REGION Network 8: IMMEDIATE STOP ALARMS
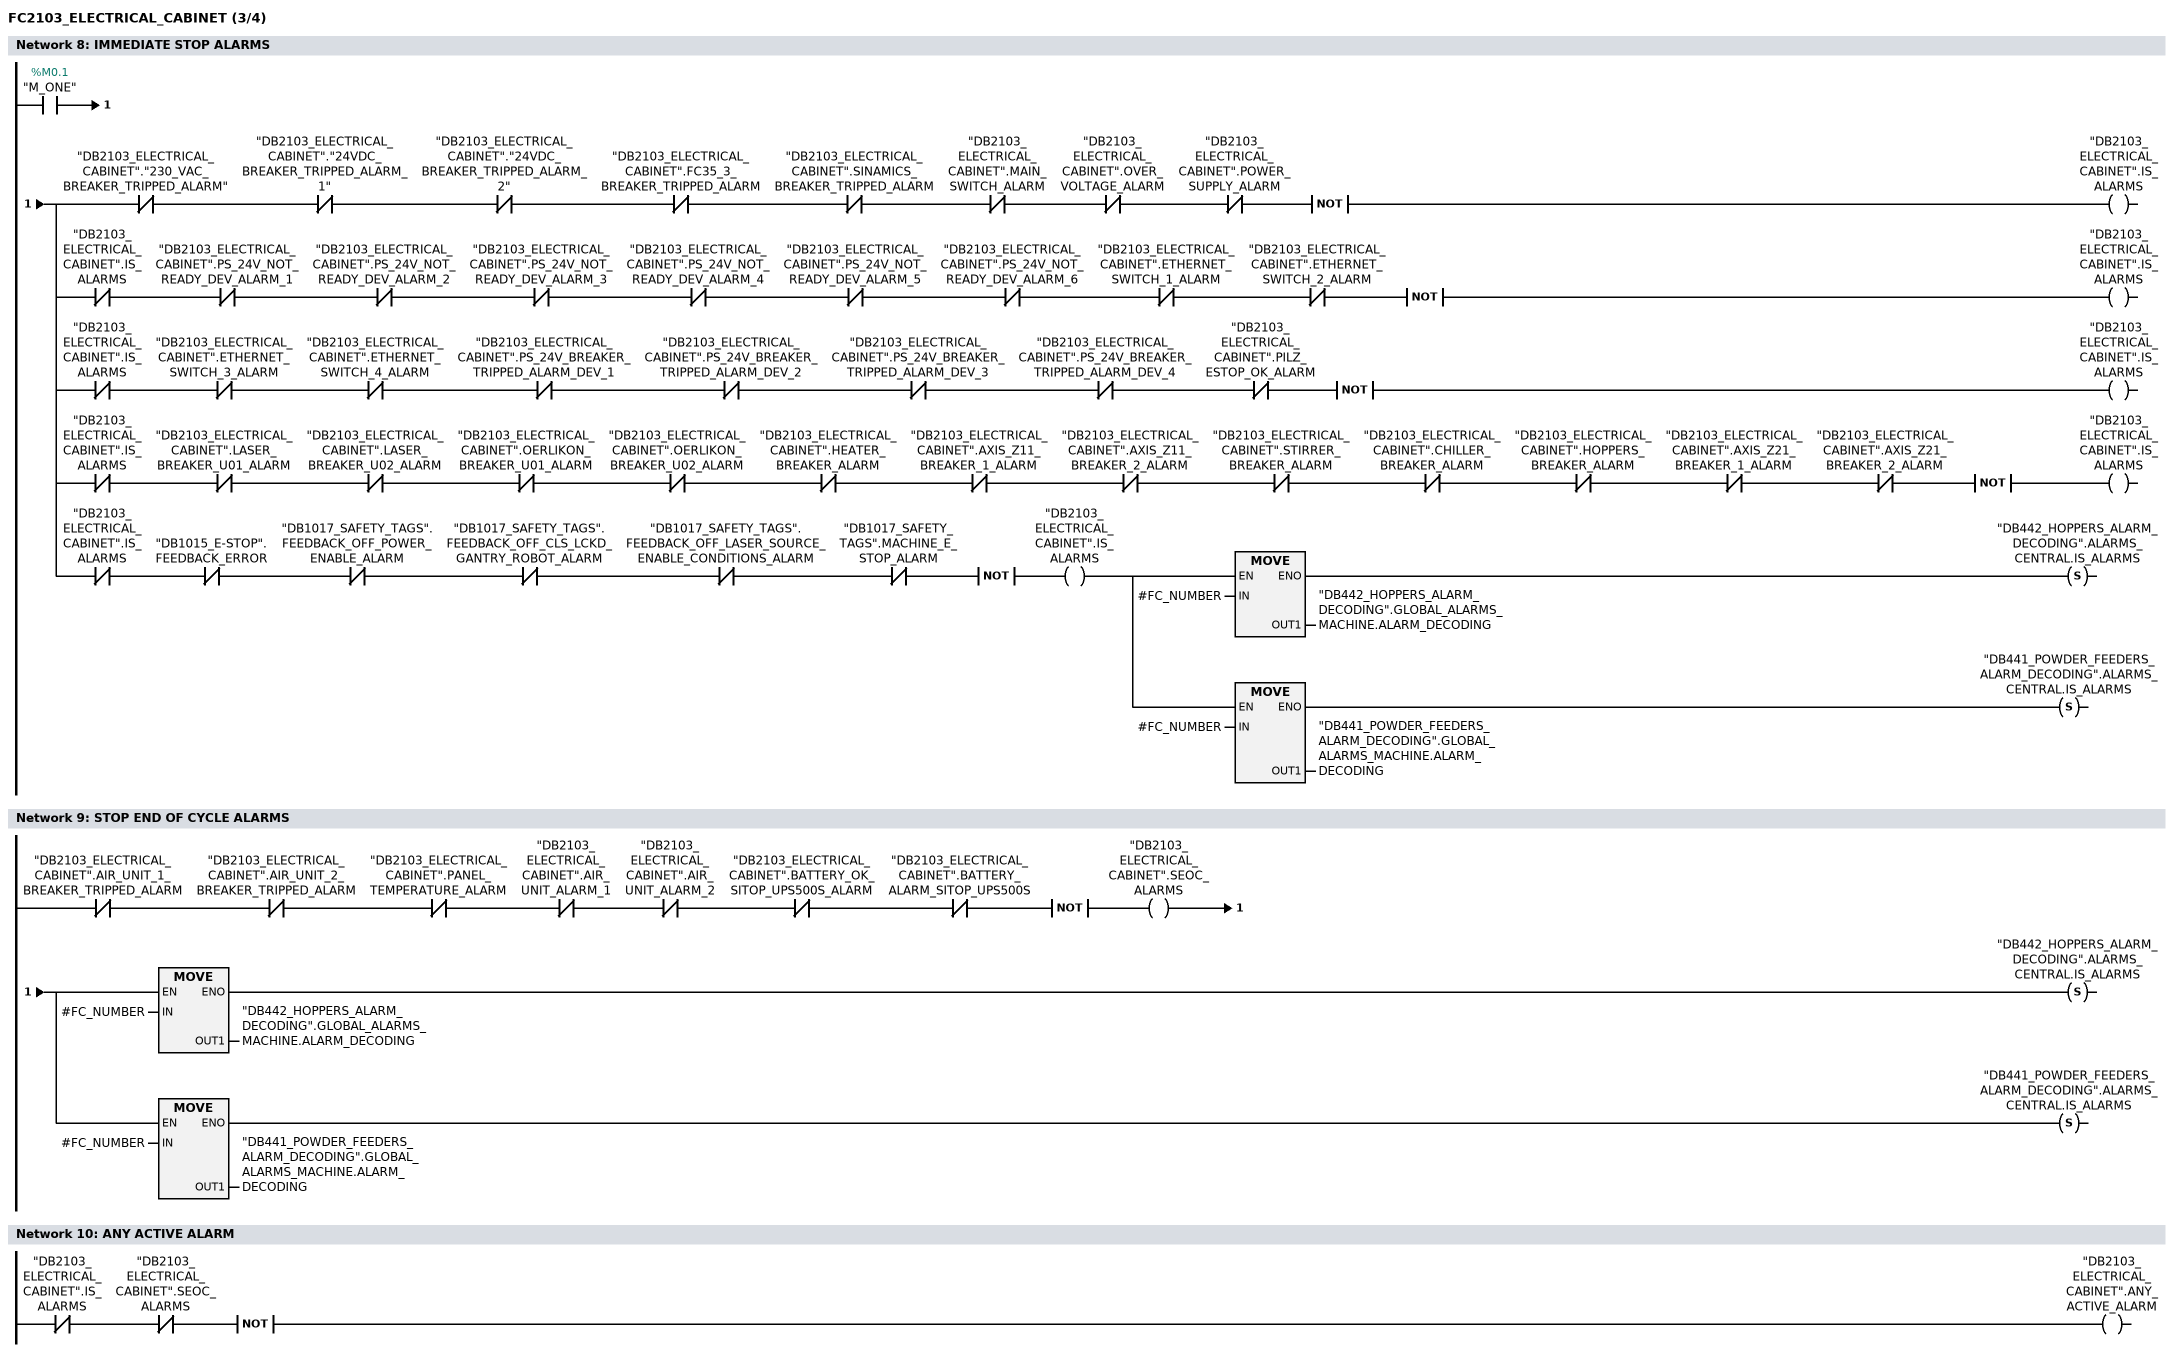
   RUNG wire#powerrail
      Contact( "M_ONE" )
      wire#w1
      I_Contact( "DB2103_ELECTRICAL_CABINET"."230_VAC_BREAKER_TRIPPED_ALARM" )
      I_Contact( "DB2103_ELECTRICAL_CABINET"."24VDC_BREAKER_TRIPPED_ALARM_1" )
      I_Contact( "DB2103_ELECTRICAL_CABINET"."24VDC_BREAKER_TRIPPED_ALARM_2" )
      I_Contact( "DB2103_ELECTRICAL_CABINET".FC35_3_BREAKER_TRIPPED_ALARM )
      I_Contact( "DB2103_ELECTRICAL_CABINET".SINAMICS_BREAKER_TRIPPED_ALARM )
      I_Contact( "DB2103_ELECTRICAL_CABINET".MAIN_SWITCH_ALARM )
      I_Contact( "DB2103_ELECTRICAL_CABINET".OVER_VOLTAGE_ALARM )
      I_Contact( "DB2103_ELECTRICAL_CABINET".POWER_SUPPLY_ALARM )
      Not()
      Coil( "DB2103_ELECTRICAL_CABINET".IS_ALARMS )
   END_RUNG
   RUNG wire#w1
      I_Contact( "DB2103_ELECTRICAL_CABINET".IS_ALARMS )
      I_Contact( "DB2103_ELECTRICAL_CABINET".PS_24V_NOT_READY_DEV_ALARM_1 )
      I_Contact( "DB2103_ELECTRICAL_CABINET".PS_24V_NOT_READY_DEV_ALARM_2 )
      I_Contact( "DB2103_ELECTRICAL_CABINET".PS_24V_NOT_READY_DEV_ALARM_3 )
      I_Contact( "DB2103_ELECTRICAL_CABINET".PS_24V_NOT_READY_DEV_ALARM_4 )
      I_Contact( "DB2103_ELECTRICAL_CABINET".PS_24V_NOT_READY_DEV_ALARM_5 )
      I_Contact( "DB2103_ELECTRICAL_CABINET".PS_24V_NOT_READY_DEV_ALARM_6 )
      I_Contact( "DB2103_ELECTRICAL_CABINET".ETHERNET_SWITCH_1_ALARM )
      I_Contact( "DB2103_ELECTRICAL_CABINET".ETHERNET_SWITCH_2_ALARM )
      Not()
      Coil( "DB2103_ELECTRICAL_CABINET".IS_ALARMS )
   END_RUNG
   RUNG wire#w1
      I_Contact( "DB2103_ELECTRICAL_CABINET".IS_ALARMS )
      I_Contact( "DB2103_ELECTRICAL_CABINET".ETHERNET_SWITCH_3_ALARM )
      I_Contact( "DB2103_ELECTRICAL_CABINET".ETHERNET_SWITCH_4_ALARM )
      I_Contact( "DB2103_ELECTRICAL_CABINET".PS_24V_BREAKER_TRIPPED_ALARM_DEV_1 )
      I_Contact( "DB2103_ELECTRICAL_CABINET".PS_24V_BREAKER_TRIPPED_ALARM_DEV_2 )
      I_Contact( "DB2103_ELECTRICAL_CABINET".PS_24V_BREAKER_TRIPPED_ALARM_DEV_3 )
      I_Contact( "DB2103_ELECTRICAL_CABINET".PS_24V_BREAKER_TRIPPED_ALARM_DEV_4 )
      I_Contact( "DB2103_ELECTRICAL_CABINET".PILZ_ESTOP_OK_ALARM )
      Not()
      Coil( "DB2103_ELECTRICAL_CABINET".IS_ALARMS )
   END_RUNG
   RUNG wire#w1
      I_Contact( "DB2103_ELECTRICAL_CABINET".IS_ALARMS )
      I_Contact( "DB2103_ELECTRICAL_CABINET".LASER_BREAKER_U01_ALARM )
      I_Contact( "DB2103_ELECTRICAL_CABINET".LASER_BREAKER_U02_ALARM )
      I_Contact( "DB2103_ELECTRICAL_CABINET".OERLIKON_BREAKER_U01_ALARM )
      I_Contact( "DB2103_ELECTRICAL_CABINET".OERLIKON_BREAKER_U02_ALARM )
      I_Contact( "DB2103_ELECTRICAL_CABINET".HEATER_BREAKER_ALARM )
      I_Contact( "DB2103_ELECTRICAL_CABINET".AXIS_Z11_BREAKER_1_ALARM )
      I_Contact( "DB2103_ELECTRICAL_CABINET".AXIS_Z11_BREAKER_2_ALARM )
      I_Contact( "DB2103_ELECTRICAL_CABINET".STIRRER_BREAKER_ALARM )
      I_Contact( "DB2103_ELECTRICAL_CABINET".CHILLER_BREAKER_ALARM )
      I_Contact( "DB2103_ELECTRICAL_CABINET".HOPPERS_BREAKER_ALARM )
      I_Contact( "DB2103_ELECTRICAL_CABINET".AXIS_Z21_BREAKER_1_ALARM )
      I_Contact( "DB2103_ELECTRICAL_CABINET".AXIS_Z21_BREAKER_2_ALARM )
      Not()
      Coil( "DB2103_ELECTRICAL_CABINET".IS_ALARMS )
   END_RUNG
   RUNG wire#w1
      I_Contact( "DB2103_ELECTRICAL_CABINET".IS_ALARMS )
      I_Contact( "DB1015_E-STOP".FEEDBACK_ERROR )
      I_Contact( "DB1017_SAFETY_TAGS".FEEDBACK_OFF_POWER_ENABLE_ALARM )
      I_Contact( "DB1017_SAFETY_TAGS".FEEDBACK_OFF_CLS_LCKD_GANTRY_ROBOT_ALARM )
      I_Contact( "DB1017_SAFETY_TAGS".FEEDBACK_OFF_LASER_SOURCE_ENABLE_CONDITIONS_ALARM )
      I_Contact( "DB1017_SAFETY_TAGS".MACHINE_E_STOP_ALARM )
      Not()
      Coil( "DB2103_ELECTRICAL_CABINET".IS_ALARMS )
      wire#w2
      { S7_GenerateENO := "TRUE" } Move(in := #FC_NUMBER, out1 => "DB442_HOPPERS_ALARM_DECODING".GLOBAL_ALARMS_MACHINE.ALARM_DECODING)
      S_Coil( "DB442_HOPPERS_ALARM_DECODING".ALARMS_CENTRAL.IS_ALARMS )
   END_RUNG
   RUNG wire#w2
      { S7_GenerateENO := "TRUE" } Move(in := #FC_NUMBER, out1 => "DB441_POWDER_FEEDERS_ALARM_DECODING".GLOBAL_ALARMS_MACHINE.ALARM_DECODING)
      S_Coil( "DB441_POWDER_FEEDERS_ALARM_DECODING".ALARMS_CENTRAL.IS_ALARMS )
   END_RUNG
   // the same network as SCL:
   // ENO of a box is taken as its EN; it also drops when the box reports an error
   "DB2103_ELECTRICAL_CABINET".IS_ALARMS := NOT ("M_ONE" AND NOT "DB2103_ELECTRICAL_CABINET"."230_VAC_BREAKER_TRIPPED_ALARM" AND NOT "DB2103_ELECTRICAL_CABINET"."24VDC_BREAKER_TRIPPED_ALARM_1" AND NOT "DB2103_ELECTRICAL_CABINET"."24VDC_BREAKER_TRIPPED_ALARM_2" AND NOT "DB2103_ELECTRICAL_CABINET".FC35_3_BREAKER_TRIPPED_ALARM AND NOT "DB2103_ELECTRICAL_CABINET".SINAMICS_BREAKER_TRIPPED_ALARM AND NOT "DB2103_ELECTRICAL_CABINET".MAIN_SWITCH_ALARM AND NOT "DB2103_ELECTRICAL_CABINET".OVER_VOLTAGE_ALARM AND NOT "DB2103_ELECTRICAL_CABINET".POWER_SUPPLY_ALARM);
   "DB2103_ELECTRICAL_CABINET".IS_ALARMS := NOT ("M_ONE" AND NOT "DB2103_ELECTRICAL_CABINET".IS_ALARMS AND NOT "DB2103_ELECTRICAL_CABINET".PS_24V_NOT_READY_DEV_ALARM_1 AND NOT "DB2103_ELECTRICAL_CABINET".PS_24V_NOT_READY_DEV_ALARM_2 AND NOT "DB2103_ELECTRICAL_CABINET".PS_24V_NOT_READY_DEV_ALARM_3 AND NOT "DB2103_ELECTRICAL_CABINET".PS_24V_NOT_READY_DEV_ALARM_4 AND NOT "DB2103_ELECTRICAL_CABINET".PS_24V_NOT_READY_DEV_ALARM_5 AND NOT "DB2103_ELECTRICAL_CABINET".PS_24V_NOT_READY_DEV_ALARM_6 AND NOT "DB2103_ELECTRICAL_CABINET".ETHERNET_SWITCH_1_ALARM AND NOT "DB2103_ELECTRICAL_CABINET".ETHERNET_SWITCH_2_ALARM);
   "DB2103_ELECTRICAL_CABINET".IS_ALARMS := NOT ("M_ONE" AND NOT "DB2103_ELECTRICAL_CABINET".IS_ALARMS AND NOT "DB2103_ELECTRICAL_CABINET".ETHERNET_SWITCH_3_ALARM AND NOT "DB2103_ELECTRICAL_CABINET".ETHERNET_SWITCH_4_ALARM AND NOT "DB2103_ELECTRICAL_CABINET".PS_24V_BREAKER_TRIPPED_ALARM_DEV_1 AND NOT "DB2103_ELECTRICAL_CABINET".PS_24V_BREAKER_TRIPPED_ALARM_DEV_2 AND NOT "DB2103_ELECTRICAL_CABINET".PS_24V_BREAKER_TRIPPED_ALARM_DEV_3 AND NOT "DB2103_ELECTRICAL_CABINET".PS_24V_BREAKER_TRIPPED_ALARM_DEV_4 AND NOT "DB2103_ELECTRICAL_CABINET".PILZ_ESTOP_OK_ALARM);
   "DB2103_ELECTRICAL_CABINET".IS_ALARMS := NOT ("M_ONE" AND NOT "DB2103_ELECTRICAL_CABINET".IS_ALARMS AND NOT "DB2103_ELECTRICAL_CABINET".LASER_BREAKER_U01_ALARM AND NOT "DB2103_ELECTRICAL_CABINET".LASER_BREAKER_U02_ALARM AND NOT "DB2103_ELECTRICAL_CABINET".OERLIKON_BREAKER_U01_ALARM AND NOT "DB2103_ELECTRICAL_CABINET".OERLIKON_BREAKER_U02_ALARM AND NOT "DB2103_ELECTRICAL_CABINET".HEATER_BREAKER_ALARM AND NOT "DB2103_ELECTRICAL_CABINET".AXIS_Z11_BREAKER_1_ALARM AND NOT "DB2103_ELECTRICAL_CABINET".AXIS_Z11_BREAKER_2_ALARM AND NOT "DB2103_ELECTRICAL_CABINET".STIRRER_BREAKER_ALARM AND NOT "DB2103_ELECTRICAL_CABINET".CHILLER_BREAKER_ALARM AND NOT "DB2103_ELECTRICAL_CABINET".HOPPERS_BREAKER_ALARM AND NOT "DB2103_ELECTRICAL_CABINET".AXIS_Z21_BREAKER_1_ALARM AND NOT "DB2103_ELECTRICAL_CABINET".AXIS_Z21_BREAKER_2_ALARM);
   "DB2103_ELECTRICAL_CABINET".IS_ALARMS := NOT ("M_ONE" AND NOT "DB2103_ELECTRICAL_CABINET".IS_ALARMS AND NOT "DB1015_E-STOP".FEEDBACK_ERROR AND NOT "DB1017_SAFETY_TAGS".FEEDBACK_OFF_POWER_ENABLE_ALARM AND NOT "DB1017_SAFETY_TAGS".FEEDBACK_OFF_CLS_LCKD_GANTRY_ROBOT_ALARM AND NOT "DB1017_SAFETY_TAGS".FEEDBACK_OFF_LASER_SOURCE_ENABLE_CONDITIONS_ALARM AND NOT "DB1017_SAFETY_TAGS".MACHINE_E_STOP_ALARM);
   IF "DB2103_ELECTRICAL_CABINET".IS_ALARMS THEN
       "DB442_HOPPERS_ALARM_DECODING".GLOBAL_ALARMS_MACHINE.ALARM_DECODING := #FC_NUMBER;
       "DB442_HOPPERS_ALARM_DECODING".ALARMS_CENTRAL.IS_ALARMS := TRUE;
       "DB441_POWDER_FEEDERS_ALARM_DECODING".GLOBAL_ALARMS_MACHINE.ALARM_DECODING := #FC_NUMBER;
       "DB441_POWDER_FEEDERS_ALARM_DECODING".ALARMS_CENTRAL.IS_ALARMS := TRUE;
   END_IF;
END_REGION

REGION Network 9: STOP END OF CYCLE ALARMS
   RUNG wire#powerrail
      I_Contact( "DB2103_ELECTRICAL_CABINET".AIR_UNIT_1_BREAKER_TRIPPED_ALARM )
      I_Contact( "DB2103_ELECTRICAL_CABINET".AIR_UNIT_2_BREAKER_TRIPPED_ALARM )
      I_Contact( "DB2103_ELECTRICAL_CABINET".PANEL_TEMPERATURE_ALARM )
      I_Contact( "DB2103_ELECTRICAL_CABINET".AIR_UNIT_ALARM_1 )
      I_Contact( "DB2103_ELECTRICAL_CABINET".AIR_UNIT_ALARM_2 )
      I_Contact( "DB2103_ELECTRICAL_CABINET".BATTERY_OK_SITOP_UPS500S_ALARM )
      I_Contact( "DB2103_ELECTRICAL_CABINET".BATTERY_ALARM_SITOP_UPS500S )
      Not()
      Coil( "DB2103_ELECTRICAL_CABINET".SEOC_ALARMS )
      wire#w1
      { S7_GenerateENO := "TRUE" } Move(in := #FC_NUMBER, out1 => "DB442_HOPPERS_ALARM_DECODING".GLOBAL_ALARMS_MACHINE.ALARM_DECODING)
      S_Coil( "DB442_HOPPERS_ALARM_DECODING".ALARMS_CENTRAL.IS_ALARMS )
   END_RUNG
   RUNG wire#w1
      { S7_GenerateENO := "TRUE" } Move(in := #FC_NUMBER, out1 => "DB441_POWDER_FEEDERS_ALARM_DECODING".GLOBAL_ALARMS_MACHINE.ALARM_DECODING)
      S_Coil( "DB441_POWDER_FEEDERS_ALARM_DECODING".ALARMS_CENTRAL.IS_ALARMS )
   END_RUNG
   // the same network as SCL:
   // ENO of a box is taken as its EN; it also drops when the box reports an error
   "DB2103_ELECTRICAL_CABINET".SEOC_ALARMS := NOT (NOT "DB2103_ELECTRICAL_CABINET".AIR_UNIT_1_BREAKER_TRIPPED_ALARM AND NOT "DB2103_ELECTRICAL_CABINET".AIR_UNIT_2_BREAKER_TRIPPED_ALARM AND NOT "DB2103_ELECTRICAL_CABINET".PANEL_TEMPERATURE_ALARM AND NOT "DB2103_ELECTRICAL_CABINET".AIR_UNIT_ALARM_1 AND NOT "DB2103_ELECTRICAL_CABINET".AIR_UNIT_ALARM_2 AND NOT "DB2103_ELECTRICAL_CABINET".BATTERY_OK_SITOP_UPS500S_ALARM AND NOT "DB2103_ELECTRICAL_CABINET".BATTERY_ALARM_SITOP_UPS500S);
   IF "DB2103_ELECTRICAL_CABINET".SEOC_ALARMS THEN
       "DB442_HOPPERS_ALARM_DECODING".GLOBAL_ALARMS_MACHINE.ALARM_DECODING := #FC_NUMBER;
       "DB442_HOPPERS_ALARM_DECODING".ALARMS_CENTRAL.IS_ALARMS := TRUE;
       "DB441_POWDER_FEEDERS_ALARM_DECODING".GLOBAL_ALARMS_MACHINE.ALARM_DECODING := #FC_NUMBER;
       "DB441_POWDER_FEEDERS_ALARM_DECODING".ALARMS_CENTRAL.IS_ALARMS := TRUE;
   END_IF;
END_REGION

REGION Network 10: ANY ACTIVE ALARM
   RUNG wire#powerrail
      I_Contact( "DB2103_ELECTRICAL_CABINET".IS_ALARMS )
      I_Contact( "DB2103_ELECTRICAL_CABINET".SEOC_ALARMS )
      Not()
      Coil( "DB2103_ELECTRICAL_CABINET".ANY_ACTIVE_ALARM )
   END_RUNG
   // the same network as SCL:
   "DB2103_ELECTRICAL_CABINET".ANY_ACTIVE_ALARM := NOT (NOT "DB2103_ELECTRICAL_CABINET".IS_ALARMS AND NOT "DB2103_ELECTRICAL_CABINET".SEOC_ALARMS);
END_REGION

REGION Network 11: WARNINGS
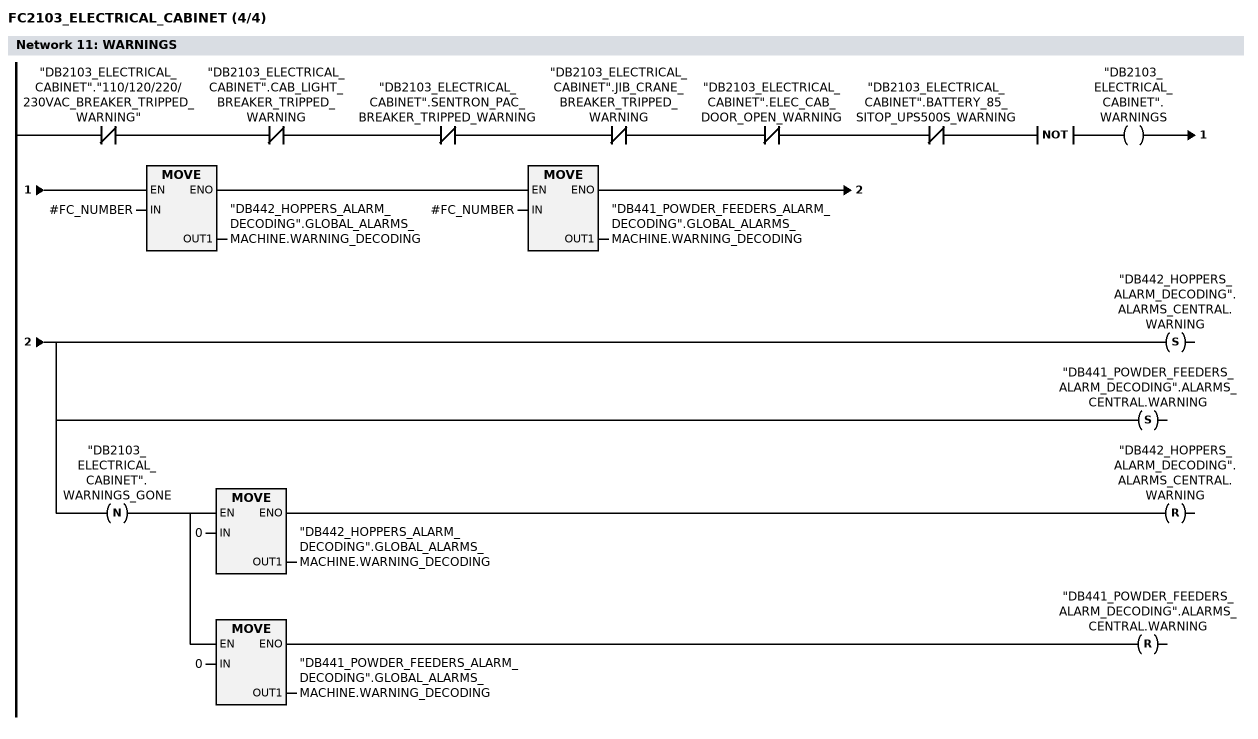
   RUNG wire#powerrail
      I_Contact( "DB2103_ELECTRICAL_CABINET"."110/120/220/230VAC_BREAKER_TRIPPED_WARNING" )
      I_Contact( "DB2103_ELECTRICAL_CABINET".CAB_LIGHT_BREAKER_TRIPPED_WARNING )
      I_Contact( "DB2103_ELECTRICAL_CABINET".SENTRON_PAC_BREAKER_TRIPPED_WARNING )
      I_Contact( "DB2103_ELECTRICAL_CABINET".JIB_CRANE_BREAKER_TRIPPED_WARNING )
      I_Contact( "DB2103_ELECTRICAL_CABINET".ELEC_CAB_DOOR_OPEN_WARNING )
      I_Contact( "DB2103_ELECTRICAL_CABINET".BATTERY_85_SITOP_UPS500S_WARNING )
      Not()
      Coil( "DB2103_ELECTRICAL_CABINET".WARNINGS )
      { S7_GenerateENO := "TRUE" } Move(in := #FC_NUMBER, out1 => "DB442_HOPPERS_ALARM_DECODING".GLOBAL_ALARMS_MACHINE.WARNING_DECODING)
      { S7_GenerateENO := "TRUE" } Move(in := #FC_NUMBER, out1 => "DB441_POWDER_FEEDERS_ALARM_DECODING".GLOBAL_ALARMS_MACHINE.WARNING_DECODING)
      wire#w1
      S_Coil( "DB442_HOPPERS_ALARM_DECODING".ALARMS_CENTRAL.WARNING )
   END_RUNG
   RUNG wire#w1
      S_Coil( "DB441_POWDER_FEEDERS_ALARM_DECODING".ALARMS_CENTRAL.WARNING )
   END_RUNG
   RUNG wire#w1
      N_Trig( "DB2103_ELECTRICAL_CABINET".WARNINGS_GONE )
      wire#w2
      { S7_GenerateENO := "TRUE" } Move(in := 0, out1 => "DB442_HOPPERS_ALARM_DECODING".GLOBAL_ALARMS_MACHINE.WARNING_DECODING)
      R_Coil( "DB442_HOPPERS_ALARM_DECODING".ALARMS_CENTRAL.WARNING )
   END_RUNG
   RUNG wire#w2
      { S7_GenerateENO := "TRUE" } Move(in := 0, out1 => "DB441_POWDER_FEEDERS_ALARM_DECODING".GLOBAL_ALARMS_MACHINE.WARNING_DECODING)
      R_Coil( "DB441_POWDER_FEEDERS_ALARM_DECODING".ALARMS_CENTRAL.WARNING )
   END_RUNG
   // the same network as SCL:
   // ENO of a box is taken as its EN; it also drops when the box reports an error
   "DB2103_ELECTRICAL_CABINET".WARNINGS := NOT (NOT "DB2103_ELECTRICAL_CABINET"."110/120/220/230VAC_BREAKER_TRIPPED_WARNING" AND NOT "DB2103_ELECTRICAL_CABINET".CAB_LIGHT_BREAKER_TRIPPED_WARNING AND NOT "DB2103_ELECTRICAL_CABINET".SENTRON_PAC_BREAKER_TRIPPED_WARNING AND NOT "DB2103_ELECTRICAL_CABINET".JIB_CRANE_BREAKER_TRIPPED_WARNING AND NOT "DB2103_ELECTRICAL_CABINET".ELEC_CAB_DOOR_OPEN_WARNING AND NOT "DB2103_ELECTRICAL_CABINET".BATTERY_85_SITOP_UPS500S_WARNING);
   IF "DB2103_ELECTRICAL_CABINET".WARNINGS THEN
       "DB442_HOPPERS_ALARM_DECODING".GLOBAL_ALARMS_MACHINE.WARNING_DECODING := #FC_NUMBER;
       "DB441_POWDER_FEEDERS_ALARM_DECODING".GLOBAL_ALARMS_MACHINE.WARNING_DECODING := #FC_NUMBER;
       "DB442_HOPPERS_ALARM_DECODING".ALARMS_CENTRAL.WARNING := TRUE;
       "DB441_POWDER_FEEDERS_ALARM_DECODING".ALARMS_CENTRAL.WARNING := TRUE;
   END_IF;
   #_w1 := NOT "DB2103_ELECTRICAL_CABINET".WARNINGS AND "DB2103_ELECTRICAL_CABINET".WARNINGS_GONE;   // falling edge
   "DB2103_ELECTRICAL_CABINET".WARNINGS_GONE := "DB2103_ELECTRICAL_CABINET".WARNINGS;
   IF #_w1 THEN
       "DB442_HOPPERS_ALARM_DECODING".GLOBAL_ALARMS_MACHINE.WARNING_DECODING := 0;
       "DB442_HOPPERS_ALARM_DECODING".ALARMS_CENTRAL.WARNING := FALSE;
       "DB441_POWDER_FEEDERS_ALARM_DECODING".GLOBAL_ALARMS_MACHINE.WARNING_DECODING := 0;
       "DB441_POWDER_FEEDERS_ALARM_DECODING".ALARMS_CENTRAL.WARNING := FALSE;
   END_IF;
END_REGION
END_FUNCTION

FUNCTION "FC2120_MPP_ITC_IPC" : Void   // FC2120, LAD
{ S7_Optimized_Access := 'FALSE' }
AUTHOR : ETXETAR
VERSION : 1.0
// stored: AutoNumber false, IsIECCheckEnabled false, SetENOAutomatically false, UDAEnableTagReadback false
   VAR_TEMP
      O_BYTE_0 : Struct   // OPTIONS BYTE 0
         IPC : Bool;   // IPC OPTION
      END_STRUCT;
      TCU_INDEX_SEL : Int;
   END_VAR
   VAR CONSTANT
      FC_NUMBER : DInt := 2120;   // FC NUMBER
   END_VAR
   VAR_TEMP   // added for the SCL form of the ladder/FBD networks
      _w1 : Bool;
      _w2 : Bool;
   END_VAR
BEGIN

REGION Network 1: OPTIONS
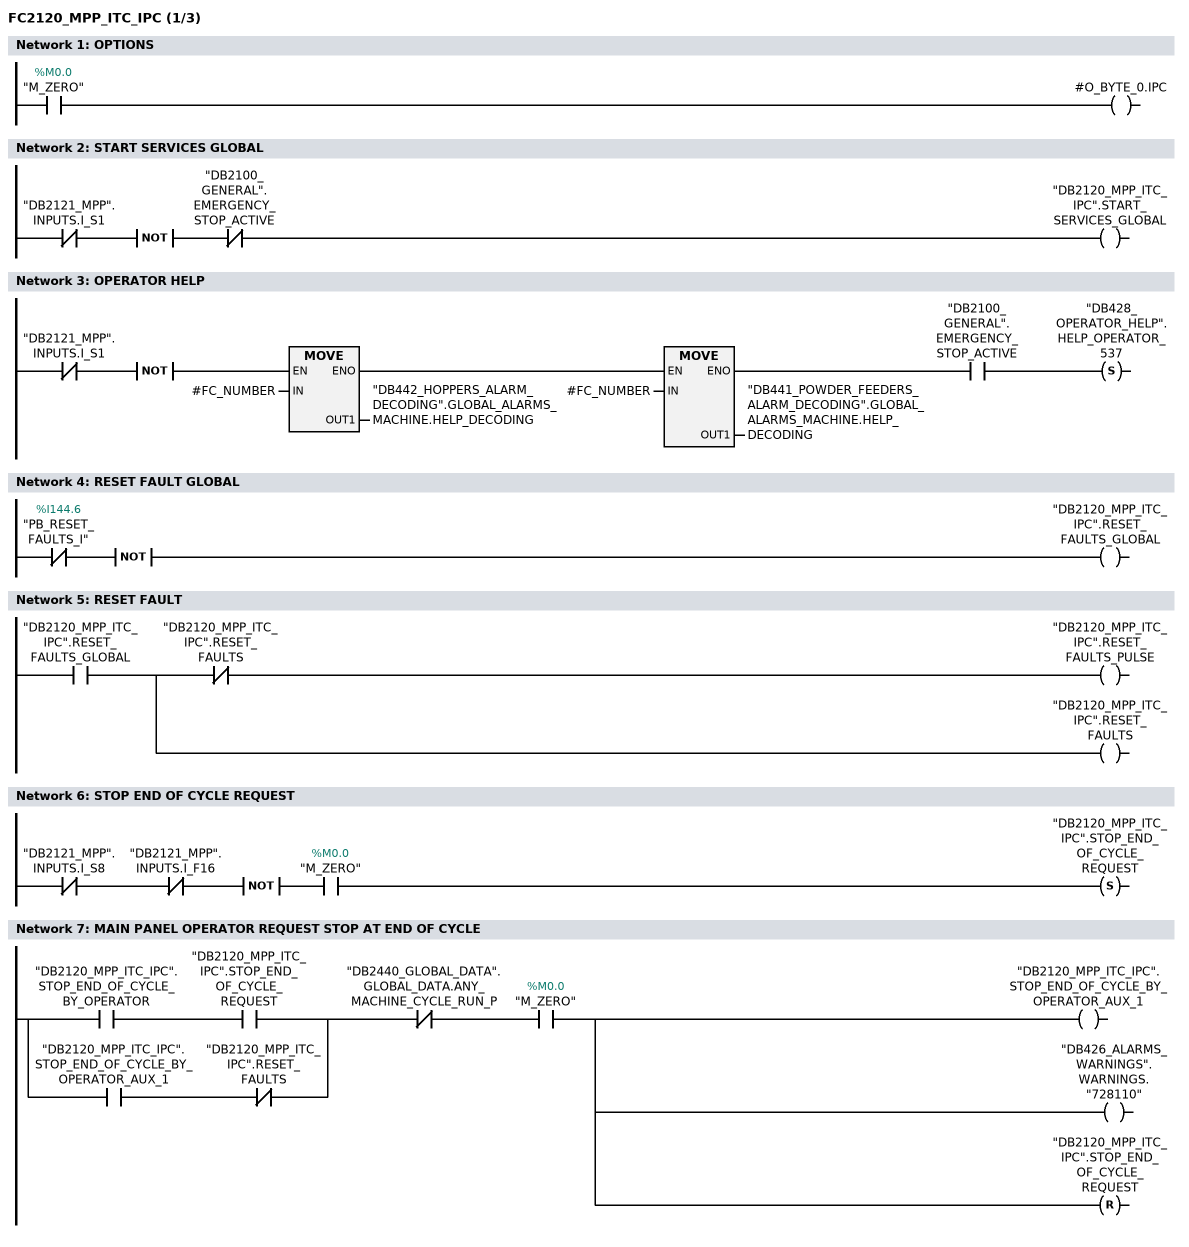
   RUNG wire#powerrail
      Contact( "M_ZERO" )
      Coil( #O_BYTE_0.IPC )
   END_RUNG
   // the same network as SCL:
   #O_BYTE_0.IPC := "M_ZERO";
END_REGION

REGION Network 2: START SERVICES GLOBAL
   RUNG wire#powerrail
      I_Contact( "DB2121_MPP".INPUTS.I_S1 )
      Not()
      I_Contact( "DB2100_GENERAL".EMERGENCY_STOP_ACTIVE )
      Coil( "DB2120_MPP_ITC_IPC".START_SERVICES_GLOBAL )
   END_RUNG
   // the same network as SCL:
   "DB2120_MPP_ITC_IPC".START_SERVICES_GLOBAL := NOT (NOT "DB2121_MPP".INPUTS.I_S1) AND NOT "DB2100_GENERAL".EMERGENCY_STOP_ACTIVE;
END_REGION

REGION Network 3: OPERATOR HELP
   RUNG wire#powerrail
      I_Contact( "DB2121_MPP".INPUTS.I_S1 )
      Not()
      { S7_GenerateENO := "TRUE" } Move(in := #FC_NUMBER, out1 => "DB442_HOPPERS_ALARM_DECODING".GLOBAL_ALARMS_MACHINE.HELP_DECODING)
      { S7_GenerateENO := "TRUE" } Move(in := #FC_NUMBER, out1 => "DB441_POWDER_FEEDERS_ALARM_DECODING".GLOBAL_ALARMS_MACHINE.HELP_DECODING)
      Contact( "DB2100_GENERAL".EMERGENCY_STOP_ACTIVE )
      S_Coil( "DB428_OPERATOR_HELP".HELP_OPERATOR_537 )
   END_RUNG
   // the same network as SCL:
   // ENO of a box is taken as its EN; it also drops when the box reports an error
   #_w1 := NOT (NOT "DB2121_MPP".INPUTS.I_S1);
   IF #_w1 THEN
       "DB442_HOPPERS_ALARM_DECODING".GLOBAL_ALARMS_MACHINE.HELP_DECODING := #FC_NUMBER;
       "DB441_POWDER_FEEDERS_ALARM_DECODING".GLOBAL_ALARMS_MACHINE.HELP_DECODING := #FC_NUMBER;
   END_IF;
   IF #_w1 AND "DB2100_GENERAL".EMERGENCY_STOP_ACTIVE THEN
       "DB428_OPERATOR_HELP".HELP_OPERATOR_537 := TRUE;
   END_IF;
END_REGION

REGION Network 4: RESET FAULT GLOBAL
   RUNG wire#powerrail
      I_Contact( "PB_RESET_FAULTS_I" )
      Not()
      Coil( "DB2120_MPP_ITC_IPC".RESET_FAULTS_GLOBAL )
   END_RUNG
   // the same network as SCL:
   "DB2120_MPP_ITC_IPC".RESET_FAULTS_GLOBAL := NOT (NOT "PB_RESET_FAULTS_I");
END_REGION

REGION Network 5: RESET FAULT
   RUNG wire#powerrail
      Contact( "DB2120_MPP_ITC_IPC".RESET_FAULTS_GLOBAL )
      wire#w1
      I_Contact( "DB2120_MPP_ITC_IPC".RESET_FAULTS )
      Coil( "DB2120_MPP_ITC_IPC".RESET_FAULTS_PULSE )
   END_RUNG
   RUNG wire#w1
      Coil( "DB2120_MPP_ITC_IPC".RESET_FAULTS )
   END_RUNG
   // the same network as SCL:
   "DB2120_MPP_ITC_IPC".RESET_FAULTS_PULSE := "DB2120_MPP_ITC_IPC".RESET_FAULTS_GLOBAL AND NOT "DB2120_MPP_ITC_IPC".RESET_FAULTS;
   "DB2120_MPP_ITC_IPC".RESET_FAULTS := "DB2120_MPP_ITC_IPC".RESET_FAULTS_GLOBAL;
END_REGION

REGION Network 6: STOP END OF CYCLE REQUEST
   RUNG wire#powerrail
      I_Contact( "DB2121_MPP".INPUTS.I_S8 )
      I_Contact( "DB2121_MPP".INPUTS.I_F16 )
      Not()
      Contact( "M_ZERO" )
      S_Coil( "DB2120_MPP_ITC_IPC".STOP_END_OF_CYCLE_REQUEST )
   END_RUNG
   // the same network as SCL:
   IF NOT (NOT "DB2121_MPP".INPUTS.I_S8 AND NOT "DB2121_MPP".INPUTS.I_F16) AND "M_ZERO" THEN
       "DB2120_MPP_ITC_IPC".STOP_END_OF_CYCLE_REQUEST := TRUE;
   END_IF;
END_REGION

REGION Network 7: MAIN PANEL OPERATOR REQUEST STOP AT END OF CYCLE
   RUNG wire#powerrail
      Contact( "DB2120_MPP_ITC_IPC".STOP_END_OF_CYCLE_BY_OPERATOR )
      Contact( "DB2120_MPP_ITC_IPC".STOP_END_OF_CYCLE_REQUEST )
      wire#w1
      I_Contact( "DB2440_GLOBAL_DATA".GLOBAL_DATA.ANY_MACHINE_CYCLE_RUN_P )
      Contact( "M_ZERO" )
      wire#w2
      Coil( "DB2120_MPP_ITC_IPC".STOP_END_OF_CYCLE_BY_OPERATOR_AUX_1 )
   END_RUNG
   RUNG wire#powerrail
      Contact( "DB2120_MPP_ITC_IPC".STOP_END_OF_CYCLE_BY_OPERATOR_AUX_1 )
      I_Contact( "DB2120_MPP_ITC_IPC".RESET_FAULTS )
   END_RUNG wire#w1
   RUNG wire#w2
      Coil( "DB426_ALARMS_WARNINGS".WARNINGS."728110" )
   END_RUNG
   RUNG wire#w2
      R_Coil( "DB2120_MPP_ITC_IPC".STOP_END_OF_CYCLE_REQUEST )
   END_RUNG
   // the same network as SCL:
   "DB2120_MPP_ITC_IPC".STOP_END_OF_CYCLE_BY_OPERATOR_AUX_1 := (("DB2120_MPP_ITC_IPC".STOP_END_OF_CYCLE_BY_OPERATOR AND "DB2120_MPP_ITC_IPC".STOP_END_OF_CYCLE_REQUEST) OR ("DB2120_MPP_ITC_IPC".STOP_END_OF_CYCLE_BY_OPERATOR_AUX_1 AND NOT "DB2120_MPP_ITC_IPC".RESET_FAULTS)) AND NOT "DB2440_GLOBAL_DATA".GLOBAL_DATA.ANY_MACHINE_CYCLE_RUN_P AND "M_ZERO";
   "DB426_ALARMS_WARNINGS".WARNINGS."728110" := "DB2120_MPP_ITC_IPC".STOP_END_OF_CYCLE_BY_OPERATOR_AUX_1;
   IF "DB2120_MPP_ITC_IPC".STOP_END_OF_CYCLE_BY_OPERATOR_AUX_1 THEN
       "DB2120_MPP_ITC_IPC".STOP_END_OF_CYCLE_REQUEST := FALSE;
   END_IF;
END_REGION

REGION Network 8: AUXILIARY PANEL OPERATOR REQUEST STOP AT END OF CYCLE
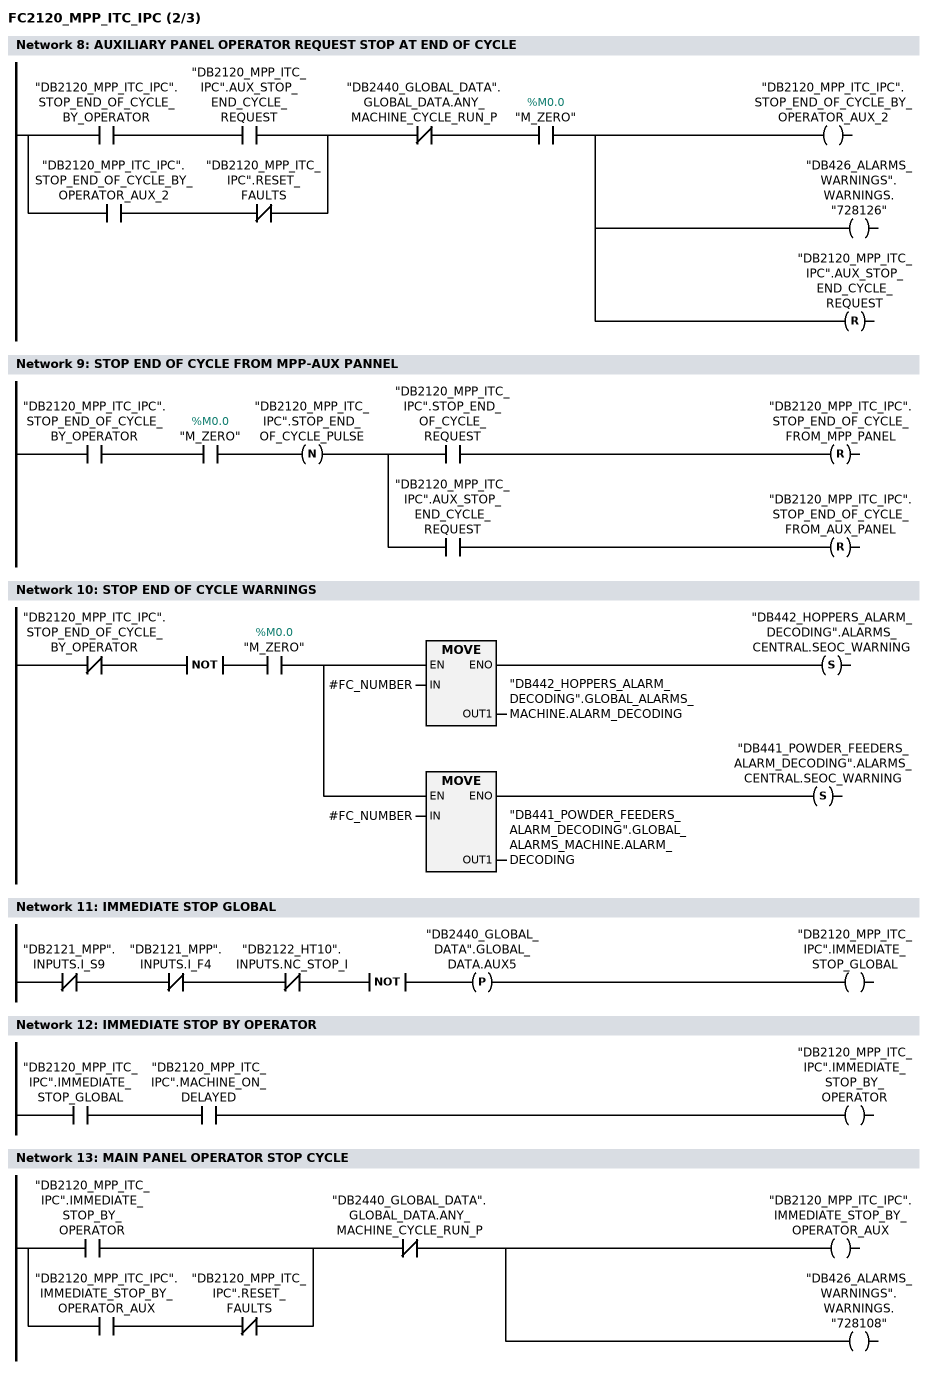
   RUNG wire#powerrail
      Contact( "DB2120_MPP_ITC_IPC".STOP_END_OF_CYCLE_BY_OPERATOR )
      Contact( "DB2120_MPP_ITC_IPC".AUX_STOP_END_CYCLE_REQUEST )
      wire#w1
      I_Contact( "DB2440_GLOBAL_DATA".GLOBAL_DATA.ANY_MACHINE_CYCLE_RUN_P )
      Contact( "M_ZERO" )
      wire#w2
      Coil( "DB2120_MPP_ITC_IPC".STOP_END_OF_CYCLE_BY_OPERATOR_AUX_2 )
   END_RUNG
   RUNG wire#powerrail
      Contact( "DB2120_MPP_ITC_IPC".STOP_END_OF_CYCLE_BY_OPERATOR_AUX_2 )
      I_Contact( "DB2120_MPP_ITC_IPC".RESET_FAULTS )
   END_RUNG wire#w1
   RUNG wire#w2
      Coil( "DB426_ALARMS_WARNINGS".WARNINGS."728126" )
   END_RUNG
   RUNG wire#w2
      R_Coil( "DB2120_MPP_ITC_IPC".AUX_STOP_END_CYCLE_REQUEST )
   END_RUNG
   // the same network as SCL:
   "DB2120_MPP_ITC_IPC".STOP_END_OF_CYCLE_BY_OPERATOR_AUX_2 := (("DB2120_MPP_ITC_IPC".STOP_END_OF_CYCLE_BY_OPERATOR AND "DB2120_MPP_ITC_IPC".AUX_STOP_END_CYCLE_REQUEST) OR ("DB2120_MPP_ITC_IPC".STOP_END_OF_CYCLE_BY_OPERATOR_AUX_2 AND NOT "DB2120_MPP_ITC_IPC".RESET_FAULTS)) AND NOT "DB2440_GLOBAL_DATA".GLOBAL_DATA.ANY_MACHINE_CYCLE_RUN_P AND "M_ZERO";
   "DB426_ALARMS_WARNINGS".WARNINGS."728126" := "DB2120_MPP_ITC_IPC".STOP_END_OF_CYCLE_BY_OPERATOR_AUX_2;
   IF "DB2120_MPP_ITC_IPC".STOP_END_OF_CYCLE_BY_OPERATOR_AUX_2 THEN
       "DB2120_MPP_ITC_IPC".AUX_STOP_END_CYCLE_REQUEST := FALSE;
   END_IF;
END_REGION

REGION Network 9: STOP END OF CYCLE FROM MPP-AUX PANNEL
   RUNG wire#powerrail
      Contact( "DB2120_MPP_ITC_IPC".STOP_END_OF_CYCLE_BY_OPERATOR )
      Contact( "M_ZERO" )
      N_Trig( "DB2120_MPP_ITC_IPC".STOP_END_OF_CYCLE_PULSE )
      wire#w1
      Contact( "DB2120_MPP_ITC_IPC".STOP_END_OF_CYCLE_REQUEST )
      R_Coil( "DB2120_MPP_ITC_IPC".STOP_END_OF_CYCLE_FROM_MPP_PANEL )
   END_RUNG
   RUNG wire#w1
      Contact( "DB2120_MPP_ITC_IPC".AUX_STOP_END_CYCLE_REQUEST )
      R_Coil( "DB2120_MPP_ITC_IPC".STOP_END_OF_CYCLE_FROM_AUX_PANEL )
   END_RUNG
   // the same network as SCL:
   #_w1 := "DB2120_MPP_ITC_IPC".STOP_END_OF_CYCLE_BY_OPERATOR AND "M_ZERO";
   #_w2 := NOT #_w1 AND "DB2120_MPP_ITC_IPC".STOP_END_OF_CYCLE_PULSE;   // falling edge
   "DB2120_MPP_ITC_IPC".STOP_END_OF_CYCLE_PULSE := #_w1;
   IF #_w2 AND "DB2120_MPP_ITC_IPC".STOP_END_OF_CYCLE_REQUEST THEN
       "DB2120_MPP_ITC_IPC".STOP_END_OF_CYCLE_FROM_MPP_PANEL := FALSE;
   END_IF;
   IF #_w2 AND "DB2120_MPP_ITC_IPC".AUX_STOP_END_CYCLE_REQUEST THEN
       "DB2120_MPP_ITC_IPC".STOP_END_OF_CYCLE_FROM_AUX_PANEL := FALSE;
   END_IF;
END_REGION

REGION Network 10: STOP END OF CYCLE WARNINGS
   RUNG wire#powerrail
      I_Contact( "DB2120_MPP_ITC_IPC".STOP_END_OF_CYCLE_BY_OPERATOR )
      Not()
      Contact( "M_ZERO" )
      wire#w1
      { S7_GenerateENO := "TRUE" } Move(in := #FC_NUMBER, out1 => "DB442_HOPPERS_ALARM_DECODING".GLOBAL_ALARMS_MACHINE.ALARM_DECODING)
      S_Coil( "DB442_HOPPERS_ALARM_DECODING".ALARMS_CENTRAL.SEOC_WARNING )
   END_RUNG
   RUNG wire#w1
      { S7_GenerateENO := "TRUE" } Move(in := #FC_NUMBER, out1 => "DB441_POWDER_FEEDERS_ALARM_DECODING".GLOBAL_ALARMS_MACHINE.ALARM_DECODING)
      S_Coil( "DB441_POWDER_FEEDERS_ALARM_DECODING".ALARMS_CENTRAL.SEOC_WARNING )
   END_RUNG
   // the same network as SCL:
   // ENO of a box is taken as its EN; it also drops when the box reports an error
   IF NOT (NOT "DB2120_MPP_ITC_IPC".STOP_END_OF_CYCLE_BY_OPERATOR) AND "M_ZERO" THEN
       "DB442_HOPPERS_ALARM_DECODING".GLOBAL_ALARMS_MACHINE.ALARM_DECODING := #FC_NUMBER;
       "DB442_HOPPERS_ALARM_DECODING".ALARMS_CENTRAL.SEOC_WARNING := TRUE;
       "DB441_POWDER_FEEDERS_ALARM_DECODING".GLOBAL_ALARMS_MACHINE.ALARM_DECODING := #FC_NUMBER;
       "DB441_POWDER_FEEDERS_ALARM_DECODING".ALARMS_CENTRAL.SEOC_WARNING := TRUE;
   END_IF;
END_REGION

REGION Network 11: IMMEDIATE STOP GLOBAL
   RUNG wire#powerrail
      I_Contact( "DB2121_MPP".INPUTS.I_S9 )
      I_Contact( "DB2121_MPP".INPUTS.I_F4 )
      I_Contact( "DB2122_HT10".INPUTS.NC_STOP_I )
      Not()
      P_Trig( "DB2440_GLOBAL_DATA".GLOBAL_DATA.AUX5 )
      Coil( "DB2120_MPP_ITC_IPC".IMMEDIATE_STOP_GLOBAL )
   END_RUNG
   // the same network as SCL:
   #_w1 := NOT (NOT "DB2121_MPP".INPUTS.I_S9 AND NOT "DB2121_MPP".INPUTS.I_F4 AND NOT "DB2122_HT10".INPUTS.NC_STOP_I);
   #_w2 := #_w1 AND NOT "DB2440_GLOBAL_DATA".GLOBAL_DATA.AUX5;   // rising edge
   "DB2440_GLOBAL_DATA".GLOBAL_DATA.AUX5 := #_w1;
   "DB2120_MPP_ITC_IPC".IMMEDIATE_STOP_GLOBAL := #_w2;
END_REGION

REGION Network 12: IMMEDIATE STOP BY OPERATOR
   RUNG wire#powerrail
      Contact( "DB2120_MPP_ITC_IPC".IMMEDIATE_STOP_GLOBAL )
      Contact( "DB2120_MPP_ITC_IPC".MACHINE_ON_DELAYED )
      Coil( "DB2120_MPP_ITC_IPC".IMMEDIATE_STOP_BY_OPERATOR )
   END_RUNG
   // the same network as SCL:
   "DB2120_MPP_ITC_IPC".IMMEDIATE_STOP_BY_OPERATOR := "DB2120_MPP_ITC_IPC".IMMEDIATE_STOP_GLOBAL AND "DB2120_MPP_ITC_IPC".MACHINE_ON_DELAYED;
END_REGION

REGION Network 13: MAIN PANEL OPERATOR STOP CYCLE
   RUNG wire#powerrail
      Contact( "DB2120_MPP_ITC_IPC".IMMEDIATE_STOP_BY_OPERATOR )
      wire#w1
      I_Contact( "DB2440_GLOBAL_DATA".GLOBAL_DATA.ANY_MACHINE_CYCLE_RUN_P )
      wire#w2
      Coil( "DB2120_MPP_ITC_IPC".IMMEDIATE_STOP_BY_OPERATOR_AUX )
   END_RUNG
   RUNG wire#powerrail
      Contact( "DB2120_MPP_ITC_IPC".IMMEDIATE_STOP_BY_OPERATOR_AUX )
      I_Contact( "DB2120_MPP_ITC_IPC".RESET_FAULTS )
   END_RUNG wire#w1
   RUNG wire#w2
      Coil( "DB426_ALARMS_WARNINGS".WARNINGS."728108" )
   END_RUNG
   // the same network as SCL:
   "DB2120_MPP_ITC_IPC".IMMEDIATE_STOP_BY_OPERATOR_AUX := ("DB2120_MPP_ITC_IPC".IMMEDIATE_STOP_BY_OPERATOR OR ("DB2120_MPP_ITC_IPC".IMMEDIATE_STOP_BY_OPERATOR_AUX AND NOT "DB2120_MPP_ITC_IPC".RESET_FAULTS)) AND NOT "DB2440_GLOBAL_DATA".GLOBAL_DATA.ANY_MACHINE_CYCLE_RUN_P;
   "DB426_ALARMS_WARNINGS".WARNINGS."728108" := "DB2120_MPP_ITC_IPC".IMMEDIATE_STOP_BY_OPERATOR_AUX;
END_REGION

REGION Network 14: IMMEDIATE STOP WARNING
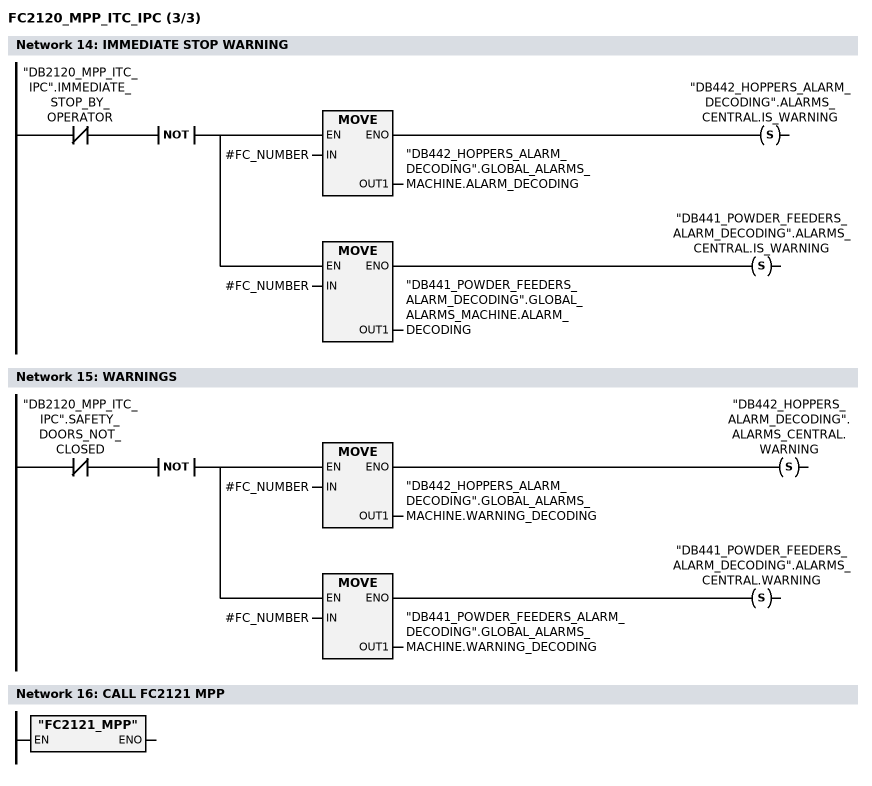
   RUNG wire#powerrail
      I_Contact( "DB2120_MPP_ITC_IPC".IMMEDIATE_STOP_BY_OPERATOR )
      Not()
      wire#w1
      { S7_GenerateENO := "TRUE" } Move(in := #FC_NUMBER, out1 => "DB442_HOPPERS_ALARM_DECODING".GLOBAL_ALARMS_MACHINE.ALARM_DECODING)
      S_Coil( "DB442_HOPPERS_ALARM_DECODING".ALARMS_CENTRAL.IS_WARNING )
   END_RUNG
   RUNG wire#w1
      { S7_GenerateENO := "TRUE" } Move(in := #FC_NUMBER, out1 => "DB441_POWDER_FEEDERS_ALARM_DECODING".GLOBAL_ALARMS_MACHINE.ALARM_DECODING)
      S_Coil( "DB441_POWDER_FEEDERS_ALARM_DECODING".ALARMS_CENTRAL.IS_WARNING )
   END_RUNG
   // the same network as SCL:
   // ENO of a box is taken as its EN; it also drops when the box reports an error
   IF NOT (NOT "DB2120_MPP_ITC_IPC".IMMEDIATE_STOP_BY_OPERATOR) THEN
       "DB442_HOPPERS_ALARM_DECODING".GLOBAL_ALARMS_MACHINE.ALARM_DECODING := #FC_NUMBER;
       "DB442_HOPPERS_ALARM_DECODING".ALARMS_CENTRAL.IS_WARNING := TRUE;
       "DB441_POWDER_FEEDERS_ALARM_DECODING".GLOBAL_ALARMS_MACHINE.ALARM_DECODING := #FC_NUMBER;
       "DB441_POWDER_FEEDERS_ALARM_DECODING".ALARMS_CENTRAL.IS_WARNING := TRUE;
   END_IF;
END_REGION

REGION Network 15: WARNINGS
   RUNG wire#powerrail
      I_Contact( "DB2120_MPP_ITC_IPC".SAFETY_DOORS_NOT_CLOSED )
      Not()
      wire#w1
      { S7_GenerateENO := "TRUE" } Move(in := #FC_NUMBER, out1 => "DB442_HOPPERS_ALARM_DECODING".GLOBAL_ALARMS_MACHINE.WARNING_DECODING)
      S_Coil( "DB442_HOPPERS_ALARM_DECODING".ALARMS_CENTRAL.WARNING )
   END_RUNG
   RUNG wire#w1
      { S7_GenerateENO := "TRUE" } Move(in := #FC_NUMBER, out1 => "DB441_POWDER_FEEDERS_ALARM_DECODING".GLOBAL_ALARMS_MACHINE.WARNING_DECODING)
      S_Coil( "DB441_POWDER_FEEDERS_ALARM_DECODING".ALARMS_CENTRAL.WARNING )
   END_RUNG
   // the same network as SCL:
   // ENO of a box is taken as its EN; it also drops when the box reports an error
   IF NOT (NOT "DB2120_MPP_ITC_IPC".SAFETY_DOORS_NOT_CLOSED) THEN
       "DB442_HOPPERS_ALARM_DECODING".GLOBAL_ALARMS_MACHINE.WARNING_DECODING := #FC_NUMBER;
       "DB442_HOPPERS_ALARM_DECODING".ALARMS_CENTRAL.WARNING := TRUE;
       "DB441_POWDER_FEEDERS_ALARM_DECODING".GLOBAL_ALARMS_MACHINE.WARNING_DECODING := #FC_NUMBER;
       "DB441_POWDER_FEEDERS_ALARM_DECODING".ALARMS_CENTRAL.WARNING := TRUE;
   END_IF;
END_REGION

REGION Network 16: CALL FC2121 MPP
   RUNG wire#powerrail
      "FC2121_MPP"()
   END_RUNG
   // the same network as SCL:
   "FC2121_MPP"();
END_REGION
END_FUNCTION

FUNCTION "FC2121_MPP" : Void   // FC2121, LAD
{ S7_Optimized_Access := 'FALSE' }
AUTHOR : ETXETAR
VERSION : 1.0
// stored: AutoNumber false, IsIECCheckEnabled false, SetENOAutomatically false, UDAEnableTagReadback false
   VAR_TEMP
      ONE : Int;
      RETVAL1 : Int;
      SIMU_PANEL_HMI_SEL : Bool;   // SIMULATED PANEL IN HMI SELECTED
   END_VAR
   VAR CONSTANT
      FC_NUMBER : DInt := 2121;   // FC NUMBER
   END_VAR
BEGIN

REGION Network 1: INPUTS
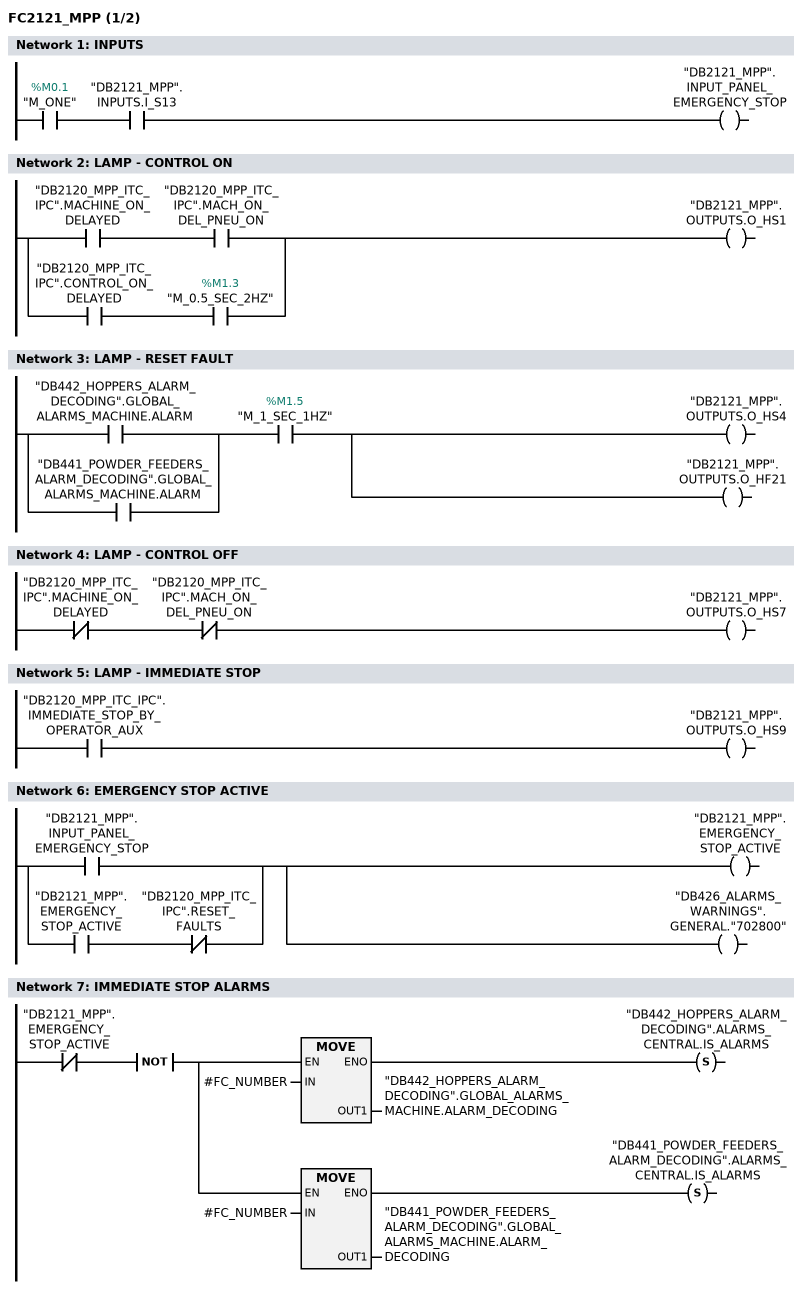
   RUNG wire#powerrail
      Contact( "M_ONE" )
      Contact( "DB2121_MPP".INPUTS.I_S13 )
      Coil( "DB2121_MPP".INPUT_PANEL_EMERGENCY_STOP )
   END_RUNG
   // the same network as SCL:
   "DB2121_MPP".INPUT_PANEL_EMERGENCY_STOP := "M_ONE" AND "DB2121_MPP".INPUTS.I_S13;
END_REGION

REGION Network 2: LAMP - CONTROL ON
   RUNG wire#powerrail
      Contact( "DB2120_MPP_ITC_IPC".MACHINE_ON_DELAYED )
      Contact( "DB2120_MPP_ITC_IPC".MACH_ON_DEL_PNEU_ON )
      wire#w1
      Coil( "DB2121_MPP".OUTPUTS.O_HS1 )
   END_RUNG
   RUNG wire#powerrail
      Contact( "DB2120_MPP_ITC_IPC".CONTROL_ON_DELAYED )
      Contact( "M_0.5_SEC_2HZ" )
   END_RUNG wire#w1
   // the same network as SCL:
   "DB2121_MPP".OUTPUTS.O_HS1 := ("DB2120_MPP_ITC_IPC".MACHINE_ON_DELAYED AND "DB2120_MPP_ITC_IPC".MACH_ON_DEL_PNEU_ON) OR ("DB2120_MPP_ITC_IPC".CONTROL_ON_DELAYED AND "M_0.5_SEC_2HZ");
END_REGION

REGION Network 3: LAMP - RESET FAULT
   RUNG wire#powerrail
      Contact( "DB442_HOPPERS_ALARM_DECODING".GLOBAL_ALARMS_MACHINE.ALARM )
      wire#w1
      Contact( "M_1_SEC_1HZ" )
      wire#w2
      Coil( "DB2121_MPP".OUTPUTS.O_HS4 )
   END_RUNG
   RUNG wire#powerrail
      Contact( "DB441_POWDER_FEEDERS_ALARM_DECODING".GLOBAL_ALARMS_MACHINE.ALARM )
   END_RUNG wire#w1
   RUNG wire#w2
      Coil( "DB2121_MPP".OUTPUTS.O_HF21 )
   END_RUNG
   // the same network as SCL:
   "DB2121_MPP".OUTPUTS.O_HS4 := ("DB442_HOPPERS_ALARM_DECODING".GLOBAL_ALARMS_MACHINE.ALARM OR "DB441_POWDER_FEEDERS_ALARM_DECODING".GLOBAL_ALARMS_MACHINE.ALARM) AND "M_1_SEC_1HZ";
   "DB2121_MPP".OUTPUTS.O_HF21 := "DB2121_MPP".OUTPUTS.O_HS4;
END_REGION

REGION Network 4: LAMP - CONTROL OFF
   RUNG wire#powerrail
      I_Contact( "DB2120_MPP_ITC_IPC".MACHINE_ON_DELAYED )
      I_Contact( "DB2120_MPP_ITC_IPC".MACH_ON_DEL_PNEU_ON )
      Coil( "DB2121_MPP".OUTPUTS.O_HS7 )
   END_RUNG
   // the same network as SCL:
   "DB2121_MPP".OUTPUTS.O_HS7 := NOT "DB2120_MPP_ITC_IPC".MACHINE_ON_DELAYED AND NOT "DB2120_MPP_ITC_IPC".MACH_ON_DEL_PNEU_ON;
END_REGION

REGION Network 5: LAMP - IMMEDIATE STOP
   RUNG wire#powerrail
      Contact( "DB2120_MPP_ITC_IPC".IMMEDIATE_STOP_BY_OPERATOR_AUX )
      Coil( "DB2121_MPP".OUTPUTS.O_HS9 )
   END_RUNG
   // the same network as SCL:
   "DB2121_MPP".OUTPUTS.O_HS9 := "DB2120_MPP_ITC_IPC".IMMEDIATE_STOP_BY_OPERATOR_AUX;
END_REGION

REGION Network 6: EMERGENCY STOP ACTIVE
   RUNG wire#powerrail
      Contact( "DB2121_MPP".INPUT_PANEL_EMERGENCY_STOP )
      wire#w1
      Coil( "DB2121_MPP".EMERGENCY_STOP_ACTIVE )
   END_RUNG
   RUNG wire#powerrail
      Contact( "DB2121_MPP".EMERGENCY_STOP_ACTIVE )
      I_Contact( "DB2120_MPP_ITC_IPC".RESET_FAULTS )
   END_RUNG wire#w1
   RUNG wire#w1
      Coil( "DB426_ALARMS_WARNINGS".GENERAL."702800" )
   END_RUNG
   // the same network as SCL:
   "DB2121_MPP".EMERGENCY_STOP_ACTIVE := "DB2121_MPP".INPUT_PANEL_EMERGENCY_STOP OR ("DB2121_MPP".EMERGENCY_STOP_ACTIVE AND NOT "DB2120_MPP_ITC_IPC".RESET_FAULTS);
   "DB426_ALARMS_WARNINGS".GENERAL."702800" := "DB2121_MPP".EMERGENCY_STOP_ACTIVE;
END_REGION

REGION Network 7: IMMEDIATE STOP ALARMS
   RUNG wire#powerrail
      I_Contact( "DB2121_MPP".EMERGENCY_STOP_ACTIVE )
      Not()
      wire#w1
      { S7_GenerateENO := "TRUE" } Move(in := #FC_NUMBER, out1 => "DB442_HOPPERS_ALARM_DECODING".GLOBAL_ALARMS_MACHINE.ALARM_DECODING)
      S_Coil( "DB442_HOPPERS_ALARM_DECODING".ALARMS_CENTRAL.IS_ALARMS )
   END_RUNG
   RUNG wire#w1
      { S7_GenerateENO := "TRUE" } Move(in := #FC_NUMBER, out1 => "DB441_POWDER_FEEDERS_ALARM_DECODING".GLOBAL_ALARMS_MACHINE.ALARM_DECODING)
      S_Coil( "DB441_POWDER_FEEDERS_ALARM_DECODING".ALARMS_CENTRAL.IS_ALARMS )
   END_RUNG
   // the same network as SCL:
   // ENO of a box is taken as its EN; it also drops when the box reports an error
   IF NOT (NOT "DB2121_MPP".EMERGENCY_STOP_ACTIVE) THEN
       "DB442_HOPPERS_ALARM_DECODING".GLOBAL_ALARMS_MACHINE.ALARM_DECODING := #FC_NUMBER;
       "DB442_HOPPERS_ALARM_DECODING".ALARMS_CENTRAL.IS_ALARMS := TRUE;
       "DB441_POWDER_FEEDERS_ALARM_DECODING".GLOBAL_ALARMS_MACHINE.ALARM_DECODING := #FC_NUMBER;
       "DB441_POWDER_FEEDERS_ALARM_DECODING".ALARMS_CENTRAL.IS_ALARMS := TRUE;
   END_IF;
END_REGION

REGION Network 8: WARNING
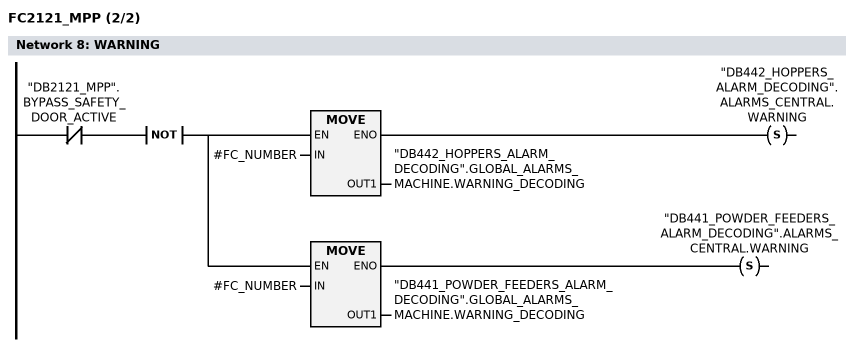
   RUNG wire#powerrail
      I_Contact( "DB2121_MPP".BYPASS_SAFETY_DOOR_ACTIVE )
      Not()
      wire#w1
      { S7_GenerateENO := "TRUE" } Move(in := #FC_NUMBER, out1 => "DB442_HOPPERS_ALARM_DECODING".GLOBAL_ALARMS_MACHINE.WARNING_DECODING)
      S_Coil( "DB442_HOPPERS_ALARM_DECODING".ALARMS_CENTRAL.WARNING )
   END_RUNG
   RUNG wire#w1
      { S7_GenerateENO := "TRUE" } Move(in := #FC_NUMBER, out1 => "DB441_POWDER_FEEDERS_ALARM_DECODING".GLOBAL_ALARMS_MACHINE.WARNING_DECODING)
      S_Coil( "DB441_POWDER_FEEDERS_ALARM_DECODING".ALARMS_CENTRAL.WARNING )
   END_RUNG
   // the same network as SCL:
   // ENO of a box is taken as its EN; it also drops when the box reports an error
   IF NOT (NOT "DB2121_MPP".BYPASS_SAFETY_DOOR_ACTIVE) THEN
       "DB442_HOPPERS_ALARM_DECODING".GLOBAL_ALARMS_MACHINE.WARNING_DECODING := #FC_NUMBER;
       "DB442_HOPPERS_ALARM_DECODING".ALARMS_CENTRAL.WARNING := TRUE;
       "DB441_POWDER_FEEDERS_ALARM_DECODING".GLOBAL_ALARMS_MACHINE.WARNING_DECODING := #FC_NUMBER;
       "DB441_POWDER_FEEDERS_ALARM_DECODING".ALARMS_CENTRAL.WARNING := TRUE;
   END_IF;
END_REGION
END_FUNCTION

FUNCTION "FC2109_HOPPERS_CONTROL_ON" : Void   // FC2109, LAD
{ S7_Optimized_Access := 'FALSE' }
AUTHOR : ETXETAR
VERSION : 1.0
// stored: AutoNumber false, IsIECCheckEnabled false, SetENOAutomatically false, UDAEnableTagReadback false
   VAR_TEMP
      O_BYTE_0 : Struct   // OPTIONS BYTE 0
         GM_COOLANT_PUMP_OFF_DELAY : Bool;   // GM COOLANT PUMP POWER OFF DELAY OPTION
      END_STRUCT;
   END_VAR
   VAR CONSTANT
      FC_NUMBER : DInt := 2109;   // FC NUMBER
   END_VAR
   VAR_TEMP   // added for the SCL form of the ladder/FBD networks
      _w1 : Bool;
   END_VAR
BEGIN

REGION Network 1: INPUTS
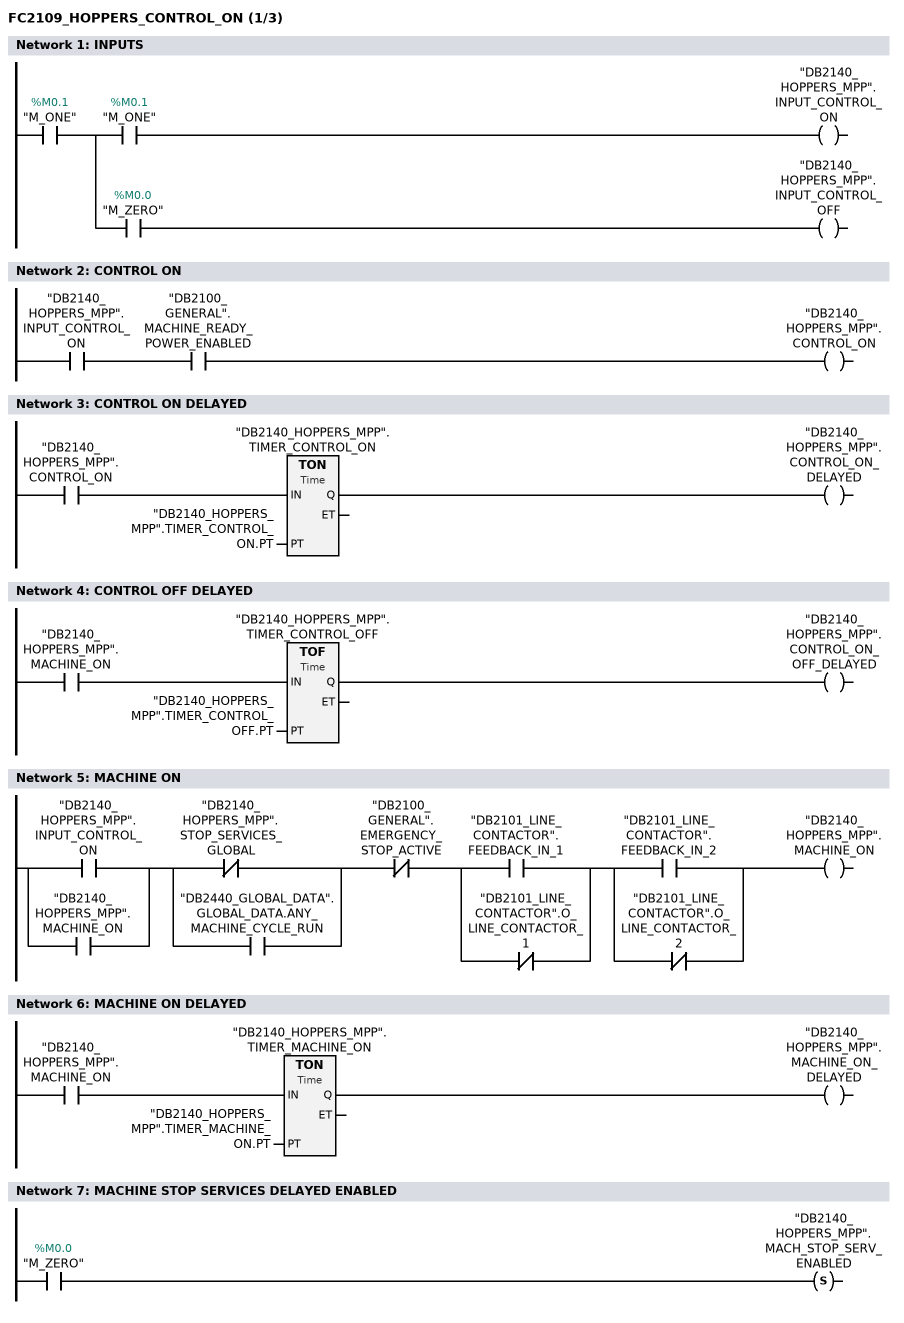
   RUNG wire#powerrail
      Contact( "M_ONE" )
      wire#w1
      Contact( "M_ONE" )
      Coil( "DB2140_HOPPERS_MPP".INPUT_CONTROL_ON )
   END_RUNG
   RUNG wire#w1
      Contact( "M_ZERO" )
      Coil( "DB2140_HOPPERS_MPP".INPUT_CONTROL_OFF )
   END_RUNG
   // the same network as SCL:
   "DB2140_HOPPERS_MPP".INPUT_CONTROL_ON := "M_ONE" AND "M_ONE";
   "DB2140_HOPPERS_MPP".INPUT_CONTROL_OFF := "M_ONE" AND "M_ZERO";
END_REGION

REGION Network 2: CONTROL ON
   RUNG wire#powerrail
      Contact( "DB2140_HOPPERS_MPP".INPUT_CONTROL_ON )
      Contact( "DB2100_GENERAL".MACHINE_READY_POWER_ENABLED )
      Coil( "DB2140_HOPPERS_MPP".CONTROL_ON )
   END_RUNG
   // the same network as SCL:
   "DB2140_HOPPERS_MPP".CONTROL_ON := "DB2140_HOPPERS_MPP".INPUT_CONTROL_ON AND "DB2100_GENERAL".MACHINE_READY_POWER_ENABLED;
END_REGION

REGION Network 3: CONTROL ON DELAYED
   RUNG wire#powerrail
      Contact( "DB2140_HOPPERS_MPP".CONTROL_ON )
      { S7_Templates := "time_type := Time" } "DB2140_HOPPERS_MPP".TIMER_CONTROL_ON.TON(pt := "DB2140_HOPPERS_MPP".TIMER_CONTROL_ON.PT, et =>)
      Coil( "DB2140_HOPPERS_MPP".CONTROL_ON_DELAYED )
   END_RUNG
   // the same network as SCL:
   "DB2140_HOPPERS_MPP".TIMER_CONTROL_ON.TON(IN := "DB2140_HOPPERS_MPP".CONTROL_ON,
                           PT := "DB2140_HOPPERS_MPP".TIMER_CONTROL_ON.PT);
   "DB2140_HOPPERS_MPP".CONTROL_ON_DELAYED := "DB2140_HOPPERS_MPP".TIMER_CONTROL_ON.Q;
END_REGION

REGION Network 4: CONTROL OFF DELAYED
   RUNG wire#powerrail
      Contact( "DB2140_HOPPERS_MPP".MACHINE_ON )
      { S7_Templates := "time_type := Time" } "DB2140_HOPPERS_MPP".TIMER_CONTROL_OFF.TOF(pt := "DB2140_HOPPERS_MPP".TIMER_CONTROL_OFF.PT, et =>)
      Coil( "DB2140_HOPPERS_MPP".CONTROL_ON_OFF_DELAYED )
   END_RUNG
   // the same network as SCL:
   "DB2140_HOPPERS_MPP".TIMER_CONTROL_OFF.TOF(IN := "DB2140_HOPPERS_MPP".MACHINE_ON,
                           PT := "DB2140_HOPPERS_MPP".TIMER_CONTROL_OFF.PT);
   "DB2140_HOPPERS_MPP".CONTROL_ON_OFF_DELAYED := "DB2140_HOPPERS_MPP".TIMER_CONTROL_OFF.Q;
END_REGION

REGION Network 5: MACHINE ON
   RUNG wire#powerrail
      Contact( "DB2140_HOPPERS_MPP".INPUT_CONTROL_ON )
      wire#w1
      I_Contact( "DB2140_HOPPERS_MPP".STOP_SERVICES_GLOBAL )
      wire#w2
      I_Contact( "DB2100_GENERAL".EMERGENCY_STOP_ACTIVE )
      wire#w3
      Contact( "DB2101_LINE_CONTACTOR".FEEDBACK_IN_1 )
      wire#w4
      Contact( "DB2101_LINE_CONTACTOR".FEEDBACK_IN_2 )
      wire#w5
      Coil( "DB2140_HOPPERS_MPP".MACHINE_ON )
   END_RUNG
   RUNG wire#powerrail
      Contact( "DB2140_HOPPERS_MPP".MACHINE_ON )
   END_RUNG wire#w1
   RUNG wire#w1
      Contact( "DB2440_GLOBAL_DATA".GLOBAL_DATA.ANY_MACHINE_CYCLE_RUN )
   END_RUNG wire#w2
   RUNG wire#w3
      I_Contact( "DB2101_LINE_CONTACTOR".O_LINE_CONTACTOR_1 )
   END_RUNG wire#w4
   RUNG wire#w4
      I_Contact( "DB2101_LINE_CONTACTOR".O_LINE_CONTACTOR_2 )
   END_RUNG wire#w5
   // the same network as SCL:
   "DB2140_HOPPERS_MPP".MACHINE_ON := ("DB2140_HOPPERS_MPP".INPUT_CONTROL_ON OR "DB2140_HOPPERS_MPP".MACHINE_ON) AND (NOT "DB2140_HOPPERS_MPP".STOP_SERVICES_GLOBAL OR "DB2440_GLOBAL_DATA".GLOBAL_DATA.ANY_MACHINE_CYCLE_RUN) AND NOT "DB2100_GENERAL".EMERGENCY_STOP_ACTIVE AND ("DB2101_LINE_CONTACTOR".FEEDBACK_IN_1 OR NOT "DB2101_LINE_CONTACTOR".O_LINE_CONTACTOR_1) AND ("DB2101_LINE_CONTACTOR".FEEDBACK_IN_2 OR NOT "DB2101_LINE_CONTACTOR".O_LINE_CONTACTOR_2);
END_REGION

REGION Network 6: MACHINE ON DELAYED
   RUNG wire#powerrail
      Contact( "DB2140_HOPPERS_MPP".MACHINE_ON )
      { S7_Templates := "time_type := Time" } "DB2140_HOPPERS_MPP".TIMER_MACHINE_ON.TON(pt := "DB2140_HOPPERS_MPP".TIMER_MACHINE_ON.PT, et =>)
      Coil( "DB2140_HOPPERS_MPP".MACHINE_ON_DELAYED )
   END_RUNG
   // the same network as SCL:
   "DB2140_HOPPERS_MPP".TIMER_MACHINE_ON.TON(IN := "DB2140_HOPPERS_MPP".MACHINE_ON,
                           PT := "DB2140_HOPPERS_MPP".TIMER_MACHINE_ON.PT);
   "DB2140_HOPPERS_MPP".MACHINE_ON_DELAYED := "DB2140_HOPPERS_MPP".TIMER_MACHINE_ON.Q;
END_REGION

REGION Network 7: MACHINE STOP SERVICES DELAYED ENABLED
   RUNG wire#powerrail
      Contact( "M_ZERO" )
      S_Coil( "DB2140_HOPPERS_MPP".MACH_STOP_SERV_ENABLED )
   END_RUNG
   // the same network as SCL:
   IF "M_ZERO" THEN "DB2140_HOPPERS_MPP".MACH_STOP_SERV_ENABLED := TRUE; END_IF;
END_REGION

REGION Network 8: MACHINE STOP SERVICES DELAYED ENABLED
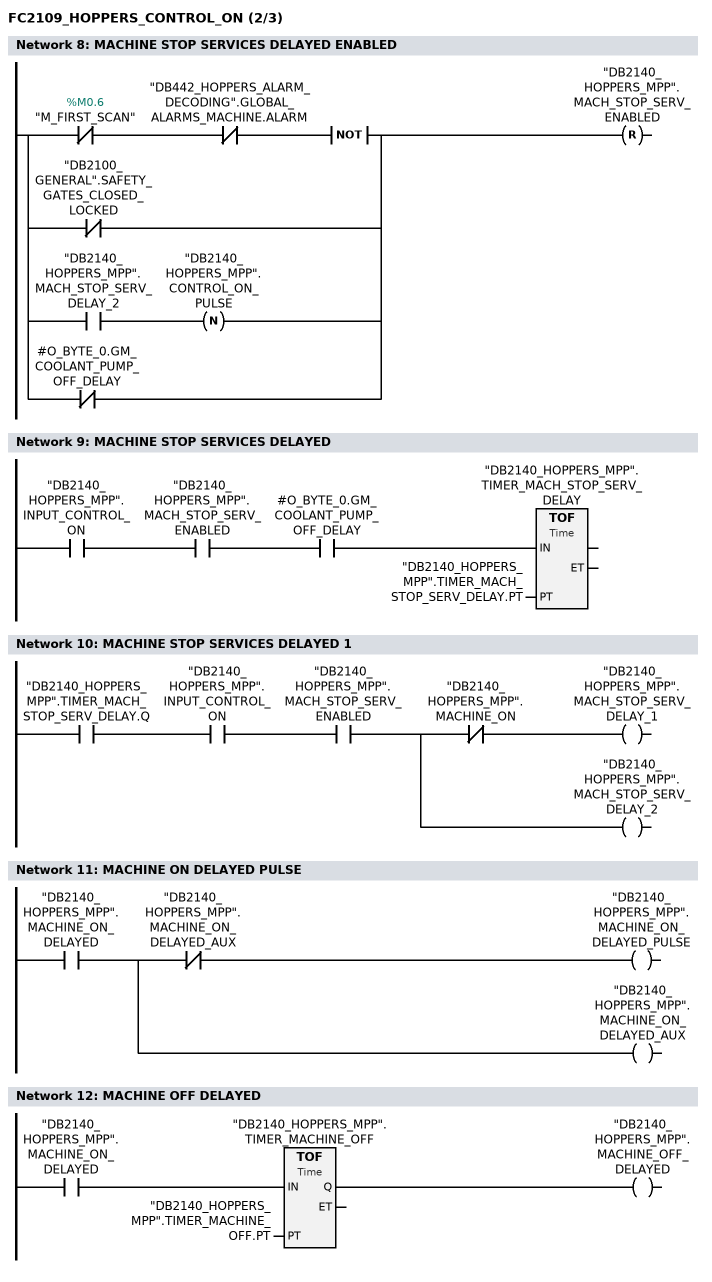
   RUNG wire#powerrail
      I_Contact( "M_FIRST_SCAN" )
      I_Contact( "DB442_HOPPERS_ALARM_DECODING".GLOBAL_ALARMS_MACHINE.ALARM )
      Not()
      wire#w1
      R_Coil( "DB2140_HOPPERS_MPP".MACH_STOP_SERV_ENABLED )
   END_RUNG
   RUNG wire#powerrail
      I_Contact( "DB2100_GENERAL".SAFETY_GATES_CLOSED_LOCKED )
   END_RUNG wire#w1
   RUNG wire#powerrail
      Contact( "DB2140_HOPPERS_MPP".MACH_STOP_SERV_DELAY_2 )
      N_Trig( "DB2140_HOPPERS_MPP".CONTROL_ON_PULSE )
   END_RUNG wire#w1
   RUNG wire#powerrail
      I_Contact( #O_BYTE_0.GM_COOLANT_PUMP_OFF_DELAY )
   END_RUNG wire#w1
   // the same network as SCL:
   #_w1 := NOT "DB2140_HOPPERS_MPP".MACH_STOP_SERV_DELAY_2 AND "DB2140_HOPPERS_MPP".CONTROL_ON_PULSE;   // falling edge
   "DB2140_HOPPERS_MPP".CONTROL_ON_PULSE := "DB2140_HOPPERS_MPP".MACH_STOP_SERV_DELAY_2;
   IF NOT (NOT "M_FIRST_SCAN" AND NOT "DB442_HOPPERS_ALARM_DECODING".GLOBAL_ALARMS_MACHINE.ALARM) OR NOT "DB2100_GENERAL".SAFETY_GATES_CLOSED_LOCKED OR #_w1 OR NOT #O_BYTE_0.GM_COOLANT_PUMP_OFF_DELAY THEN
       "DB2140_HOPPERS_MPP".MACH_STOP_SERV_ENABLED := FALSE;
   END_IF;
END_REGION

REGION Network 9: MACHINE STOP SERVICES DELAYED
   RUNG wire#powerrail
      Contact( "DB2140_HOPPERS_MPP".INPUT_CONTROL_ON )
      Contact( "DB2140_HOPPERS_MPP".MACH_STOP_SERV_ENABLED )
      Contact( #O_BYTE_0.GM_COOLANT_PUMP_OFF_DELAY )
      { S7_Templates := "time_type := Time" } "DB2140_HOPPERS_MPP".TIMER_MACH_STOP_SERV_DELAY.TOF(pt := "DB2140_HOPPERS_MPP".TIMER_MACH_STOP_SERV_DELAY.PT, et =>)
   END_RUNG
   // the same network as SCL:
   "DB2140_HOPPERS_MPP".TIMER_MACH_STOP_SERV_DELAY.TOF(IN := "DB2140_HOPPERS_MPP".INPUT_CONTROL_ON AND "DB2140_HOPPERS_MPP".MACH_STOP_SERV_ENABLED AND #O_BYTE_0.GM_COOLANT_PUMP_OFF_DELAY,
                           PT := "DB2140_HOPPERS_MPP".TIMER_MACH_STOP_SERV_DELAY.PT);
END_REGION

REGION Network 10: MACHINE STOP SERVICES DELAYED 1
   RUNG wire#powerrail
      Contact( "DB2140_HOPPERS_MPP".TIMER_MACH_STOP_SERV_DELAY.Q )
      Contact( "DB2140_HOPPERS_MPP".INPUT_CONTROL_ON )
      Contact( "DB2140_HOPPERS_MPP".MACH_STOP_SERV_ENABLED )
      wire#w1
      I_Contact( "DB2140_HOPPERS_MPP".MACHINE_ON )
      Coil( "DB2140_HOPPERS_MPP".MACH_STOP_SERV_DELAY_1 )
   END_RUNG
   RUNG wire#w1
      Coil( "DB2140_HOPPERS_MPP".MACH_STOP_SERV_DELAY_2 )
   END_RUNG
   // the same network as SCL:
   #_w1 := "DB2140_HOPPERS_MPP".TIMER_MACH_STOP_SERV_DELAY.Q AND "DB2140_HOPPERS_MPP".INPUT_CONTROL_ON AND "DB2140_HOPPERS_MPP".MACH_STOP_SERV_ENABLED;
   "DB2140_HOPPERS_MPP".MACH_STOP_SERV_DELAY_1 := #_w1 AND NOT "DB2140_HOPPERS_MPP".MACHINE_ON;
   "DB2140_HOPPERS_MPP".MACH_STOP_SERV_DELAY_2 := #_w1;
END_REGION

REGION Network 11: MACHINE ON DELAYED PULSE
   RUNG wire#powerrail
      Contact( "DB2140_HOPPERS_MPP".MACHINE_ON_DELAYED )
      wire#w1
      I_Contact( "DB2140_HOPPERS_MPP".MACHINE_ON_DELAYED_AUX )
      Coil( "DB2140_HOPPERS_MPP".MACHINE_ON_DELAYED_PULSE )
   END_RUNG
   RUNG wire#w1
      Coil( "DB2140_HOPPERS_MPP".MACHINE_ON_DELAYED_AUX )
   END_RUNG
   // the same network as SCL:
   "DB2140_HOPPERS_MPP".MACHINE_ON_DELAYED_PULSE := "DB2140_HOPPERS_MPP".MACHINE_ON_DELAYED AND NOT "DB2140_HOPPERS_MPP".MACHINE_ON_DELAYED_AUX;
   "DB2140_HOPPERS_MPP".MACHINE_ON_DELAYED_AUX := "DB2140_HOPPERS_MPP".MACHINE_ON_DELAYED;
END_REGION

REGION Network 12: MACHINE OFF DELAYED
   RUNG wire#powerrail
      Contact( "DB2140_HOPPERS_MPP".MACHINE_ON_DELAYED )
      { S7_Templates := "time_type := Time" } "DB2140_HOPPERS_MPP".TIMER_MACHINE_OFF.TOF(pt := "DB2140_HOPPERS_MPP".TIMER_MACHINE_OFF.PT, et =>)
      Coil( "DB2140_HOPPERS_MPP".MACHINE_OFF_DELAYED )
   END_RUNG
   // the same network as SCL:
   "DB2140_HOPPERS_MPP".TIMER_MACHINE_OFF.TOF(IN := "DB2140_HOPPERS_MPP".MACHINE_ON_DELAYED,
                           PT := "DB2140_HOPPERS_MPP".TIMER_MACHINE_OFF.PT);
   "DB2140_HOPPERS_MPP".MACHINE_OFF_DELAYED := "DB2140_HOPPERS_MPP".TIMER_MACHINE_OFF.Q;
END_REGION

REGION Network 13: MACHINE ON DELAYED AND HYDRAULIC AND PNEUMATIC IN SERVICE
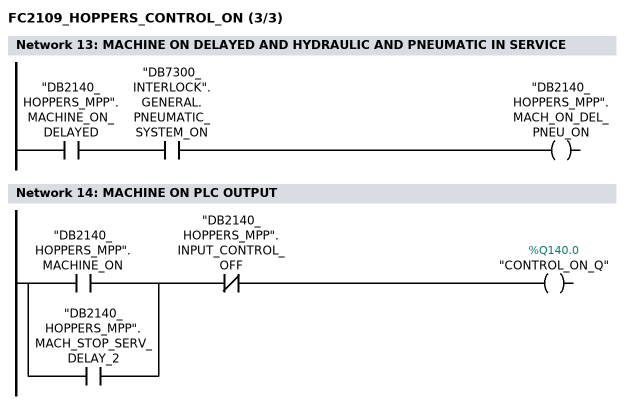
   RUNG wire#powerrail
      Contact( "DB2140_HOPPERS_MPP".MACHINE_ON_DELAYED )
      Contact( "DB7300_INTERLOCK".GENERAL.PNEUMATIC_SYSTEM_ON )
      Coil( "DB2140_HOPPERS_MPP".MACH_ON_DEL_PNEU_ON )
   END_RUNG
   // the same network as SCL:
   "DB2140_HOPPERS_MPP".MACH_ON_DEL_PNEU_ON := "DB2140_HOPPERS_MPP".MACHINE_ON_DELAYED AND "DB7300_INTERLOCK".GENERAL.PNEUMATIC_SYSTEM_ON;
END_REGION

REGION Network 14: MACHINE ON PLC OUTPUT
   RUNG wire#powerrail
      Contact( "DB2140_HOPPERS_MPP".MACHINE_ON )
      wire#w1
      I_Contact( "DB2140_HOPPERS_MPP".INPUT_CONTROL_OFF )
      Coil( "CONTROL_ON_Q" )
   END_RUNG
   RUNG wire#powerrail
      Contact( "DB2140_HOPPERS_MPP".MACH_STOP_SERV_DELAY_2 )
   END_RUNG wire#w1
   // the same network as SCL:
   "CONTROL_ON_Q" := ("DB2140_HOPPERS_MPP".MACHINE_ON OR "DB2140_HOPPERS_MPP".MACH_STOP_SERV_DELAY_2) AND NOT "DB2140_HOPPERS_MPP".INPUT_CONTROL_OFF;
END_REGION
END_FUNCTION

FUNCTION "FC2140_HOPPERS_BUTTONS" : Void   // FC2140, LAD
{ S7_Optimized_Access := 'FALSE' }
AUTHOR : ETXETAR
VERSION : 1.0
// stored: AutoNumber false, IsIECCheckEnabled false, SetENOAutomatically false, UDAEnableTagReadback false
   VAR_TEMP
      O_BYTE_0 : Struct   // OPTIONS BYTE 0
         IPC : Bool;   // IPC OPTION
      END_STRUCT;
      TCU_INDEX_SEL : Int;
   END_VAR
   VAR CONSTANT
      FC_NUMBER : DInt := 2140;   // FC NUMBER
   END_VAR
   VAR_TEMP   // added for the SCL form of the ladder/FBD networks
      _w1 : Bool;
   END_VAR
BEGIN

REGION Network 1: OPTIONS
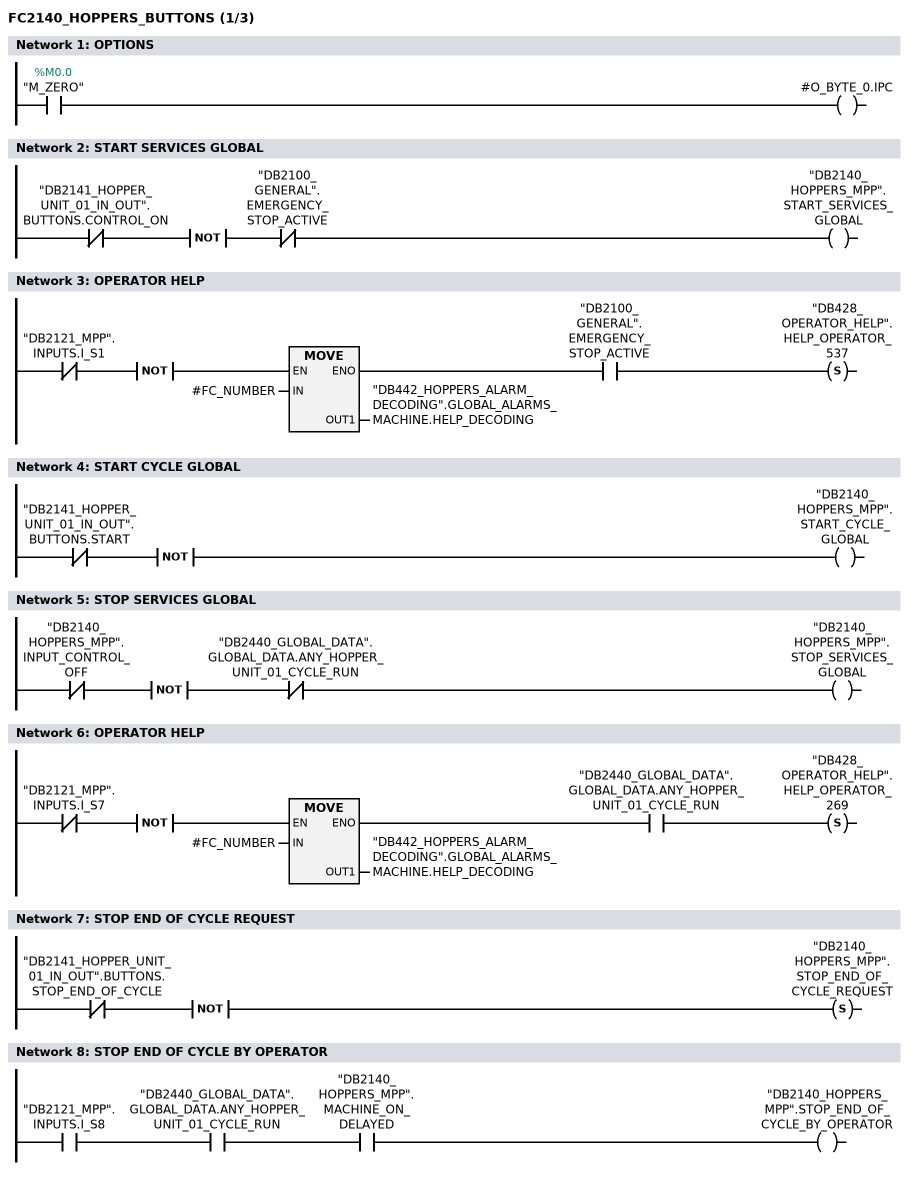
   RUNG wire#powerrail
      Contact( "M_ZERO" )
      Coil( #O_BYTE_0.IPC )
   END_RUNG
   // the same network as SCL:
   #O_BYTE_0.IPC := "M_ZERO";
END_REGION

REGION Network 2: START SERVICES GLOBAL
   RUNG wire#powerrail
      I_Contact( "DB2141_HOPPER_UNIT_01_IN_OUT".BUTTONS.CONTROL_ON )
      Not()
      I_Contact( "DB2100_GENERAL".EMERGENCY_STOP_ACTIVE )
      Coil( "DB2140_HOPPERS_MPP".START_SERVICES_GLOBAL )
   END_RUNG
   // the same network as SCL:
   "DB2140_HOPPERS_MPP".START_SERVICES_GLOBAL := NOT (NOT "DB2141_HOPPER_UNIT_01_IN_OUT".BUTTONS.CONTROL_ON) AND NOT "DB2100_GENERAL".EMERGENCY_STOP_ACTIVE;
END_REGION

REGION Network 3: OPERATOR HELP
   RUNG wire#powerrail
      I_Contact( "DB2121_MPP".INPUTS.I_S1 )
      Not()
      { S7_GenerateENO := "TRUE" } Move(in := #FC_NUMBER, out1 => "DB442_HOPPERS_ALARM_DECODING".GLOBAL_ALARMS_MACHINE.HELP_DECODING)
      Contact( "DB2100_GENERAL".EMERGENCY_STOP_ACTIVE )
      S_Coil( "DB428_OPERATOR_HELP".HELP_OPERATOR_537 )
   END_RUNG
   // the same network as SCL:
   // ENO of a box is taken as its EN; it also drops when the box reports an error
   #_w1 := NOT (NOT "DB2121_MPP".INPUTS.I_S1);
   IF #_w1 THEN "DB442_HOPPERS_ALARM_DECODING".GLOBAL_ALARMS_MACHINE.HELP_DECODING := #FC_NUMBER; END_IF;
   IF #_w1 AND "DB2100_GENERAL".EMERGENCY_STOP_ACTIVE THEN
       "DB428_OPERATOR_HELP".HELP_OPERATOR_537 := TRUE;
   END_IF;
END_REGION

REGION Network 4: START CYCLE GLOBAL
   RUNG wire#powerrail
      I_Contact( "DB2141_HOPPER_UNIT_01_IN_OUT".BUTTONS.START )
      Not()
      Coil( "DB2140_HOPPERS_MPP".START_CYCLE_GLOBAL )
   END_RUNG
   // the same network as SCL:
   "DB2140_HOPPERS_MPP".START_CYCLE_GLOBAL := NOT (NOT "DB2141_HOPPER_UNIT_01_IN_OUT".BUTTONS.START);
END_REGION

REGION Network 5: STOP SERVICES GLOBAL
   RUNG wire#powerrail
      I_Contact( "DB2140_HOPPERS_MPP".INPUT_CONTROL_OFF )
      Not()
      I_Contact( "DB2440_GLOBAL_DATA".GLOBAL_DATA.ANY_HOPPER_UNIT_01_CYCLE_RUN )
      Coil( "DB2140_HOPPERS_MPP".STOP_SERVICES_GLOBAL )
   END_RUNG
   // the same network as SCL:
   "DB2140_HOPPERS_MPP".STOP_SERVICES_GLOBAL := NOT (NOT "DB2140_HOPPERS_MPP".INPUT_CONTROL_OFF) AND NOT "DB2440_GLOBAL_DATA".GLOBAL_DATA.ANY_HOPPER_UNIT_01_CYCLE_RUN;
END_REGION

REGION Network 6: OPERATOR HELP
   RUNG wire#powerrail
      I_Contact( "DB2121_MPP".INPUTS.I_S7 )
      Not()
      { S7_GenerateENO := "TRUE" } Move(in := #FC_NUMBER, out1 => "DB442_HOPPERS_ALARM_DECODING".GLOBAL_ALARMS_MACHINE.HELP_DECODING)
      Contact( "DB2440_GLOBAL_DATA".GLOBAL_DATA.ANY_HOPPER_UNIT_01_CYCLE_RUN )
      S_Coil( "DB428_OPERATOR_HELP".HELP_OPERATOR_269 )
   END_RUNG
   // the same network as SCL:
   // ENO of a box is taken as its EN; it also drops when the box reports an error
   #_w1 := NOT (NOT "DB2121_MPP".INPUTS.I_S7);
   IF #_w1 THEN "DB442_HOPPERS_ALARM_DECODING".GLOBAL_ALARMS_MACHINE.HELP_DECODING := #FC_NUMBER; END_IF;
   IF #_w1 AND "DB2440_GLOBAL_DATA".GLOBAL_DATA.ANY_HOPPER_UNIT_01_CYCLE_RUN THEN
       "DB428_OPERATOR_HELP".HELP_OPERATOR_269 := TRUE;
   END_IF;
END_REGION

REGION Network 7: STOP END OF CYCLE REQUEST
   RUNG wire#powerrail
      I_Contact( "DB2141_HOPPER_UNIT_01_IN_OUT".BUTTONS.STOP_END_OF_CYCLE )
      Not()
      S_Coil( "DB2140_HOPPERS_MPP".STOP_END_OF_CYCLE_REQUEST )
   END_RUNG
   // the same network as SCL:
   IF NOT (NOT "DB2141_HOPPER_UNIT_01_IN_OUT".BUTTONS.STOP_END_OF_CYCLE) THEN
       "DB2140_HOPPERS_MPP".STOP_END_OF_CYCLE_REQUEST := TRUE;
   END_IF;
END_REGION

REGION Network 8: STOP END OF CYCLE BY OPERATOR
   RUNG wire#powerrail
      Contact( "DB2121_MPP".INPUTS.I_S8 )
      Contact( "DB2440_GLOBAL_DATA".GLOBAL_DATA.ANY_HOPPER_UNIT_01_CYCLE_RUN )
      Contact( "DB2140_HOPPERS_MPP".MACHINE_ON_DELAYED )
      Coil( "DB2140_HOPPERS_MPP".STOP_END_OF_CYCLE_BY_OPERATOR )
   END_RUNG
   // the same network as SCL:
   "DB2140_HOPPERS_MPP".STOP_END_OF_CYCLE_BY_OPERATOR := "DB2121_MPP".INPUTS.I_S8 AND "DB2440_GLOBAL_DATA".GLOBAL_DATA.ANY_HOPPER_UNIT_01_CYCLE_RUN AND "DB2140_HOPPERS_MPP".MACHINE_ON_DELAYED;
END_REGION

REGION Network 9: MAIN PANEL OPERATOR REQUEST STOP AT END OF CYCLE
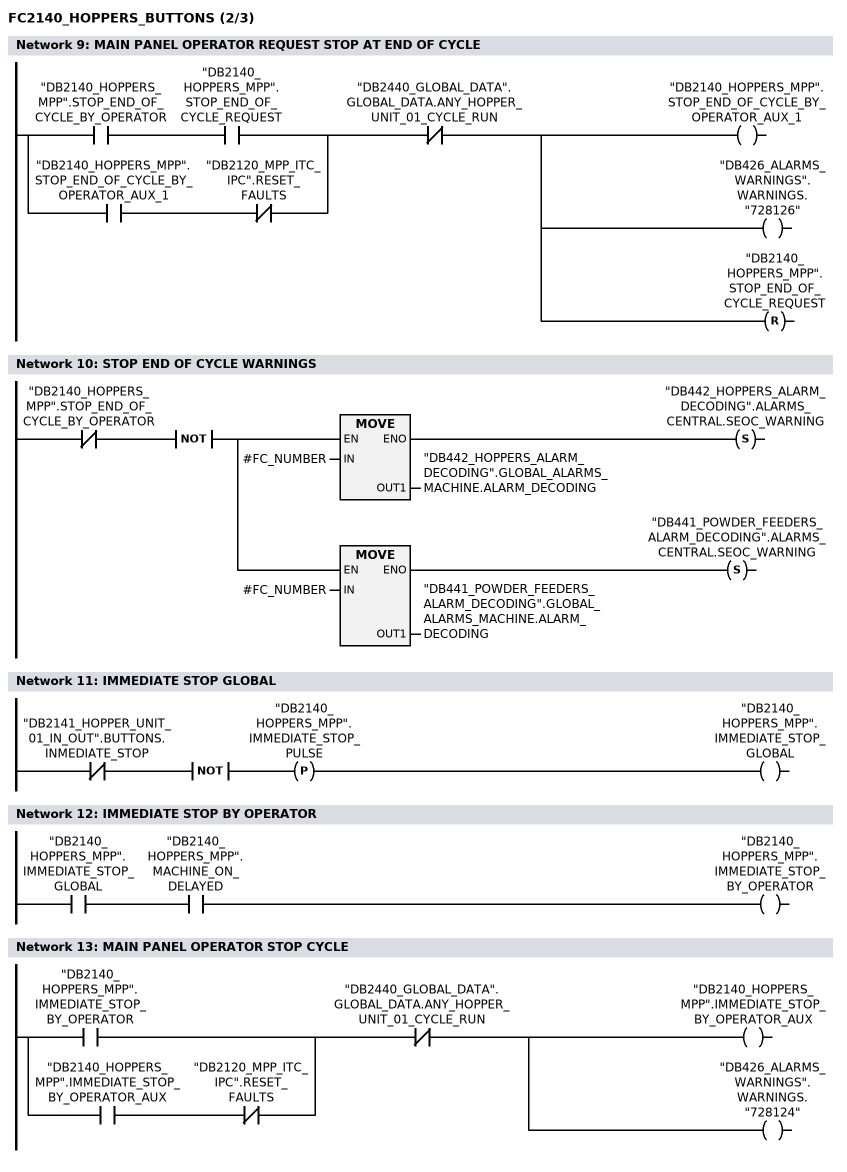
   RUNG wire#powerrail
      Contact( "DB2140_HOPPERS_MPP".STOP_END_OF_CYCLE_BY_OPERATOR )
      Contact( "DB2140_HOPPERS_MPP".STOP_END_OF_CYCLE_REQUEST )
      wire#w1
      I_Contact( "DB2440_GLOBAL_DATA".GLOBAL_DATA.ANY_HOPPER_UNIT_01_CYCLE_RUN )
      wire#w2
      Coil( "DB2140_HOPPERS_MPP".STOP_END_OF_CYCLE_BY_OPERATOR_AUX_1 )
   END_RUNG
   RUNG wire#powerrail
      Contact( "DB2140_HOPPERS_MPP".STOP_END_OF_CYCLE_BY_OPERATOR_AUX_1 )
      I_Contact( "DB2120_MPP_ITC_IPC".RESET_FAULTS )
   END_RUNG wire#w1
   RUNG wire#w2
      Coil( "DB426_ALARMS_WARNINGS".WARNINGS."728126" )
   END_RUNG
   RUNG wire#w2
      R_Coil( "DB2140_HOPPERS_MPP".STOP_END_OF_CYCLE_REQUEST )
   END_RUNG
   // the same network as SCL:
   "DB2140_HOPPERS_MPP".STOP_END_OF_CYCLE_BY_OPERATOR_AUX_1 := (("DB2140_HOPPERS_MPP".STOP_END_OF_CYCLE_BY_OPERATOR AND "DB2140_HOPPERS_MPP".STOP_END_OF_CYCLE_REQUEST) OR ("DB2140_HOPPERS_MPP".STOP_END_OF_CYCLE_BY_OPERATOR_AUX_1 AND NOT "DB2120_MPP_ITC_IPC".RESET_FAULTS)) AND NOT "DB2440_GLOBAL_DATA".GLOBAL_DATA.ANY_HOPPER_UNIT_01_CYCLE_RUN;
   "DB426_ALARMS_WARNINGS".WARNINGS."728126" := "DB2140_HOPPERS_MPP".STOP_END_OF_CYCLE_BY_OPERATOR_AUX_1;
   IF "DB2140_HOPPERS_MPP".STOP_END_OF_CYCLE_BY_OPERATOR_AUX_1 THEN
       "DB2140_HOPPERS_MPP".STOP_END_OF_CYCLE_REQUEST := FALSE;
   END_IF;
END_REGION

REGION Network 10: STOP END OF CYCLE WARNINGS
   RUNG wire#powerrail
      I_Contact( "DB2140_HOPPERS_MPP".STOP_END_OF_CYCLE_BY_OPERATOR )
      Not()
      wire#w1
      { S7_GenerateENO := "TRUE" } Move(in := #FC_NUMBER, out1 => "DB442_HOPPERS_ALARM_DECODING".GLOBAL_ALARMS_MACHINE.ALARM_DECODING)
      S_Coil( "DB442_HOPPERS_ALARM_DECODING".ALARMS_CENTRAL.SEOC_WARNING )
   END_RUNG
   RUNG wire#w1
      { S7_GenerateENO := "TRUE" } Move(in := #FC_NUMBER, out1 => "DB441_POWDER_FEEDERS_ALARM_DECODING".GLOBAL_ALARMS_MACHINE.ALARM_DECODING)
      S_Coil( "DB441_POWDER_FEEDERS_ALARM_DECODING".ALARMS_CENTRAL.SEOC_WARNING )
   END_RUNG
   // the same network as SCL:
   // ENO of a box is taken as its EN; it also drops when the box reports an error
   IF NOT (NOT "DB2140_HOPPERS_MPP".STOP_END_OF_CYCLE_BY_OPERATOR) THEN
       "DB442_HOPPERS_ALARM_DECODING".GLOBAL_ALARMS_MACHINE.ALARM_DECODING := #FC_NUMBER;
       "DB442_HOPPERS_ALARM_DECODING".ALARMS_CENTRAL.SEOC_WARNING := TRUE;
       "DB441_POWDER_FEEDERS_ALARM_DECODING".GLOBAL_ALARMS_MACHINE.ALARM_DECODING := #FC_NUMBER;
       "DB441_POWDER_FEEDERS_ALARM_DECODING".ALARMS_CENTRAL.SEOC_WARNING := TRUE;
   END_IF;
END_REGION

REGION Network 11: IMMEDIATE STOP GLOBAL
   RUNG wire#powerrail
      I_Contact( "DB2141_HOPPER_UNIT_01_IN_OUT".BUTTONS.INMEDIATE_STOP )
      Not()
      P_Trig( "DB2140_HOPPERS_MPP".IMMEDIATE_STOP_PULSE )
      Coil( "DB2140_HOPPERS_MPP".IMMEDIATE_STOP_GLOBAL )
   END_RUNG
   // the same network as SCL:
   #_w1 := NOT (NOT "DB2141_HOPPER_UNIT_01_IN_OUT".BUTTONS.INMEDIATE_STOP) AND NOT "DB2140_HOPPERS_MPP".IMMEDIATE_STOP_PULSE;   // rising edge
   "DB2140_HOPPERS_MPP".IMMEDIATE_STOP_PULSE := NOT (NOT "DB2141_HOPPER_UNIT_01_IN_OUT".BUTTONS.INMEDIATE_STOP);
   "DB2140_HOPPERS_MPP".IMMEDIATE_STOP_GLOBAL := #_w1;
END_REGION

REGION Network 12: IMMEDIATE STOP BY OPERATOR
   RUNG wire#powerrail
      Contact( "DB2140_HOPPERS_MPP".IMMEDIATE_STOP_GLOBAL )
      Contact( "DB2140_HOPPERS_MPP".MACHINE_ON_DELAYED )
      Coil( "DB2140_HOPPERS_MPP".IMMEDIATE_STOP_BY_OPERATOR )
   END_RUNG
   // the same network as SCL:
   "DB2140_HOPPERS_MPP".IMMEDIATE_STOP_BY_OPERATOR := "DB2140_HOPPERS_MPP".IMMEDIATE_STOP_GLOBAL AND "DB2140_HOPPERS_MPP".MACHINE_ON_DELAYED;
END_REGION

REGION Network 13: MAIN PANEL OPERATOR STOP CYCLE
   RUNG wire#powerrail
      Contact( "DB2140_HOPPERS_MPP".IMMEDIATE_STOP_BY_OPERATOR )
      wire#w1
      I_Contact( "DB2440_GLOBAL_DATA".GLOBAL_DATA.ANY_HOPPER_UNIT_01_CYCLE_RUN )
      wire#w2
      Coil( "DB2140_HOPPERS_MPP".IMMEDIATE_STOP_BY_OPERATOR_AUX )
   END_RUNG
   RUNG wire#powerrail
      Contact( "DB2140_HOPPERS_MPP".IMMEDIATE_STOP_BY_OPERATOR_AUX )
      I_Contact( "DB2120_MPP_ITC_IPC".RESET_FAULTS )
   END_RUNG wire#w1
   RUNG wire#w2
      Coil( "DB426_ALARMS_WARNINGS".WARNINGS."728124" )
   END_RUNG
   // the same network as SCL:
   "DB2140_HOPPERS_MPP".IMMEDIATE_STOP_BY_OPERATOR_AUX := ("DB2140_HOPPERS_MPP".IMMEDIATE_STOP_BY_OPERATOR OR ("DB2140_HOPPERS_MPP".IMMEDIATE_STOP_BY_OPERATOR_AUX AND NOT "DB2120_MPP_ITC_IPC".RESET_FAULTS)) AND NOT "DB2440_GLOBAL_DATA".GLOBAL_DATA.ANY_HOPPER_UNIT_01_CYCLE_RUN;
   "DB426_ALARMS_WARNINGS".WARNINGS."728124" := "DB2140_HOPPERS_MPP".IMMEDIATE_STOP_BY_OPERATOR_AUX;
END_REGION

REGION Network 14: IMMEDIATE STOP WARNING
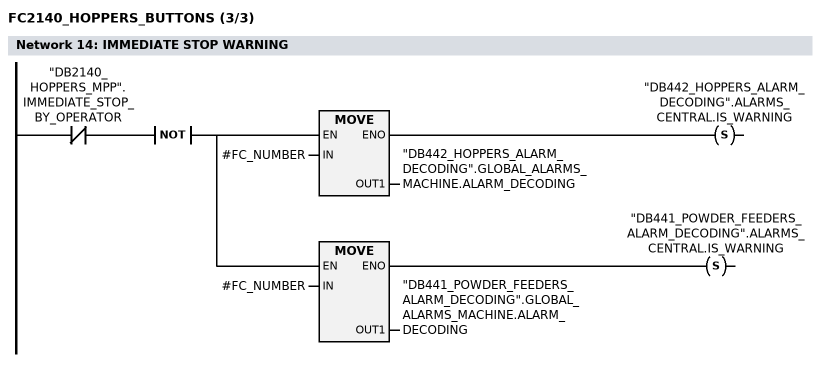
   RUNG wire#powerrail
      I_Contact( "DB2140_HOPPERS_MPP".IMMEDIATE_STOP_BY_OPERATOR )
      Not()
      wire#w1
      { S7_GenerateENO := "TRUE" } Move(in := #FC_NUMBER, out1 => "DB442_HOPPERS_ALARM_DECODING".GLOBAL_ALARMS_MACHINE.ALARM_DECODING)
      S_Coil( "DB442_HOPPERS_ALARM_DECODING".ALARMS_CENTRAL.IS_WARNING )
   END_RUNG
   RUNG wire#w1
      { S7_GenerateENO := "TRUE" } Move(in := #FC_NUMBER, out1 => "DB441_POWDER_FEEDERS_ALARM_DECODING".GLOBAL_ALARMS_MACHINE.ALARM_DECODING)
      S_Coil( "DB441_POWDER_FEEDERS_ALARM_DECODING".ALARMS_CENTRAL.IS_WARNING )
   END_RUNG
   // the same network as SCL:
   // ENO of a box is taken as its EN; it also drops when the box reports an error
   IF NOT (NOT "DB2140_HOPPERS_MPP".IMMEDIATE_STOP_BY_OPERATOR) THEN
       "DB442_HOPPERS_ALARM_DECODING".GLOBAL_ALARMS_MACHINE.ALARM_DECODING := #FC_NUMBER;
       "DB442_HOPPERS_ALARM_DECODING".ALARMS_CENTRAL.IS_WARNING := TRUE;
       "DB441_POWDER_FEEDERS_ALARM_DECODING".GLOBAL_ALARMS_MACHINE.ALARM_DECODING := #FC_NUMBER;
       "DB441_POWDER_FEEDERS_ALARM_DECODING".ALARMS_CENTRAL.IS_WARNING := TRUE;
   END_IF;
END_REGION
END_FUNCTION

FUNCTION "FC2141_HOPPERS_LAMPS" : Void   // FC2141, LAD
{ S7_Optimized_Access := 'FALSE' }
AUTHOR : ETXETAR
VERSION : 1.0
// stored: AutoNumber false, IsIECCheckEnabled false, SetENOAutomatically false, UDAEnableTagReadback false
   VAR_TEMP
      ONE : Int;
      RETVAL1 : Int;
      SIMU_PANEL_HMI_SEL : Bool;   // SIMULATED PANEL IN HMI SELECTED
   END_VAR
   VAR CONSTANT
      FC_NUMBER : DInt := 2141;   // FC NUMBER
   END_VAR
BEGIN

REGION Network 1: LAMP - CONTROL ON
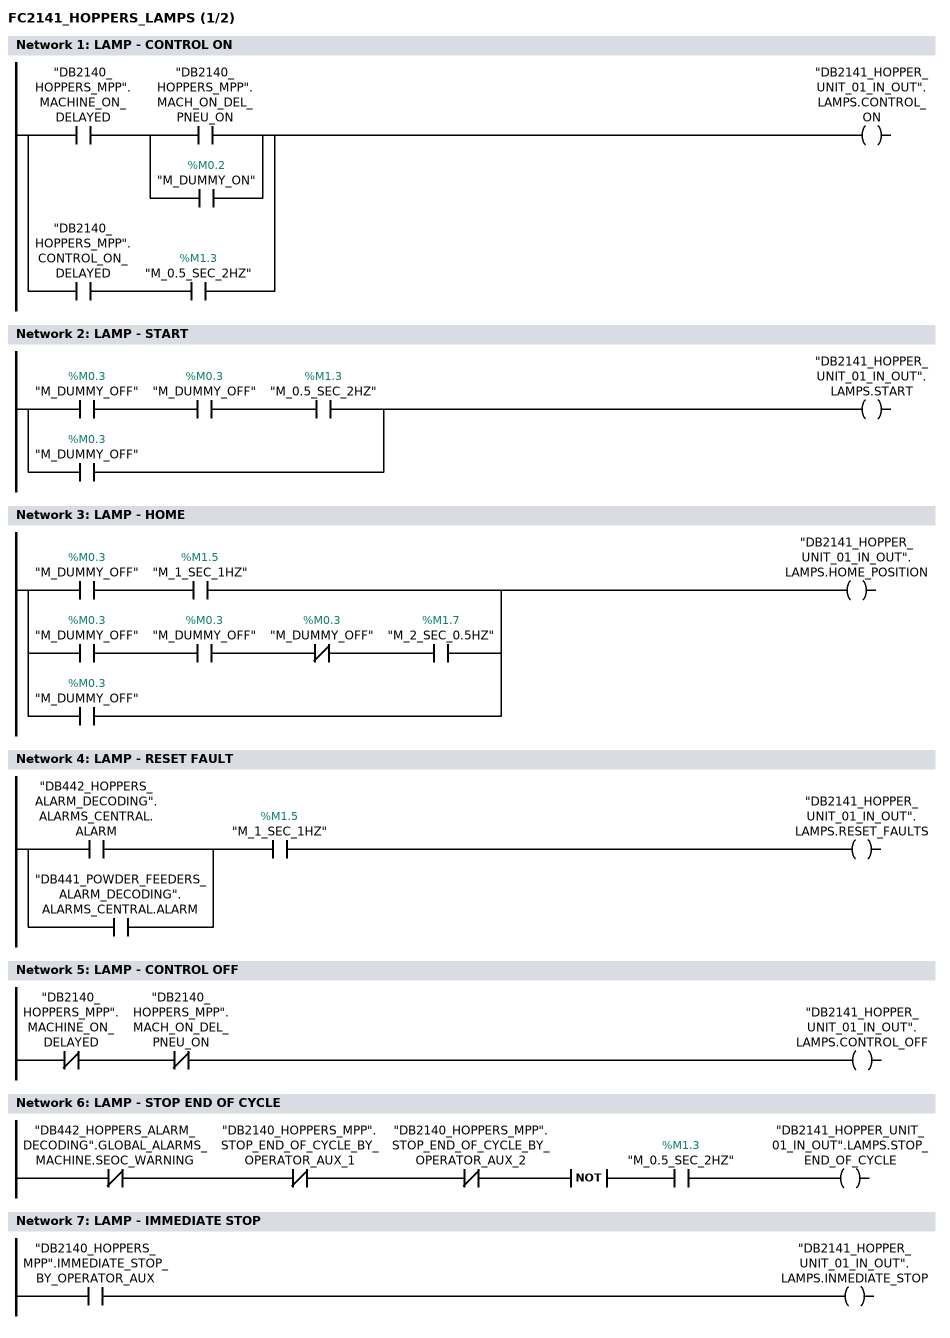
   RUNG wire#powerrail
      Contact( "DB2140_HOPPERS_MPP".MACHINE_ON_DELAYED )
      wire#w1
      Contact( "DB2140_HOPPERS_MPP".MACH_ON_DEL_PNEU_ON )
      wire#w2
      Coil( "DB2141_HOPPER_UNIT_01_IN_OUT".LAMPS.CONTROL_ON )
   END_RUNG
   RUNG wire#w1
      Contact( "M_DUMMY_ON" )
   END_RUNG wire#w2
   RUNG wire#powerrail
      Contact( "DB2140_HOPPERS_MPP".CONTROL_ON_DELAYED )
      Contact( "M_0.5_SEC_2HZ" )
   END_RUNG wire#w2
   // the same network as SCL:
   "DB2141_HOPPER_UNIT_01_IN_OUT".LAMPS.CONTROL_ON := ("DB2140_HOPPERS_MPP".MACHINE_ON_DELAYED AND ("DB2140_HOPPERS_MPP".MACH_ON_DEL_PNEU_ON OR "M_DUMMY_ON")) OR ("DB2140_HOPPERS_MPP".CONTROL_ON_DELAYED AND "M_0.5_SEC_2HZ");
END_REGION

REGION Network 2: LAMP - START
   RUNG wire#powerrail
      Contact( "M_DUMMY_OFF" )
      Contact( "M_DUMMY_OFF" )
      Contact( "M_0.5_SEC_2HZ" )
      wire#w1
      Coil( "DB2141_HOPPER_UNIT_01_IN_OUT".LAMPS.START )
   END_RUNG
   RUNG wire#powerrail
      Contact( "M_DUMMY_OFF" )
   END_RUNG wire#w1
   // the same network as SCL:
   "DB2141_HOPPER_UNIT_01_IN_OUT".LAMPS.START := ("M_DUMMY_OFF" AND "M_DUMMY_OFF" AND "M_0.5_SEC_2HZ") OR "M_DUMMY_OFF";
END_REGION

REGION Network 3: LAMP - HOME
   RUNG wire#powerrail
      Contact( "M_DUMMY_OFF" )
      Contact( "M_1_SEC_1HZ" )
      wire#w1
      Coil( "DB2141_HOPPER_UNIT_01_IN_OUT".LAMPS.HOME_POSITION )
   END_RUNG
   RUNG wire#powerrail
      Contact( "M_DUMMY_OFF" )
      Contact( "M_DUMMY_OFF" )
      I_Contact( "M_DUMMY_OFF" )
      Contact( "M_2_SEC_0.5HZ" )
   END_RUNG wire#w1
   RUNG wire#powerrail
      Contact( "M_DUMMY_OFF" )
   END_RUNG wire#w1
   // the same network as SCL:
   "DB2141_HOPPER_UNIT_01_IN_OUT".LAMPS.HOME_POSITION := ("M_DUMMY_OFF" AND "M_1_SEC_1HZ") OR ("M_DUMMY_OFF" AND "M_DUMMY_OFF" AND NOT "M_DUMMY_OFF" AND "M_2_SEC_0.5HZ") OR "M_DUMMY_OFF";
END_REGION

REGION Network 4: LAMP - RESET FAULT
   RUNG wire#powerrail
      Contact( "DB442_HOPPERS_ALARM_DECODING".ALARMS_CENTRAL.ALARM )
      wire#w1
      Contact( "M_1_SEC_1HZ" )
      Coil( "DB2141_HOPPER_UNIT_01_IN_OUT".LAMPS.RESET_FAULTS )
   END_RUNG
   RUNG wire#powerrail
      Contact( "DB441_POWDER_FEEDERS_ALARM_DECODING".ALARMS_CENTRAL.ALARM )
   END_RUNG wire#w1
   // the same network as SCL:
   "DB2141_HOPPER_UNIT_01_IN_OUT".LAMPS.RESET_FAULTS := ("DB442_HOPPERS_ALARM_DECODING".ALARMS_CENTRAL.ALARM OR "DB441_POWDER_FEEDERS_ALARM_DECODING".ALARMS_CENTRAL.ALARM) AND "M_1_SEC_1HZ";
END_REGION

REGION Network 5: LAMP - CONTROL OFF
   RUNG wire#powerrail
      I_Contact( "DB2140_HOPPERS_MPP".MACHINE_ON_DELAYED )
      I_Contact( "DB2140_HOPPERS_MPP".MACH_ON_DEL_PNEU_ON )
      Coil( "DB2141_HOPPER_UNIT_01_IN_OUT".LAMPS.CONTROL_OFF )
   END_RUNG
   // the same network as SCL:
   "DB2141_HOPPER_UNIT_01_IN_OUT".LAMPS.CONTROL_OFF := NOT "DB2140_HOPPERS_MPP".MACHINE_ON_DELAYED AND NOT "DB2140_HOPPERS_MPP".MACH_ON_DEL_PNEU_ON;
END_REGION

REGION Network 6: LAMP - STOP END OF CYCLE
   RUNG wire#powerrail
      I_Contact( "DB442_HOPPERS_ALARM_DECODING".GLOBAL_ALARMS_MACHINE.SEOC_WARNING )
      I_Contact( "DB2140_HOPPERS_MPP".STOP_END_OF_CYCLE_BY_OPERATOR_AUX_1 )
      I_Contact( "DB2140_HOPPERS_MPP".STOP_END_OF_CYCLE_BY_OPERATOR_AUX_2 )
      Not()
      Contact( "M_0.5_SEC_2HZ" )
      Coil( "DB2141_HOPPER_UNIT_01_IN_OUT".LAMPS.STOP_END_OF_CYCLE )
   END_RUNG
   // the same network as SCL:
   "DB2141_HOPPER_UNIT_01_IN_OUT".LAMPS.STOP_END_OF_CYCLE := NOT (NOT "DB442_HOPPERS_ALARM_DECODING".GLOBAL_ALARMS_MACHINE.SEOC_WARNING AND NOT "DB2140_HOPPERS_MPP".STOP_END_OF_CYCLE_BY_OPERATOR_AUX_1 AND NOT "DB2140_HOPPERS_MPP".STOP_END_OF_CYCLE_BY_OPERATOR_AUX_2) AND "M_0.5_SEC_2HZ";
END_REGION

REGION Network 7: LAMP - IMMEDIATE STOP
   RUNG wire#powerrail
      Contact( "DB2140_HOPPERS_MPP".IMMEDIATE_STOP_BY_OPERATOR_AUX )
      Coil( "DB2141_HOPPER_UNIT_01_IN_OUT".LAMPS.INMEDIATE_STOP )
   END_RUNG
   // the same network as SCL:
   "DB2141_HOPPER_UNIT_01_IN_OUT".LAMPS.INMEDIATE_STOP := "DB2140_HOPPERS_MPP".IMMEDIATE_STOP_BY_OPERATOR_AUX;
END_REGION

REGION Network 8: LAMPS - MODES
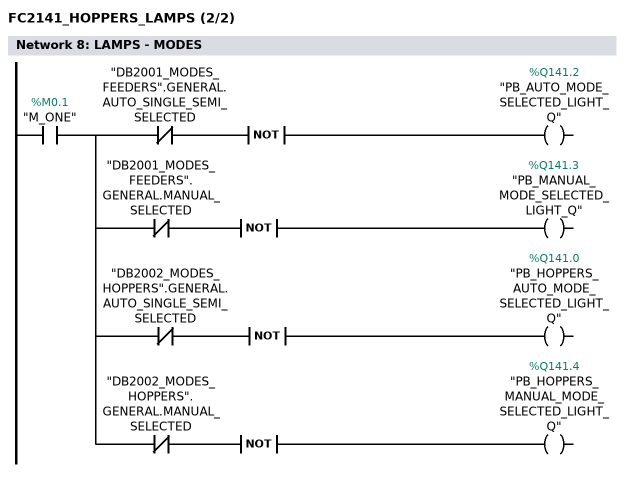
   RUNG wire#powerrail
      Contact( "M_ONE" )
      wire#w1
      I_Contact( "DB2001_MODES_FEEDERS".GENERAL.AUTO_SINGLE_SEMI_SELECTED )
      Not()
      Coil( "PB_AUTO_MODE_SELECTED_LIGHT_Q" )
   END_RUNG
   RUNG wire#w1
      I_Contact( "DB2001_MODES_FEEDERS".GENERAL.MANUAL_SELECTED )
      Not()
      Coil( "PB_MANUAL_MODE_SELECTED_LIGHT_Q" )
   END_RUNG
   RUNG wire#w1
      I_Contact( "DB2002_MODES_HOPPERS".GENERAL.AUTO_SINGLE_SEMI_SELECTED )
      Not()
      Coil( "PB_HOPPERS_AUTO_MODE_SELECTED_LIGHT_Q" )
   END_RUNG
   RUNG wire#w1
      I_Contact( "DB2002_MODES_HOPPERS".GENERAL.MANUAL_SELECTED )
      Not()
      Coil( "PB_HOPPERS_MANUAL_MODE_SELECTED_LIGHT_Q" )
   END_RUNG
   // the same network as SCL:
   "PB_AUTO_MODE_SELECTED_LIGHT_Q" := NOT ("M_ONE" AND NOT "DB2001_MODES_FEEDERS".GENERAL.AUTO_SINGLE_SEMI_SELECTED);
   "PB_MANUAL_MODE_SELECTED_LIGHT_Q" := NOT ("M_ONE" AND NOT "DB2001_MODES_FEEDERS".GENERAL.MANUAL_SELECTED);
   "PB_HOPPERS_AUTO_MODE_SELECTED_LIGHT_Q" := NOT ("M_ONE" AND NOT "DB2002_MODES_HOPPERS".GENERAL.AUTO_SINGLE_SEMI_SELECTED);
   "PB_HOPPERS_MANUAL_MODE_SELECTED_LIGHT_Q" := NOT ("M_ONE" AND NOT "DB2002_MODES_HOPPERS".GENERAL.MANUAL_SELECTED);
END_REGION
END_FUNCTION

FUNCTION "FC6500_CYLINDERS" : Void   // FC6500, LAD
{ S7_Optimized_Access := 'FALSE' }
AUTHOR : ETXETAR
VERSION : 1.0
// stored: AutoNumber false, IsIECCheckEnabled false, SetENOAutomatically false, UDAEnableTagReadback false
BEGIN

REGION Network 1: FC6600_UNIT_01_UP_SEALING_STRUCTURE
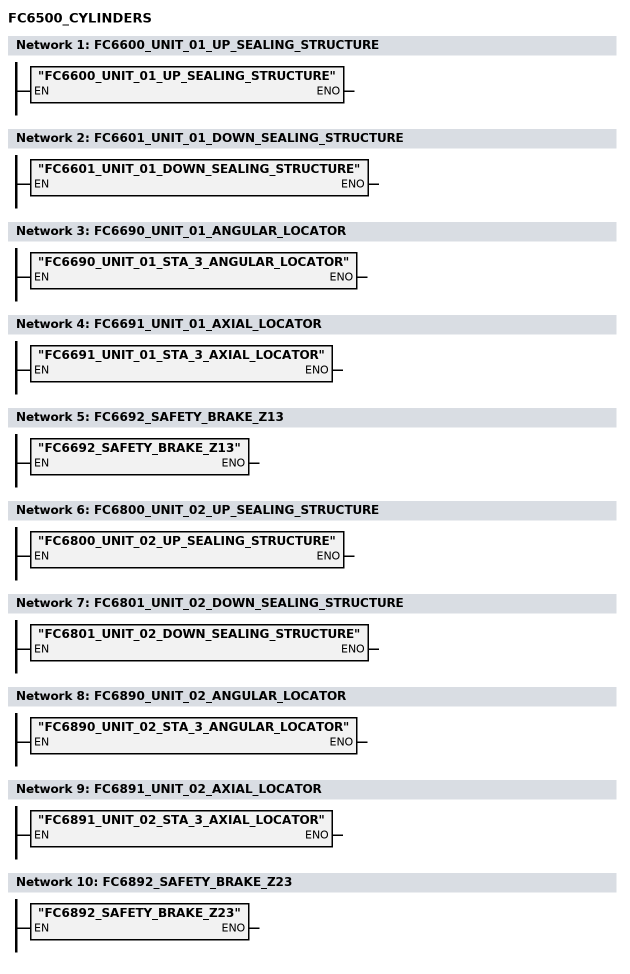
   RUNG wire#powerrail
      "FC6600_UNIT_01_UP_SEALING_STRUCTURE"()
   END_RUNG
   // the same network as SCL:
   "FC6600_UNIT_01_UP_SEALING_STRUCTURE"();
END_REGION

REGION Network 2: FC6601_UNIT_01_DOWN_SEALING_STRUCTURE
   RUNG wire#powerrail
      "FC6601_UNIT_01_DOWN_SEALING_STRUCTURE"()
   END_RUNG
   // the same network as SCL:
   "FC6601_UNIT_01_DOWN_SEALING_STRUCTURE"();
END_REGION

REGION Network 3: FC6690_UNIT_01_ANGULAR_LOCATOR
   RUNG wire#powerrail
      "FC6690_UNIT_01_STA_3_ANGULAR_LOCATOR"()
   END_RUNG
   // the same network as SCL:
   "FC6690_UNIT_01_STA_3_ANGULAR_LOCATOR"();
END_REGION

REGION Network 4: FC6691_UNIT_01_AXIAL_LOCATOR
   RUNG wire#powerrail
      "FC6691_UNIT_01_STA_3_AXIAL_LOCATOR"()
   END_RUNG
   // the same network as SCL:
   "FC6691_UNIT_01_STA_3_AXIAL_LOCATOR"();
END_REGION

REGION Network 5: FC6692_SAFETY_BRAKE_Z13
   RUNG wire#powerrail
      "FC6692_SAFETY_BRAKE_Z13"()
   END_RUNG
   // the same network as SCL:
   "FC6692_SAFETY_BRAKE_Z13"();
END_REGION

REGION Network 6: FC6800_UNIT_02_UP_SEALING_STRUCTURE
   RUNG wire#powerrail
      "FC6800_UNIT_02_UP_SEALING_STRUCTURE"()
   END_RUNG
   // the same network as SCL:
   "FC6800_UNIT_02_UP_SEALING_STRUCTURE"();
END_REGION

REGION Network 7: FC6801_UNIT_02_DOWN_SEALING_STRUCTURE
   RUNG wire#powerrail
      "FC6801_UNIT_02_DOWN_SEALING_STRUCTURE"()
   END_RUNG
   // the same network as SCL:
   "FC6801_UNIT_02_DOWN_SEALING_STRUCTURE"();
END_REGION

REGION Network 8: FC6890_UNIT_02_ANGULAR_LOCATOR
   RUNG wire#powerrail
      "FC6890_UNIT_02_STA_3_ANGULAR_LOCATOR"()
   END_RUNG
   // the same network as SCL:
   "FC6890_UNIT_02_STA_3_ANGULAR_LOCATOR"();
END_REGION

REGION Network 9: FC6891_UNIT_02_AXIAL_LOCATOR
   RUNG wire#powerrail
      "FC6891_UNIT_02_STA_3_AXIAL_LOCATOR"()
   END_RUNG
   // the same network as SCL:
   "FC6891_UNIT_02_STA_3_AXIAL_LOCATOR"();
END_REGION

REGION Network 10: FC6892_SAFETY_BRAKE_Z23
   RUNG wire#powerrail
      "FC6892_SAFETY_BRAKE_Z23"()
   END_RUNG
   // the same network as SCL:
   "FC6892_SAFETY_BRAKE_Z23"();
END_REGION
END_FUNCTION

FUNCTION "FC7000_SAFETY_DOORS" : Void   // FC7000, LAD
{ S7_Optimized_Access := 'FALSE' }
AUTHOR : ETXETAR
VERSION : 1.0
// stored: AutoNumber false, IsIECCheckEnabled false, SetENOAutomatically false, UDAEnableTagReadback false
BEGIN

REGION Network 1: CALL FC7002 UNIT 01 STATION 2 SAFETY DOOR
   // 2#0000_0001 OPTIONS 0 BIT 0 IMMEDIATE STOP REACTION OPTION
   // 2#0000_0010 OPTIONS 0 BIT 1 SEOC WARNING REACTION OPTION
   // 2#0000_0100 OPTIONS 0 BIT 2 CLOSED SENSOR INPUT OPTION
   // 2#0000_1000 OPTIONS 0 BIT 3 CIRCUIT E2 OPTION
   // 2#0001_0000 OPTIONS 0 BIT 4 PNEUMATIC DRIVE OPTION
   // 2#0010_0000 OPTIONS 0 BIT 5 GANTRY ROBOT OK TO OPEN OPTION
   // 2#0100_0000 OPTIONS 0 BIT 6 SPARE OPTION
   // 2#1000_0000 OPTIONS 0 BIT 7 SPARE OPTION
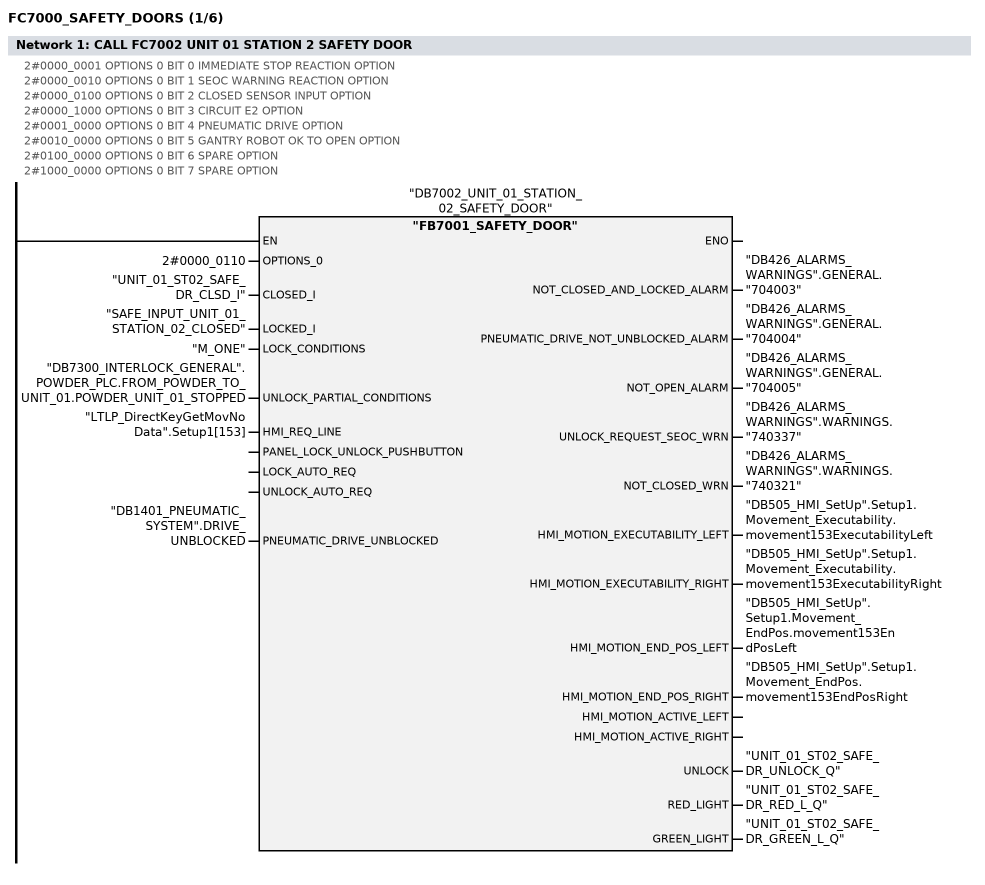
   RUNG wire#powerrail
      "DB7002_UNIT_01_STATION_02_SAFETY_DOOR"(OPTIONS_0 := 2#0000_0110, CLOSED_I := "UNIT_01_ST02_SAFE_DR_CLSD_I", LOCKED_I := "SAFE_INPUT_UNIT_01_STATION_02_CLOSED", LOCK_CONDITIONS := "M_ONE", UNLOCK_PARTIAL_CONDITIONS := "DB7300_INTERLOCK_GENERAL".POWDER_PLC.FROM_POWDER_TO_UNIT_01.POWDER_UNIT_01_STOPPED, HMI_REQ_LINE := "LTLP_DirectKeyGetMovNoData".Setup1[153], PANEL_LOCK_UNLOCK_PUSHBUTTON :=, LOCK_AUTO_REQ :=, UNLOCK_AUTO_REQ :=, PNEUMATIC_DRIVE_UNBLOCKED := "DB1401_PNEUMATIC_SYSTEM".DRIVE_UNBLOCKED, NOT_CLOSED_AND_LOCKED_ALARM => "DB426_ALARMS_WARNINGS".GENERAL."704003", PNEUMATIC_DRIVE_NOT_UNBLOCKED_ALARM => "DB426_ALARMS_WARNINGS".GENERAL."704004", NOT_OPEN_ALARM => "DB426_ALARMS_WARNINGS".GENERAL."704005", UNLOCK_REQUEST_SEOC_WRN => "DB426_ALARMS_WARNINGS".WARNINGS."740337", NOT_CLOSED_WRN => "DB426_ALARMS_WARNINGS".WARNINGS."740321", HMI_MOTION_EXECUTABILITY_LEFT => "DB505_HMI_SetUp".Setup1.Movement_Executability.movement153ExecutabilityLeft, HMI_MOTION_EXECUTABILITY_RIGHT => "DB505_HMI_SetUp".Setup1.Movement_Executability.movement153ExecutabilityRight, HMI_MOTION_END_POS_LEFT => "DB505_HMI_SetUp".Setup1.Movement_EndPos.movement153EndPosLeft, HMI_MOTION_END_POS_RIGHT => "DB505_HMI_SetUp".Setup1.Movement_EndPos.movement153EndPosRight, HMI_MOTION_ACTIVE_LEFT =>, HMI_MOTION_ACTIVE_RIGHT =>, UNLOCK => "UNIT_01_ST02_SAFE_DR_UNLOCK_Q", RED_LIGHT => "UNIT_01_ST02_SAFE_DR_RED_L_Q", GREEN_LIGHT => "UNIT_01_ST02_SAFE_DR_GREEN_L_Q")
   END_RUNG
   // the same network as SCL:
   "DB7002_UNIT_01_STATION_02_SAFETY_DOOR"(OPTIONS_0 := 2#0000_0110,   // "FB7001_SAFETY_DOOR"
                           CLOSED_I := "UNIT_01_ST02_SAFE_DR_CLSD_I",
                           LOCKED_I := "SAFE_INPUT_UNIT_01_STATION_02_CLOSED",
                           LOCK_CONDITIONS := "M_ONE",
                           UNLOCK_PARTIAL_CONDITIONS := "DB7300_INTERLOCK_GENERAL".POWDER_PLC.FROM_POWDER_TO_UNIT_01.POWDER_UNIT_01_STOPPED,
                           HMI_REQ_LINE := "LTLP_DirectKeyGetMovNoData".Setup1[153],
                           PNEUMATIC_DRIVE_UNBLOCKED := "DB1401_PNEUMATIC_SYSTEM".DRIVE_UNBLOCKED,
                           NOT_CLOSED_AND_LOCKED_ALARM => "DB426_ALARMS_WARNINGS".GENERAL."704003",
                           PNEUMATIC_DRIVE_NOT_UNBLOCKED_ALARM => "DB426_ALARMS_WARNINGS".GENERAL."704004",
                           NOT_OPEN_ALARM => "DB426_ALARMS_WARNINGS".GENERAL."704005",
                           UNLOCK_REQUEST_SEOC_WRN => "DB426_ALARMS_WARNINGS".WARNINGS."740337",
                           NOT_CLOSED_WRN => "DB426_ALARMS_WARNINGS".WARNINGS."740321",
                           HMI_MOTION_EXECUTABILITY_LEFT => "DB505_HMI_SetUp".Setup1.Movement_Executability.movement153ExecutabilityLeft,
                           HMI_MOTION_EXECUTABILITY_RIGHT => "DB505_HMI_SetUp".Setup1.Movement_Executability.movement153ExecutabilityRight,
                           HMI_MOTION_END_POS_LEFT => "DB505_HMI_SetUp".Setup1.Movement_EndPos.movement153EndPosLeft,
                           HMI_MOTION_END_POS_RIGHT => "DB505_HMI_SetUp".Setup1.Movement_EndPos.movement153EndPosRight,
                           UNLOCK => "UNIT_01_ST02_SAFE_DR_UNLOCK_Q",
                           RED_LIGHT => "UNIT_01_ST02_SAFE_DR_RED_L_Q",
                           GREEN_LIGHT => "UNIT_01_ST02_SAFE_DR_GREEN_L_Q");
END_REGION

REGION Network 2: CALL FC7002 UNIT 01 STATION 4 SAFETY DOOR
   // 2#0000_0001 OPTIONS 0 BIT 0 IMMEDIATE STOP REACTION OPTION
   // 2#0000_0010 OPTIONS 0 BIT 1 SEOC WARNING REACTION OPTION
   // 2#0000_0100 OPTIONS 0 BIT 2 CLOSED SENSOR INPUT OPTION
   // 2#0000_1000 OPTIONS 0 BIT 3 CIRCUIT E2 OPTION
   // 2#0001_0000 OPTIONS 0 BIT 4 PNEUMATIC DRIVE OPTION
   // 2#0010_0000 OPTIONS 0 BIT 5 GANTRY ROBOT OK TO OPEN OPTION
   // 2#0100_0000 OPTIONS 0 BIT 6 SPARE OPTION
   // 2#1000_0000 OPTIONS 0 BIT 7 SPARE OPTION
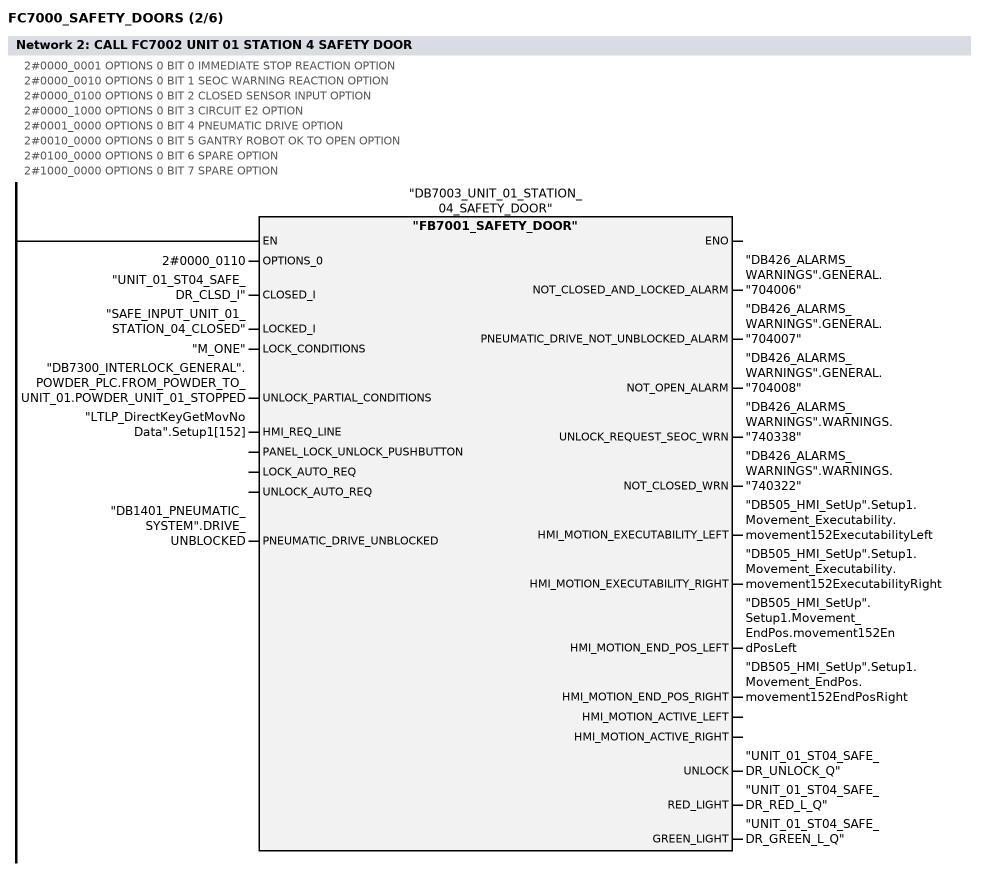
   RUNG wire#powerrail
      "DB7003_UNIT_01_STATION_04_SAFETY_DOOR"(OPTIONS_0 := 2#0000_0110, CLOSED_I := "UNIT_01_ST04_SAFE_DR_CLSD_I", LOCKED_I := "SAFE_INPUT_UNIT_01_STATION_04_CLOSED", LOCK_CONDITIONS := "M_ONE", UNLOCK_PARTIAL_CONDITIONS := "DB7300_INTERLOCK_GENERAL".POWDER_PLC.FROM_POWDER_TO_UNIT_01.POWDER_UNIT_01_STOPPED, HMI_REQ_LINE := "LTLP_DirectKeyGetMovNoData".Setup1[152], PANEL_LOCK_UNLOCK_PUSHBUTTON :=, LOCK_AUTO_REQ :=, UNLOCK_AUTO_REQ :=, PNEUMATIC_DRIVE_UNBLOCKED := "DB1401_PNEUMATIC_SYSTEM".DRIVE_UNBLOCKED, NOT_CLOSED_AND_LOCKED_ALARM => "DB426_ALARMS_WARNINGS".GENERAL."704006", PNEUMATIC_DRIVE_NOT_UNBLOCKED_ALARM => "DB426_ALARMS_WARNINGS".GENERAL."704007", NOT_OPEN_ALARM => "DB426_ALARMS_WARNINGS".GENERAL."704008", UNLOCK_REQUEST_SEOC_WRN => "DB426_ALARMS_WARNINGS".WARNINGS."740338", NOT_CLOSED_WRN => "DB426_ALARMS_WARNINGS".WARNINGS."740322", HMI_MOTION_EXECUTABILITY_LEFT => "DB505_HMI_SetUp".Setup1.Movement_Executability.movement152ExecutabilityLeft, HMI_MOTION_EXECUTABILITY_RIGHT => "DB505_HMI_SetUp".Setup1.Movement_Executability.movement152ExecutabilityRight, HMI_MOTION_END_POS_LEFT => "DB505_HMI_SetUp".Setup1.Movement_EndPos.movement152EndPosLeft, HMI_MOTION_END_POS_RIGHT => "DB505_HMI_SetUp".Setup1.Movement_EndPos.movement152EndPosRight, HMI_MOTION_ACTIVE_LEFT =>, HMI_MOTION_ACTIVE_RIGHT =>, UNLOCK => "UNIT_01_ST04_SAFE_DR_UNLOCK_Q", RED_LIGHT => "UNIT_01_ST04_SAFE_DR_RED_L_Q", GREEN_LIGHT => "UNIT_01_ST04_SAFE_DR_GREEN_L_Q")
   END_RUNG
   // the same network as SCL:
   "DB7003_UNIT_01_STATION_04_SAFETY_DOOR"(OPTIONS_0 := 2#0000_0110,   // "FB7001_SAFETY_DOOR"
                           CLOSED_I := "UNIT_01_ST04_SAFE_DR_CLSD_I",
                           LOCKED_I := "SAFE_INPUT_UNIT_01_STATION_04_CLOSED",
                           LOCK_CONDITIONS := "M_ONE",
                           UNLOCK_PARTIAL_CONDITIONS := "DB7300_INTERLOCK_GENERAL".POWDER_PLC.FROM_POWDER_TO_UNIT_01.POWDER_UNIT_01_STOPPED,
                           HMI_REQ_LINE := "LTLP_DirectKeyGetMovNoData".Setup1[152],
                           PNEUMATIC_DRIVE_UNBLOCKED := "DB1401_PNEUMATIC_SYSTEM".DRIVE_UNBLOCKED,
                           NOT_CLOSED_AND_LOCKED_ALARM => "DB426_ALARMS_WARNINGS".GENERAL."704006",
                           PNEUMATIC_DRIVE_NOT_UNBLOCKED_ALARM => "DB426_ALARMS_WARNINGS".GENERAL."704007",
                           NOT_OPEN_ALARM => "DB426_ALARMS_WARNINGS".GENERAL."704008",
                           UNLOCK_REQUEST_SEOC_WRN => "DB426_ALARMS_WARNINGS".WARNINGS."740338",
                           NOT_CLOSED_WRN => "DB426_ALARMS_WARNINGS".WARNINGS."740322",
                           HMI_MOTION_EXECUTABILITY_LEFT => "DB505_HMI_SetUp".Setup1.Movement_Executability.movement152ExecutabilityLeft,
                           HMI_MOTION_EXECUTABILITY_RIGHT => "DB505_HMI_SetUp".Setup1.Movement_Executability.movement152ExecutabilityRight,
                           HMI_MOTION_END_POS_LEFT => "DB505_HMI_SetUp".Setup1.Movement_EndPos.movement152EndPosLeft,
                           HMI_MOTION_END_POS_RIGHT => "DB505_HMI_SetUp".Setup1.Movement_EndPos.movement152EndPosRight,
                           UNLOCK => "UNIT_01_ST04_SAFE_DR_UNLOCK_Q",
                           RED_LIGHT => "UNIT_01_ST04_SAFE_DR_RED_L_Q",
                           GREEN_LIGHT => "UNIT_01_ST04_SAFE_DR_GREEN_L_Q");
END_REGION

REGION Network 3: CALL FC7001 UNIT 01 MAIN SAFETY DOOR
   // 2#0000_0001 OPTIONS 0 BIT 0 IMMEDIATE STOP REACTION OPTION
   // 2#0000_0010 OPTIONS 0 BIT 1 SEOC WARNING REACTION OPTION
   // 2#0000_0100 OPTIONS 0 BIT 2 CLOSED SENSOR INPUT OPTION
   // 2#0000_1000 OPTIONS 0 BIT 3 CIRCUIT E2 OPTION
   // 2#0001_0000 OPTIONS 0 BIT 4 PNEUMATIC DRIVE OPTION
   // 2#0010_0000 OPTIONS 0 BIT 5 GANTRY ROBOT OK TO OPEN OPTION
   // 2#0100_0000 OPTIONS 0 BIT 6 SPARE OPTION
   // 2#1000_0000 OPTIONS 0 BIT 7 SPARE OPTION
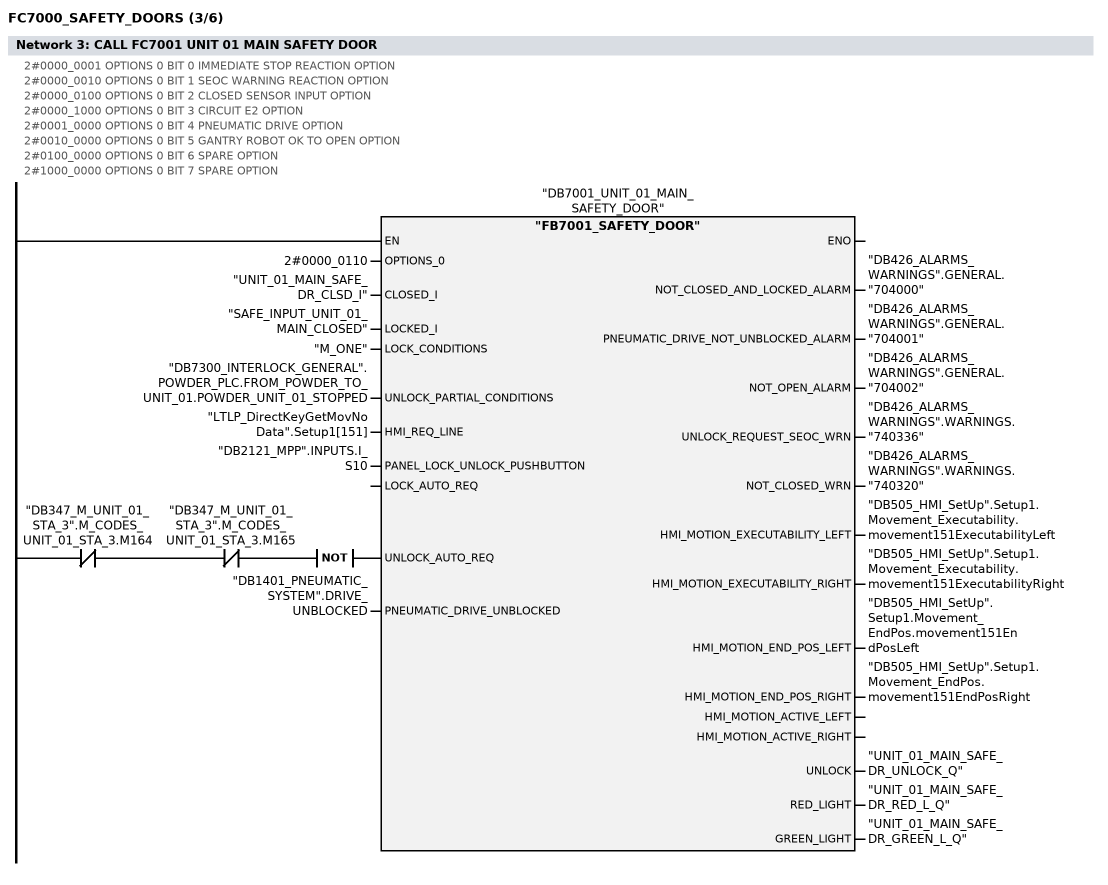
   RUNG wire#powerrail
      "DB7001_UNIT_01_MAIN_SAFETY_DOOR"(UNLOCK_AUTO_REQ := wire#w1, OPTIONS_0 := 2#0000_0110, CLOSED_I := "UNIT_01_MAIN_SAFE_DR_CLSD_I", LOCKED_I := "SAFE_INPUT_UNIT_01_MAIN_CLOSED", LOCK_CONDITIONS := "M_ONE", UNLOCK_PARTIAL_CONDITIONS := "DB7300_INTERLOCK_GENERAL".POWDER_PLC.FROM_POWDER_TO_UNIT_01.POWDER_UNIT_01_STOPPED, HMI_REQ_LINE := "LTLP_DirectKeyGetMovNoData".Setup1[151], PANEL_LOCK_UNLOCK_PUSHBUTTON := "DB2121_MPP".INPUTS.I_S10, LOCK_AUTO_REQ :=, PNEUMATIC_DRIVE_UNBLOCKED := "DB1401_PNEUMATIC_SYSTEM".DRIVE_UNBLOCKED, NOT_CLOSED_AND_LOCKED_ALARM => "DB426_ALARMS_WARNINGS".GENERAL."704000", PNEUMATIC_DRIVE_NOT_UNBLOCKED_ALARM => "DB426_ALARMS_WARNINGS".GENERAL."704001", NOT_OPEN_ALARM => "DB426_ALARMS_WARNINGS".GENERAL."704002", UNLOCK_REQUEST_SEOC_WRN => "DB426_ALARMS_WARNINGS".WARNINGS."740336", NOT_CLOSED_WRN => "DB426_ALARMS_WARNINGS".WARNINGS."740320", HMI_MOTION_EXECUTABILITY_LEFT => "DB505_HMI_SetUp".Setup1.Movement_Executability.movement151ExecutabilityLeft, HMI_MOTION_EXECUTABILITY_RIGHT => "DB505_HMI_SetUp".Setup1.Movement_Executability.movement151ExecutabilityRight, HMI_MOTION_END_POS_LEFT => "DB505_HMI_SetUp".Setup1.Movement_EndPos.movement151EndPosLeft, HMI_MOTION_END_POS_RIGHT => "DB505_HMI_SetUp".Setup1.Movement_EndPos.movement151EndPosRight, HMI_MOTION_ACTIVE_LEFT =>, HMI_MOTION_ACTIVE_RIGHT =>, UNLOCK => "UNIT_01_MAIN_SAFE_DR_UNLOCK_Q", RED_LIGHT => "UNIT_01_MAIN_SAFE_DR_RED_L_Q", GREEN_LIGHT => "UNIT_01_MAIN_SAFE_DR_GREEN_L_Q")
   END_RUNG
   RUNG wire#powerrail
      I_Contact( "DB347_M_UNIT_01_STA_3".M_CODES_UNIT_01_STA_3.M164 )
      I_Contact( "DB347_M_UNIT_01_STA_3".M_CODES_UNIT_01_STA_3.M165 )
      Not()
   END_RUNG wire#w1
   // the same network as SCL:
   "DB7001_UNIT_01_MAIN_SAFETY_DOOR"(OPTIONS_0 := 2#0000_0110,   // "FB7001_SAFETY_DOOR"
                           CLOSED_I := "UNIT_01_MAIN_SAFE_DR_CLSD_I",
                           LOCKED_I := "SAFE_INPUT_UNIT_01_MAIN_CLOSED",
                           LOCK_CONDITIONS := "M_ONE",
                           UNLOCK_PARTIAL_CONDITIONS := "DB7300_INTERLOCK_GENERAL".POWDER_PLC.FROM_POWDER_TO_UNIT_01.POWDER_UNIT_01_STOPPED,
                           HMI_REQ_LINE := "LTLP_DirectKeyGetMovNoData".Setup1[151],
                           PANEL_LOCK_UNLOCK_PUSHBUTTON := "DB2121_MPP".INPUTS.I_S10,
                           UNLOCK_AUTO_REQ := NOT (NOT "DB347_M_UNIT_01_STA_3".M_CODES_UNIT_01_STA_3.M164 AND NOT "DB347_M_UNIT_01_STA_3".M_CODES_UNIT_01_STA_3.M165),
                           PNEUMATIC_DRIVE_UNBLOCKED := "DB1401_PNEUMATIC_SYSTEM".DRIVE_UNBLOCKED,
                           NOT_CLOSED_AND_LOCKED_ALARM => "DB426_ALARMS_WARNINGS".GENERAL."704000",
                           PNEUMATIC_DRIVE_NOT_UNBLOCKED_ALARM => "DB426_ALARMS_WARNINGS".GENERAL."704001",
                           NOT_OPEN_ALARM => "DB426_ALARMS_WARNINGS".GENERAL."704002",
                           UNLOCK_REQUEST_SEOC_WRN => "DB426_ALARMS_WARNINGS".WARNINGS."740336",
                           NOT_CLOSED_WRN => "DB426_ALARMS_WARNINGS".WARNINGS."740320",
                           HMI_MOTION_EXECUTABILITY_LEFT => "DB505_HMI_SetUp".Setup1.Movement_Executability.movement151ExecutabilityLeft,
                           HMI_MOTION_EXECUTABILITY_RIGHT => "DB505_HMI_SetUp".Setup1.Movement_Executability.movement151ExecutabilityRight,
                           HMI_MOTION_END_POS_LEFT => "DB505_HMI_SetUp".Setup1.Movement_EndPos.movement151EndPosLeft,
                           HMI_MOTION_END_POS_RIGHT => "DB505_HMI_SetUp".Setup1.Movement_EndPos.movement151EndPosRight,
                           UNLOCK => "UNIT_01_MAIN_SAFE_DR_UNLOCK_Q",
                           RED_LIGHT => "UNIT_01_MAIN_SAFE_DR_RED_L_Q",
                           GREEN_LIGHT => "UNIT_01_MAIN_SAFE_DR_GREEN_L_Q");
END_REGION

REGION Network 4: CALL FC7012 UNIT 02 STATION 2 SAFETY DOOR
   // 2#0000_0001 OPTIONS 0 BIT 0 IMMEDIATE STOP REACTION OPTION
   // 2#0000_0010 OPTIONS 0 BIT 1 SEOC WARNING REACTION OPTION
   // 2#0000_0100 OPTIONS 0 BIT 2 CLOSED SENSOR INPUT OPTION
   // 2#0000_1000 OPTIONS 0 BIT 3 CIRCUIT E2 OPTION
   // 2#0001_0000 OPTIONS 0 BIT 4 PNEUMATIC DRIVE OPTION
   // 2#0010_0000 OPTIONS 0 BIT 5 GANTRY ROBOT OK TO OPEN OPTION
   // 2#0100_0000 OPTIONS 0 BIT 6 SPARE OPTION
   // 2#1000_0000 OPTIONS 0 BIT 7 SPARE OPTION
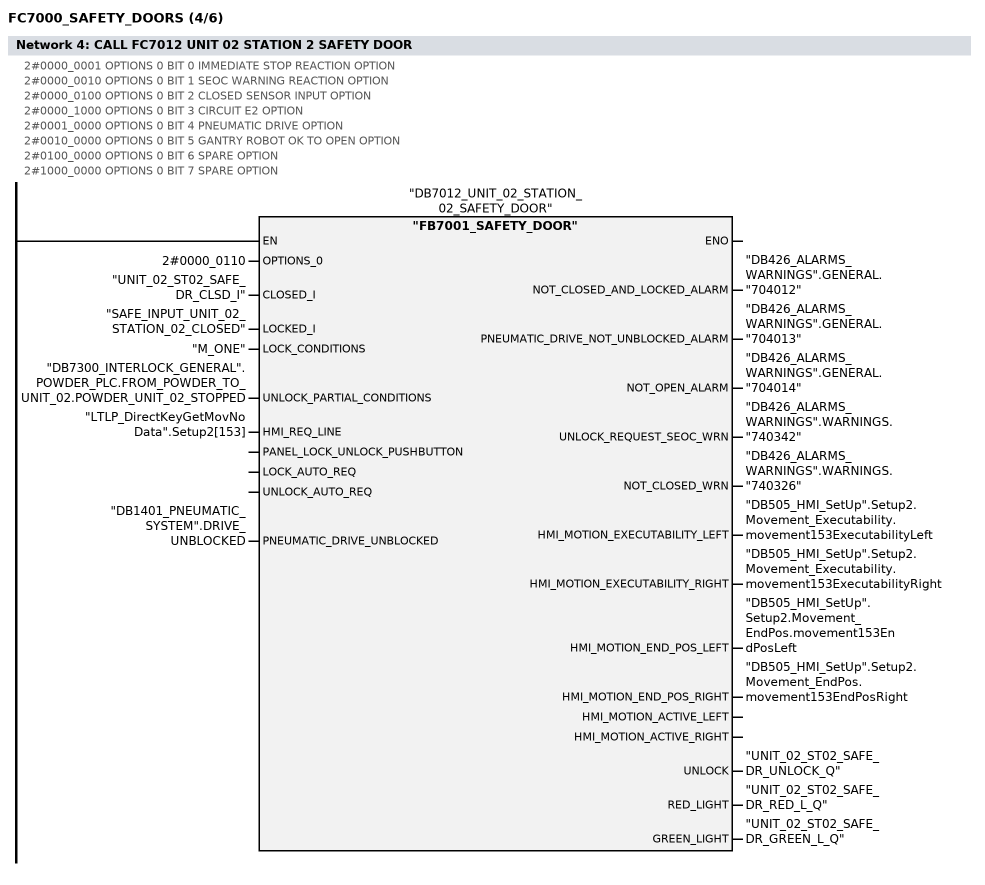
   RUNG wire#powerrail
      "DB7012_UNIT_02_STATION_02_SAFETY_DOOR"(OPTIONS_0 := 2#0000_0110, CLOSED_I := "UNIT_02_ST02_SAFE_DR_CLSD_I", LOCKED_I := "SAFE_INPUT_UNIT_02_STATION_02_CLOSED", LOCK_CONDITIONS := "M_ONE", UNLOCK_PARTIAL_CONDITIONS := "DB7300_INTERLOCK_GENERAL".POWDER_PLC.FROM_POWDER_TO_UNIT_02.POWDER_UNIT_02_STOPPED, HMI_REQ_LINE := "LTLP_DirectKeyGetMovNoData".Setup2[153], PANEL_LOCK_UNLOCK_PUSHBUTTON :=, LOCK_AUTO_REQ :=, UNLOCK_AUTO_REQ :=, PNEUMATIC_DRIVE_UNBLOCKED := "DB1401_PNEUMATIC_SYSTEM".DRIVE_UNBLOCKED, NOT_CLOSED_AND_LOCKED_ALARM => "DB426_ALARMS_WARNINGS".GENERAL."704012", PNEUMATIC_DRIVE_NOT_UNBLOCKED_ALARM => "DB426_ALARMS_WARNINGS".GENERAL."704013", NOT_OPEN_ALARM => "DB426_ALARMS_WARNINGS".GENERAL."704014", UNLOCK_REQUEST_SEOC_WRN => "DB426_ALARMS_WARNINGS".WARNINGS."740342", NOT_CLOSED_WRN => "DB426_ALARMS_WARNINGS".WARNINGS."740326", HMI_MOTION_EXECUTABILITY_LEFT => "DB505_HMI_SetUp".Setup2.Movement_Executability.movement153ExecutabilityLeft, HMI_MOTION_EXECUTABILITY_RIGHT => "DB505_HMI_SetUp".Setup2.Movement_Executability.movement153ExecutabilityRight, HMI_MOTION_END_POS_LEFT => "DB505_HMI_SetUp".Setup2.Movement_EndPos.movement153EndPosLeft, HMI_MOTION_END_POS_RIGHT => "DB505_HMI_SetUp".Setup2.Movement_EndPos.movement153EndPosRight, HMI_MOTION_ACTIVE_LEFT =>, HMI_MOTION_ACTIVE_RIGHT =>, UNLOCK => "UNIT_02_ST02_SAFE_DR_UNLOCK_Q", RED_LIGHT => "UNIT_02_ST02_SAFE_DR_RED_L_Q", GREEN_LIGHT => "UNIT_02_ST02_SAFE_DR_GREEN_L_Q")
   END_RUNG
   // the same network as SCL:
   "DB7012_UNIT_02_STATION_02_SAFETY_DOOR"(OPTIONS_0 := 2#0000_0110,   // "FB7001_SAFETY_DOOR"
                           CLOSED_I := "UNIT_02_ST02_SAFE_DR_CLSD_I",
                           LOCKED_I := "SAFE_INPUT_UNIT_02_STATION_02_CLOSED",
                           LOCK_CONDITIONS := "M_ONE",
                           UNLOCK_PARTIAL_CONDITIONS := "DB7300_INTERLOCK_GENERAL".POWDER_PLC.FROM_POWDER_TO_UNIT_02.POWDER_UNIT_02_STOPPED,
                           HMI_REQ_LINE := "LTLP_DirectKeyGetMovNoData".Setup2[153],
                           PNEUMATIC_DRIVE_UNBLOCKED := "DB1401_PNEUMATIC_SYSTEM".DRIVE_UNBLOCKED,
                           NOT_CLOSED_AND_LOCKED_ALARM => "DB426_ALARMS_WARNINGS".GENERAL."704012",
                           PNEUMATIC_DRIVE_NOT_UNBLOCKED_ALARM => "DB426_ALARMS_WARNINGS".GENERAL."704013",
                           NOT_OPEN_ALARM => "DB426_ALARMS_WARNINGS".GENERAL."704014",
                           UNLOCK_REQUEST_SEOC_WRN => "DB426_ALARMS_WARNINGS".WARNINGS."740342",
                           NOT_CLOSED_WRN => "DB426_ALARMS_WARNINGS".WARNINGS."740326",
                           HMI_MOTION_EXECUTABILITY_LEFT => "DB505_HMI_SetUp".Setup2.Movement_Executability.movement153ExecutabilityLeft,
                           HMI_MOTION_EXECUTABILITY_RIGHT => "DB505_HMI_SetUp".Setup2.Movement_Executability.movement153ExecutabilityRight,
                           HMI_MOTION_END_POS_LEFT => "DB505_HMI_SetUp".Setup2.Movement_EndPos.movement153EndPosLeft,
                           HMI_MOTION_END_POS_RIGHT => "DB505_HMI_SetUp".Setup2.Movement_EndPos.movement153EndPosRight,
                           UNLOCK => "UNIT_02_ST02_SAFE_DR_UNLOCK_Q",
                           RED_LIGHT => "UNIT_02_ST02_SAFE_DR_RED_L_Q",
                           GREEN_LIGHT => "UNIT_02_ST02_SAFE_DR_GREEN_L_Q");
END_REGION

REGION Network 5: CALL FC7013 UNIT 02 STATION 4 SAFETY DOOR
   // 2#0000_0001 OPTIONS 0 BIT 0 IMMEDIATE STOP REACTION OPTION
   // 2#0000_0010 OPTIONS 0 BIT 1 SEOC WARNING REACTION OPTION
   // 2#0000_0100 OPTIONS 0 BIT 2 CLOSED SENSOR INPUT OPTION
   // 2#0000_1000 OPTIONS 0 BIT 3 CIRCUIT E2 OPTION
   // 2#0001_0000 OPTIONS 0 BIT 4 PNEUMATIC DRIVE OPTION
   // 2#0010_0000 OPTIONS 0 BIT 5 GANTRY ROBOT OK TO OPEN OPTION
   // 2#0100_0000 OPTIONS 0 BIT 6 SPARE OPTION
   // 2#1000_0000 OPTIONS 0 BIT 7 SPARE OPTION
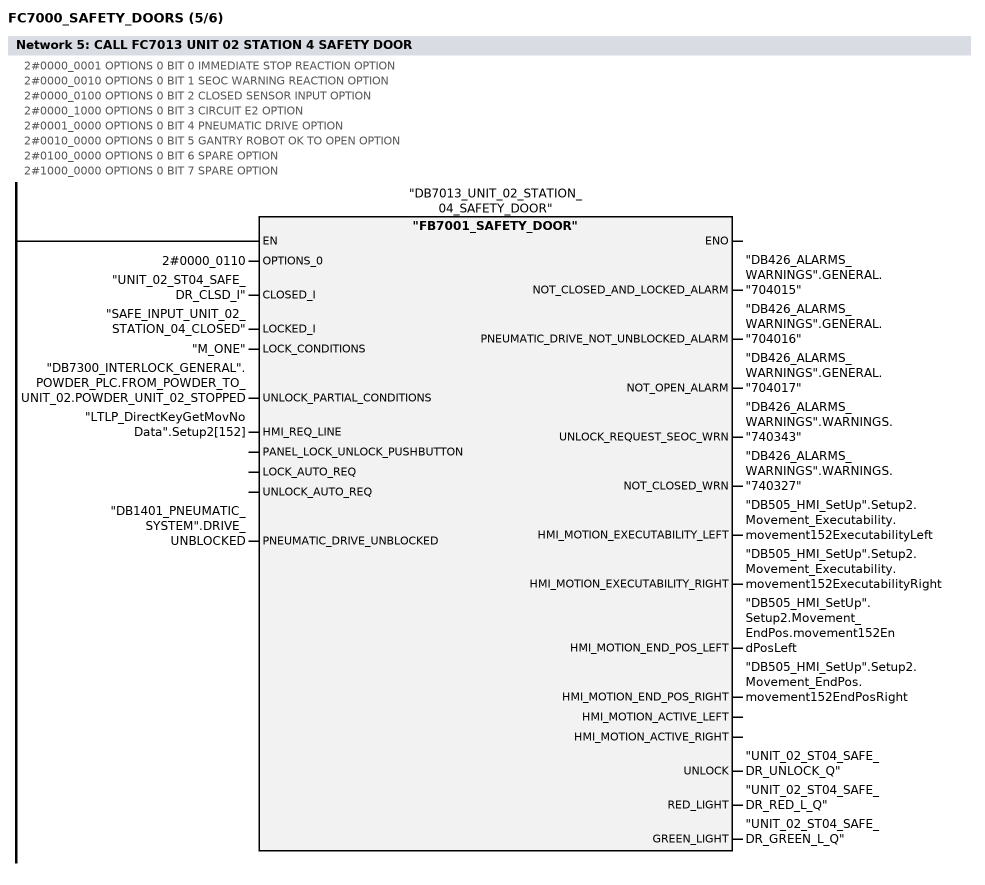
   RUNG wire#powerrail
      "DB7013_UNIT_02_STATION_04_SAFETY_DOOR"(OPTIONS_0 := 2#0000_0110, CLOSED_I := "UNIT_02_ST04_SAFE_DR_CLSD_I", LOCKED_I := "SAFE_INPUT_UNIT_02_STATION_04_CLOSED", LOCK_CONDITIONS := "M_ONE", UNLOCK_PARTIAL_CONDITIONS := "DB7300_INTERLOCK_GENERAL".POWDER_PLC.FROM_POWDER_TO_UNIT_02.POWDER_UNIT_02_STOPPED, HMI_REQ_LINE := "LTLP_DirectKeyGetMovNoData".Setup2[152], PANEL_LOCK_UNLOCK_PUSHBUTTON :=, LOCK_AUTO_REQ :=, UNLOCK_AUTO_REQ :=, PNEUMATIC_DRIVE_UNBLOCKED := "DB1401_PNEUMATIC_SYSTEM".DRIVE_UNBLOCKED, NOT_CLOSED_AND_LOCKED_ALARM => "DB426_ALARMS_WARNINGS".GENERAL."704015", PNEUMATIC_DRIVE_NOT_UNBLOCKED_ALARM => "DB426_ALARMS_WARNINGS".GENERAL."704016", NOT_OPEN_ALARM => "DB426_ALARMS_WARNINGS".GENERAL."704017", UNLOCK_REQUEST_SEOC_WRN => "DB426_ALARMS_WARNINGS".WARNINGS."740343", NOT_CLOSED_WRN => "DB426_ALARMS_WARNINGS".WARNINGS."740327", HMI_MOTION_EXECUTABILITY_LEFT => "DB505_HMI_SetUp".Setup2.Movement_Executability.movement152ExecutabilityLeft, HMI_MOTION_EXECUTABILITY_RIGHT => "DB505_HMI_SetUp".Setup2.Movement_Executability.movement152ExecutabilityRight, HMI_MOTION_END_POS_LEFT => "DB505_HMI_SetUp".Setup2.Movement_EndPos.movement152EndPosLeft, HMI_MOTION_END_POS_RIGHT => "DB505_HMI_SetUp".Setup2.Movement_EndPos.movement152EndPosRight, HMI_MOTION_ACTIVE_LEFT =>, HMI_MOTION_ACTIVE_RIGHT =>, UNLOCK => "UNIT_02_ST04_SAFE_DR_UNLOCK_Q", RED_LIGHT => "UNIT_02_ST04_SAFE_DR_RED_L_Q", GREEN_LIGHT => "UNIT_02_ST04_SAFE_DR_GREEN_L_Q")
   END_RUNG
   // the same network as SCL:
   "DB7013_UNIT_02_STATION_04_SAFETY_DOOR"(OPTIONS_0 := 2#0000_0110,   // "FB7001_SAFETY_DOOR"
                           CLOSED_I := "UNIT_02_ST04_SAFE_DR_CLSD_I",
                           LOCKED_I := "SAFE_INPUT_UNIT_02_STATION_04_CLOSED",
                           LOCK_CONDITIONS := "M_ONE",
                           UNLOCK_PARTIAL_CONDITIONS := "DB7300_INTERLOCK_GENERAL".POWDER_PLC.FROM_POWDER_TO_UNIT_02.POWDER_UNIT_02_STOPPED,
                           HMI_REQ_LINE := "LTLP_DirectKeyGetMovNoData".Setup2[152],
                           PNEUMATIC_DRIVE_UNBLOCKED := "DB1401_PNEUMATIC_SYSTEM".DRIVE_UNBLOCKED,
                           NOT_CLOSED_AND_LOCKED_ALARM => "DB426_ALARMS_WARNINGS".GENERAL."704015",
                           PNEUMATIC_DRIVE_NOT_UNBLOCKED_ALARM => "DB426_ALARMS_WARNINGS".GENERAL."704016",
                           NOT_OPEN_ALARM => "DB426_ALARMS_WARNINGS".GENERAL."704017",
                           UNLOCK_REQUEST_SEOC_WRN => "DB426_ALARMS_WARNINGS".WARNINGS."740343",
                           NOT_CLOSED_WRN => "DB426_ALARMS_WARNINGS".WARNINGS."740327",
                           HMI_MOTION_EXECUTABILITY_LEFT => "DB505_HMI_SetUp".Setup2.Movement_Executability.movement152ExecutabilityLeft,
                           HMI_MOTION_EXECUTABILITY_RIGHT => "DB505_HMI_SetUp".Setup2.Movement_Executability.movement152ExecutabilityRight,
                           HMI_MOTION_END_POS_LEFT => "DB505_HMI_SetUp".Setup2.Movement_EndPos.movement152EndPosLeft,
                           HMI_MOTION_END_POS_RIGHT => "DB505_HMI_SetUp".Setup2.Movement_EndPos.movement152EndPosRight,
                           UNLOCK => "UNIT_02_ST04_SAFE_DR_UNLOCK_Q",
                           RED_LIGHT => "UNIT_02_ST04_SAFE_DR_RED_L_Q",
                           GREEN_LIGHT => "UNIT_02_ST04_SAFE_DR_GREEN_L_Q");
END_REGION

REGION Network 6: CALL FC7011 UNIT 02 MAIN SAFETY DOOR
   // 2#0000_0001 OPTIONS 0 BIT 0 IMMEDIATE STOP REACTION OPTION
   // 2#0000_0010 OPTIONS 0 BIT 1 SEOC WARNING REACTION OPTION
   // 2#0000_0100 OPTIONS 0 BIT 2 CLOSED SENSOR INPUT OPTION
   // 2#0000_1000 OPTIONS 0 BIT 3 CIRCUIT E2 OPTION
   // 2#0001_0000 OPTIONS 0 BIT 4 PNEUMATIC DRIVE OPTION
   // 2#0010_0000 OPTIONS 0 BIT 5 GANTRY ROBOT OK TO OPEN OPTION
   // 2#0100_0000 OPTIONS 0 BIT 6 SPARE OPTION
   // 2#1000_0000 OPTIONS 0 BIT 7 SPARE OPTION
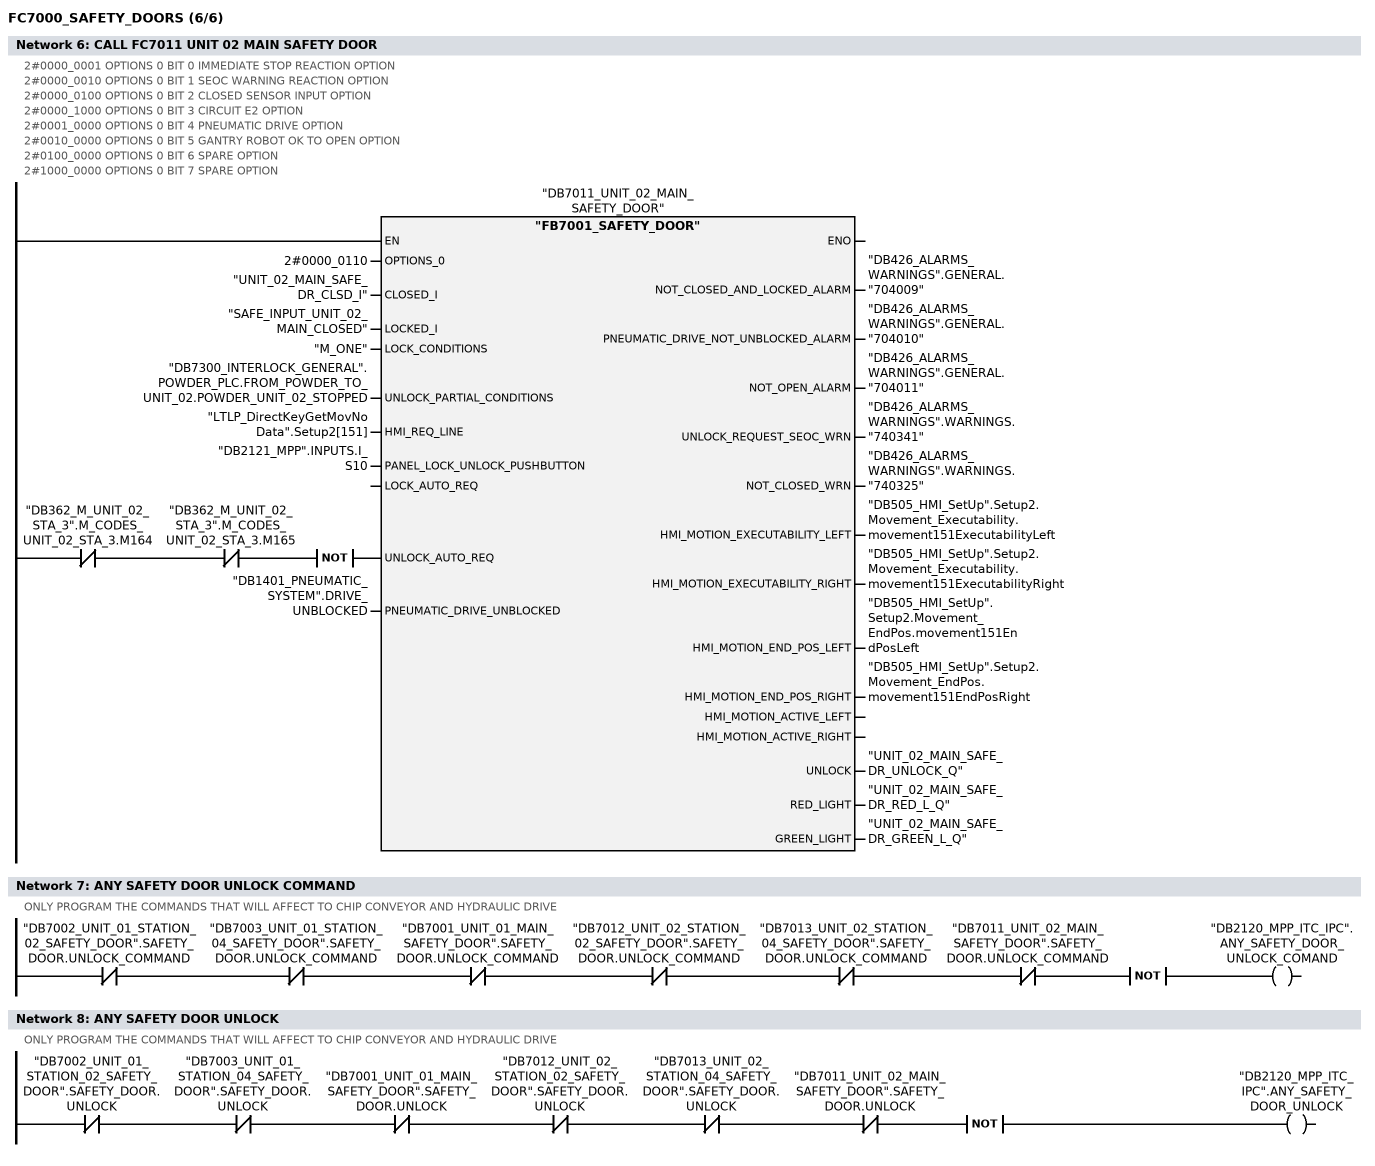
   RUNG wire#powerrail
      "DB7011_UNIT_02_MAIN_SAFETY_DOOR"(UNLOCK_AUTO_REQ := wire#w1, OPTIONS_0 := 2#0000_0110, CLOSED_I := "UNIT_02_MAIN_SAFE_DR_CLSD_I", LOCKED_I := "SAFE_INPUT_UNIT_02_MAIN_CLOSED", LOCK_CONDITIONS := "M_ONE", UNLOCK_PARTIAL_CONDITIONS := "DB7300_INTERLOCK_GENERAL".POWDER_PLC.FROM_POWDER_TO_UNIT_02.POWDER_UNIT_02_STOPPED, HMI_REQ_LINE := "LTLP_DirectKeyGetMovNoData".Setup2[151], PANEL_LOCK_UNLOCK_PUSHBUTTON := "DB2121_MPP".INPUTS.I_S10, LOCK_AUTO_REQ :=, PNEUMATIC_DRIVE_UNBLOCKED := "DB1401_PNEUMATIC_SYSTEM".DRIVE_UNBLOCKED, NOT_CLOSED_AND_LOCKED_ALARM => "DB426_ALARMS_WARNINGS".GENERAL."704009", PNEUMATIC_DRIVE_NOT_UNBLOCKED_ALARM => "DB426_ALARMS_WARNINGS".GENERAL."704010", NOT_OPEN_ALARM => "DB426_ALARMS_WARNINGS".GENERAL."704011", UNLOCK_REQUEST_SEOC_WRN => "DB426_ALARMS_WARNINGS".WARNINGS."740341", NOT_CLOSED_WRN => "DB426_ALARMS_WARNINGS".WARNINGS."740325", HMI_MOTION_EXECUTABILITY_LEFT => "DB505_HMI_SetUp".Setup2.Movement_Executability.movement151ExecutabilityLeft, HMI_MOTION_EXECUTABILITY_RIGHT => "DB505_HMI_SetUp".Setup2.Movement_Executability.movement151ExecutabilityRight, HMI_MOTION_END_POS_LEFT => "DB505_HMI_SetUp".Setup2.Movement_EndPos.movement151EndPosLeft, HMI_MOTION_END_POS_RIGHT => "DB505_HMI_SetUp".Setup2.Movement_EndPos.movement151EndPosRight, HMI_MOTION_ACTIVE_LEFT =>, HMI_MOTION_ACTIVE_RIGHT =>, UNLOCK => "UNIT_02_MAIN_SAFE_DR_UNLOCK_Q", RED_LIGHT => "UNIT_02_MAIN_SAFE_DR_RED_L_Q", GREEN_LIGHT => "UNIT_02_MAIN_SAFE_DR_GREEN_L_Q")
   END_RUNG
   RUNG wire#powerrail
      I_Contact( "DB362_M_UNIT_02_STA_3".M_CODES_UNIT_02_STA_3.M164 )
      I_Contact( "DB362_M_UNIT_02_STA_3".M_CODES_UNIT_02_STA_3.M165 )
      Not()
   END_RUNG wire#w1
   // the same network as SCL:
   "DB7011_UNIT_02_MAIN_SAFETY_DOOR"(OPTIONS_0 := 2#0000_0110,   // "FB7001_SAFETY_DOOR"
                           CLOSED_I := "UNIT_02_MAIN_SAFE_DR_CLSD_I",
                           LOCKED_I := "SAFE_INPUT_UNIT_02_MAIN_CLOSED",
                           LOCK_CONDITIONS := "M_ONE",
                           UNLOCK_PARTIAL_CONDITIONS := "DB7300_INTERLOCK_GENERAL".POWDER_PLC.FROM_POWDER_TO_UNIT_02.POWDER_UNIT_02_STOPPED,
                           HMI_REQ_LINE := "LTLP_DirectKeyGetMovNoData".Setup2[151],
                           PANEL_LOCK_UNLOCK_PUSHBUTTON := "DB2121_MPP".INPUTS.I_S10,
                           UNLOCK_AUTO_REQ := NOT (NOT "DB362_M_UNIT_02_STA_3".M_CODES_UNIT_02_STA_3.M164 AND NOT "DB362_M_UNIT_02_STA_3".M_CODES_UNIT_02_STA_3.M165),
                           PNEUMATIC_DRIVE_UNBLOCKED := "DB1401_PNEUMATIC_SYSTEM".DRIVE_UNBLOCKED,
                           NOT_CLOSED_AND_LOCKED_ALARM => "DB426_ALARMS_WARNINGS".GENERAL."704009",
                           PNEUMATIC_DRIVE_NOT_UNBLOCKED_ALARM => "DB426_ALARMS_WARNINGS".GENERAL."704010",
                           NOT_OPEN_ALARM => "DB426_ALARMS_WARNINGS".GENERAL."704011",
                           UNLOCK_REQUEST_SEOC_WRN => "DB426_ALARMS_WARNINGS".WARNINGS."740341",
                           NOT_CLOSED_WRN => "DB426_ALARMS_WARNINGS".WARNINGS."740325",
                           HMI_MOTION_EXECUTABILITY_LEFT => "DB505_HMI_SetUp".Setup2.Movement_Executability.movement151ExecutabilityLeft,
                           HMI_MOTION_EXECUTABILITY_RIGHT => "DB505_HMI_SetUp".Setup2.Movement_Executability.movement151ExecutabilityRight,
                           HMI_MOTION_END_POS_LEFT => "DB505_HMI_SetUp".Setup2.Movement_EndPos.movement151EndPosLeft,
                           HMI_MOTION_END_POS_RIGHT => "DB505_HMI_SetUp".Setup2.Movement_EndPos.movement151EndPosRight,
                           UNLOCK => "UNIT_02_MAIN_SAFE_DR_UNLOCK_Q",
                           RED_LIGHT => "UNIT_02_MAIN_SAFE_DR_RED_L_Q",
                           GREEN_LIGHT => "UNIT_02_MAIN_SAFE_DR_GREEN_L_Q");
END_REGION

REGION Network 7: ANY SAFETY DOOR UNLOCK COMMAND
   // ONLY PROGRAM THE COMMANDS THAT WILL AFFECT TO CHIP CONVEYOR AND HYDRAULIC DRIVE
   RUNG wire#powerrail
      I_Contact( "DB7002_UNIT_01_STATION_02_SAFETY_DOOR".SAFETY_DOOR.UNLOCK_COMMAND )
      I_Contact( "DB7003_UNIT_01_STATION_04_SAFETY_DOOR".SAFETY_DOOR.UNLOCK_COMMAND )
      I_Contact( "DB7001_UNIT_01_MAIN_SAFETY_DOOR".SAFETY_DOOR.UNLOCK_COMMAND )
      I_Contact( "DB7012_UNIT_02_STATION_02_SAFETY_DOOR".SAFETY_DOOR.UNLOCK_COMMAND )
      I_Contact( "DB7013_UNIT_02_STATION_04_SAFETY_DOOR".SAFETY_DOOR.UNLOCK_COMMAND )
      I_Contact( "DB7011_UNIT_02_MAIN_SAFETY_DOOR".SAFETY_DOOR.UNLOCK_COMMAND )
      Not()
      Coil( "DB2120_MPP_ITC_IPC".ANY_SAFETY_DOOR_UNLOCK_COMAND )
   END_RUNG
   // the same network as SCL:
   "DB2120_MPP_ITC_IPC".ANY_SAFETY_DOOR_UNLOCK_COMAND := NOT (NOT "DB7002_UNIT_01_STATION_02_SAFETY_DOOR".SAFETY_DOOR.UNLOCK_COMMAND AND NOT "DB7003_UNIT_01_STATION_04_SAFETY_DOOR".SAFETY_DOOR.UNLOCK_COMMAND AND NOT "DB7001_UNIT_01_MAIN_SAFETY_DOOR".SAFETY_DOOR.UNLOCK_COMMAND AND NOT "DB7012_UNIT_02_STATION_02_SAFETY_DOOR".SAFETY_DOOR.UNLOCK_COMMAND AND NOT "DB7013_UNIT_02_STATION_04_SAFETY_DOOR".SAFETY_DOOR.UNLOCK_COMMAND AND NOT "DB7011_UNIT_02_MAIN_SAFETY_DOOR".SAFETY_DOOR.UNLOCK_COMMAND);
END_REGION

REGION Network 8: ANY SAFETY DOOR UNLOCK
   // ONLY PROGRAM THE COMMANDS THAT WILL AFFECT TO CHIP CONVEYOR AND HYDRAULIC DRIVE
   RUNG wire#powerrail
      I_Contact( "DB7002_UNIT_01_STATION_02_SAFETY_DOOR".SAFETY_DOOR.UNLOCK )
      I_Contact( "DB7003_UNIT_01_STATION_04_SAFETY_DOOR".SAFETY_DOOR.UNLOCK )
      I_Contact( "DB7001_UNIT_01_MAIN_SAFETY_DOOR".SAFETY_DOOR.UNLOCK )
      I_Contact( "DB7012_UNIT_02_STATION_02_SAFETY_DOOR".SAFETY_DOOR.UNLOCK )
      I_Contact( "DB7013_UNIT_02_STATION_04_SAFETY_DOOR".SAFETY_DOOR.UNLOCK )
      I_Contact( "DB7011_UNIT_02_MAIN_SAFETY_DOOR".SAFETY_DOOR.UNLOCK )
      Not()
      Coil( "DB2120_MPP_ITC_IPC".ANY_SAFETY_DOOR_UNLOCK )
   END_RUNG
   // the same network as SCL:
   "DB2120_MPP_ITC_IPC".ANY_SAFETY_DOOR_UNLOCK := NOT (NOT "DB7002_UNIT_01_STATION_02_SAFETY_DOOR".SAFETY_DOOR.UNLOCK AND NOT "DB7003_UNIT_01_STATION_04_SAFETY_DOOR".SAFETY_DOOR.UNLOCK AND NOT "DB7001_UNIT_01_MAIN_SAFETY_DOOR".SAFETY_DOOR.UNLOCK AND NOT "DB7012_UNIT_02_STATION_02_SAFETY_DOOR".SAFETY_DOOR.UNLOCK AND NOT "DB7013_UNIT_02_STATION_04_SAFETY_DOOR".SAFETY_DOOR.UNLOCK AND NOT "DB7011_UNIT_02_MAIN_SAFETY_DOOR".SAFETY_DOOR.UNLOCK);
END_REGION
END_FUNCTION

FUNCTION_BLOCK "FB7001_SAFETY_DOOR"   // FB7001, LAD
{ S7_Optimized_Access := 'FALSE' }
AUTHOR : ETXETAR
VERSION : 1.0
// stored: AutoNumber false, IsIECCheckEnabled false, SetENOAutomatically false, UDAEnableTagReadback false
   VAR_INPUT
      OPTIONS_0 : Byte := 2#0000_0000;   // OPTIONS 0
      CLOSED_I : Bool;   // N.O / CLOSED INPUT
      LOCKED_I : Bool;   // N.O / LOCKED INPUT
      LOCK_CONDITIONS : Bool;   // LOCK CONDITIONS
      UNLOCK_PARTIAL_CONDITIONS : Bool;   // UNLOCK PARTIAL CONDITIONS
      HMI_REQ_LINE : Bool;   // HMI REQUEST LINE 1
      PANEL_LOCK_UNLOCK_PUSHBUTTON : Bool;   // PANEL LOCK UNLOCK PUSHBUTTON
      LOCK_AUTO_REQ : Bool;   // LOCK AUTO REQUEST
      UNLOCK_AUTO_REQ : Bool;   // UNLOCK AUTO REQUEST
      PNEUMATIC_DRIVE_UNBLOCKED : Bool;   // PNEUMATIC DRIVE 1 UNBLOCKED
   END_VAR
   VAR_OUTPUT
      NOT_CLOSED_AND_LOCKED_ALARM : Bool;   // NOT CLOSED AND LOCKED ALARM
      PNEUMATIC_DRIVE_NOT_UNBLOCKED_ALARM : Bool;   // PNEUMATIC DRIVE NOT UNBLOCKED ALARM
      NOT_OPEN_ALARM : Bool;   // NOT OPEN ALARM
      UNLOCK_REQUEST_SEOC_WRN : Bool;   // UNLOCK REQUEST SEOC WARNING
      NOT_CLOSED_WRN : Bool;   // NOT CLOSED WARNING
      HMI_MOTION_EXECUTABILITY_LEFT : Bool;   // HMI MOTION EXECUTABILITY LEFT
      HMI_MOTION_EXECUTABILITY_RIGHT : Bool;   // HMI MOTION EXECUTABILITY RIGHT
      HMI_MOTION_END_POS_LEFT : Bool;   // HMI MOTION END POSITION LEFT
      HMI_MOTION_END_POS_RIGHT : Bool;   // HMI MOTION END POSITION RIGHT
      HMI_MOTION_ACTIVE_LEFT : Bool;   // HMI MOTION ACTIVE LEFT
      HMI_MOTION_ACTIVE_RIGHT : Bool;   // HMI MOTION ACTIVE RIGHT
      UNLOCK : Bool;   // UNLOCK OUTPUT
      RED_LIGHT : Bool;   // RED LIGHT OUTPUT
      GREEN_LIGHT : Bool;   // GREEN LIGHT OUTPUT
   END_VAR
   VAR DB_SPECIFIC
      SAFETY_DOOR : "SAFETY_DOOR";
   END_VAR
   VAR_TEMP
      INPUTS_MASK : Byte;   // INPUTS_MASK
      O_BYTE_0 : Struct   // OPTIONS BYTE 0
         IMMEDIATE_STOP : Bool;   // IMMEDIATE STOP REACTION OPTION
         SEOC_WARNING : Bool;   // SEOC WARNING REACTION OPTION
         CLOSED_SENSOR : Bool;   // CLOSED SENSOR OPTION
         CIRCUIT_E2 : Bool;   // CIRCUIT E2 OPTION
         PNEUMATIC_DRIVE : Bool;   // PNEUMATIC DRIVE OPTION
         GANTRY_ROBOT_OK_TO_OPEN : Bool;   // GANTRY ROBOT OK TO OPEN SAFETY DOOR OPTION
         SPARE_6 : Bool;   // SPARE 6 OPTION
         SPARE_7 : Bool;   // SPARE 7 OPTION
      END_STRUCT;
      DB_NUMBER : DInt;   // DB NUMBER FOR ALARM AND HELP DECODING
   END_VAR
   // SAFETY_DOOR.TIMER_UNLOCK_PARTIAL_CONDITIONS.PT := T#250ms;
   // SAFETY_DOOR.TIMER_UNLOCK.PT := T#250ms;
   // SAFETY_DOOR.TIMER_PNEUMATIC_DRIVE_1_NOT_UNLOCKED.PT := T#2s;
   // SAFETY_DOOR.TIMER_NOT_OPEN.PT := T#3s;
   VAR_TEMP   // added for the SCL form of the ladder/FBD networks
      _w1 : Bool;
      _w2 : Bool;
   END_VAR
BEGIN

NETWORK
TITLE = READ INSTANCE DB
      L     DINO;
      +     10#800000;
      T     #DB_NUMBER;


REGION Network 2: OPTIONS
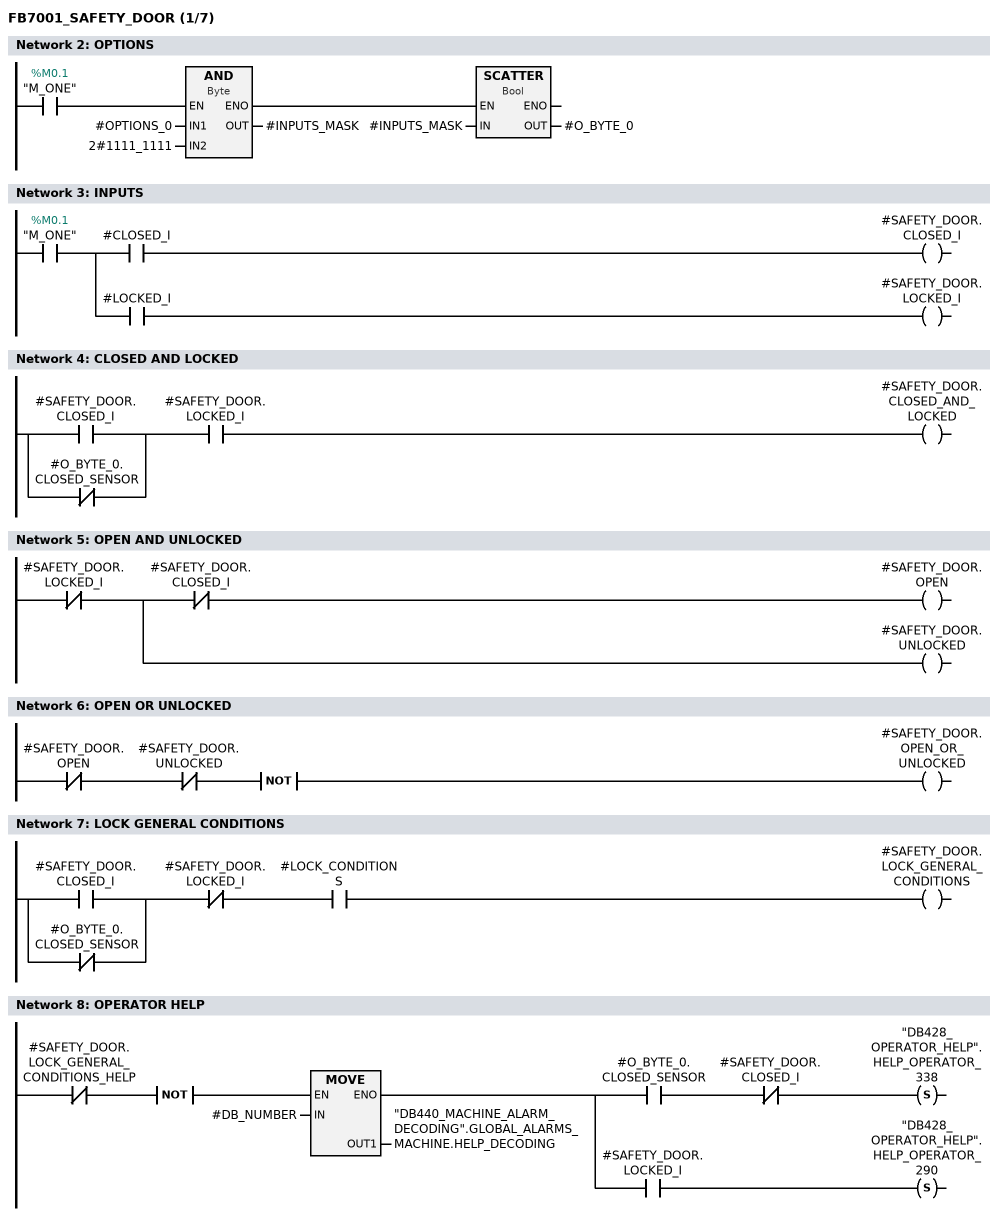
   RUNG wire#powerrail
      Contact( "M_ONE" )
      { S7_Templates := "SrcType := Byte"; S7_GenerateENO := "TRUE" } And(in1 := #OPTIONS_0, in2 := 2#1111_1111, out => #INPUTS_MASK)
      { S7_Templates := "[dest_type := Bool, src_type := Byte]" } SCATTER(IN := #INPUTS_MASK, OUT => #O_BYTE_0)
   END_RUNG
   // the same network as SCL:
   IF "M_ONE" THEN
       #INPUTS_MASK := #OPTIONS_0 AND 2#1111_1111;
       SCATTER(IN := #INPUTS_MASK, OUT => #O_BYTE_0);
   END_IF;
END_REGION

REGION Network 3: INPUTS
   RUNG wire#powerrail
      Contact( "M_ONE" )
      wire#w1
      Contact( #CLOSED_I )
      Coil( #SAFETY_DOOR.CLOSED_I )
   END_RUNG
   RUNG wire#w1
      Contact( #LOCKED_I )
      Coil( #SAFETY_DOOR.LOCKED_I )
   END_RUNG
   // the same network as SCL:
   #SAFETY_DOOR.CLOSED_I := "M_ONE" AND #CLOSED_I;
   #SAFETY_DOOR.LOCKED_I := "M_ONE" AND #LOCKED_I;
END_REGION

REGION Network 4: CLOSED AND LOCKED
   RUNG wire#powerrail
      Contact( #SAFETY_DOOR.CLOSED_I )
      wire#w1
      Contact( #SAFETY_DOOR.LOCKED_I )
      Coil( #SAFETY_DOOR.CLOSED_AND_LOCKED )
   END_RUNG
   RUNG wire#powerrail
      I_Contact( #O_BYTE_0.CLOSED_SENSOR )
   END_RUNG wire#w1
   // the same network as SCL:
   #SAFETY_DOOR.CLOSED_AND_LOCKED := (#SAFETY_DOOR.CLOSED_I OR NOT #O_BYTE_0.CLOSED_SENSOR) AND #SAFETY_DOOR.LOCKED_I;
END_REGION

REGION Network 5: OPEN AND UNLOCKED
   RUNG wire#powerrail
      I_Contact( #SAFETY_DOOR.LOCKED_I )
      wire#w1
      I_Contact( #SAFETY_DOOR.CLOSED_I )
      Coil( #SAFETY_DOOR.OPEN )
   END_RUNG
   RUNG wire#w1
      Coil( #SAFETY_DOOR.UNLOCKED )
   END_RUNG
   // the same network as SCL:
   #_w1 := NOT #SAFETY_DOOR.LOCKED_I;
   #SAFETY_DOOR.OPEN := #_w1 AND NOT #SAFETY_DOOR.CLOSED_I;
   #SAFETY_DOOR.UNLOCKED := #_w1;
END_REGION

REGION Network 6: OPEN OR UNLOCKED
   RUNG wire#powerrail
      I_Contact( #SAFETY_DOOR.OPEN )
      I_Contact( #SAFETY_DOOR.UNLOCKED )
      Not()
      Coil( #SAFETY_DOOR.OPEN_OR_UNLOCKED )
   END_RUNG
   // the same network as SCL:
   #SAFETY_DOOR.OPEN_OR_UNLOCKED := NOT (NOT #SAFETY_DOOR.OPEN AND NOT #SAFETY_DOOR.UNLOCKED);
END_REGION

REGION Network 7: LOCK GENERAL CONDITIONS
   RUNG wire#powerrail
      Contact( #SAFETY_DOOR.CLOSED_I )
      wire#w1
      I_Contact( #SAFETY_DOOR.LOCKED_I )
      Contact( #LOCK_CONDITIONS )
      Coil( #SAFETY_DOOR.LOCK_GENERAL_CONDITIONS )
   END_RUNG
   RUNG wire#powerrail
      I_Contact( #O_BYTE_0.CLOSED_SENSOR )
   END_RUNG wire#w1
   // the same network as SCL:
   #SAFETY_DOOR.LOCK_GENERAL_CONDITIONS := (#SAFETY_DOOR.CLOSED_I OR NOT #O_BYTE_0.CLOSED_SENSOR) AND NOT #SAFETY_DOOR.LOCKED_I AND #LOCK_CONDITIONS;
END_REGION

REGION Network 8: OPERATOR HELP
   RUNG wire#powerrail
      I_Contact( #SAFETY_DOOR.LOCK_GENERAL_CONDITIONS_HELP )
      Not()
      { S7_GenerateENO := "TRUE" } Move(in := #DB_NUMBER, out1 => "DB440_MACHINE_ALARM_DECODING".GLOBAL_ALARMS_MACHINE.HELP_DECODING)
      wire#w1
      Contact( #O_BYTE_0.CLOSED_SENSOR )
      I_Contact( #SAFETY_DOOR.CLOSED_I )
      S_Coil( "DB428_OPERATOR_HELP".HELP_OPERATOR_338 )
   END_RUNG
   RUNG wire#w1
      Contact( #SAFETY_DOOR.LOCKED_I )
      S_Coil( "DB428_OPERATOR_HELP".HELP_OPERATOR_290 )
   END_RUNG
   // the same network as SCL:
   // ENO of a box is taken as its EN; it also drops when the box reports an error
   #_w1 := NOT (NOT #SAFETY_DOOR.LOCK_GENERAL_CONDITIONS_HELP);
   IF #_w1 THEN "DB440_MACHINE_ALARM_DECODING".GLOBAL_ALARMS_MACHINE.HELP_DECODING := #DB_NUMBER; END_IF;
   IF #_w1 AND #O_BYTE_0.CLOSED_SENSOR AND NOT #SAFETY_DOOR.CLOSED_I THEN
       "DB428_OPERATOR_HELP".HELP_OPERATOR_338 := TRUE;
   END_IF;
   IF #_w1 AND #SAFETY_DOOR.LOCKED_I THEN "DB428_OPERATOR_HELP".HELP_OPERATOR_290 := TRUE; END_IF;
END_REGION

REGION Network 9: LOCK MANUAL REQUEST
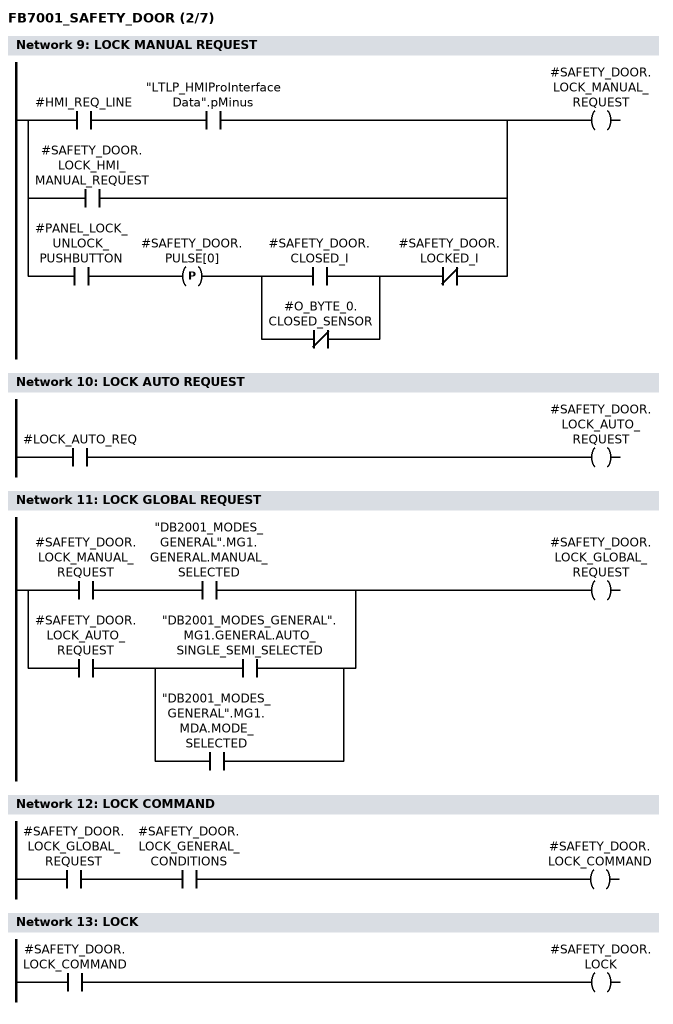
   RUNG wire#powerrail
      Contact( #HMI_REQ_LINE )
      Contact( "LTLP_HMIProInterfaceData".pMinus )
      wire#w1
      Coil( #SAFETY_DOOR.LOCK_MANUAL_REQUEST )
   END_RUNG
   RUNG wire#powerrail
      Contact( #SAFETY_DOOR.LOCK_HMI_MANUAL_REQUEST )
   END_RUNG wire#w1
   RUNG wire#powerrail
      Contact( #PANEL_LOCK_UNLOCK_PUSHBUTTON )
      P_Trig( #SAFETY_DOOR.PULSE[0] )
      wire#w2
      Contact( #SAFETY_DOOR.CLOSED_I )
      wire#w3
      I_Contact( #SAFETY_DOOR.LOCKED_I )
   END_RUNG wire#w1
   RUNG wire#w2
      I_Contact( #O_BYTE_0.CLOSED_SENSOR )
   END_RUNG wire#w3
   // the same network as SCL:
   #_w1 := #PANEL_LOCK_UNLOCK_PUSHBUTTON AND NOT #SAFETY_DOOR.PULSE[0];   // rising edge
   #SAFETY_DOOR.PULSE[0] := #PANEL_LOCK_UNLOCK_PUSHBUTTON;
   #SAFETY_DOOR.LOCK_MANUAL_REQUEST := (#HMI_REQ_LINE AND "LTLP_HMIProInterfaceData".pMinus) OR #SAFETY_DOOR.LOCK_HMI_MANUAL_REQUEST OR (#_w1 AND (#SAFETY_DOOR.CLOSED_I OR NOT #O_BYTE_0.CLOSED_SENSOR) AND NOT #SAFETY_DOOR.LOCKED_I);
END_REGION

REGION Network 10: LOCK AUTO REQUEST
   RUNG wire#powerrail
      Contact( #LOCK_AUTO_REQ )
      Coil( #SAFETY_DOOR.LOCK_AUTO_REQUEST )
   END_RUNG
   // the same network as SCL:
   #SAFETY_DOOR.LOCK_AUTO_REQUEST := #LOCK_AUTO_REQ;
END_REGION

REGION Network 11: LOCK GLOBAL REQUEST
   RUNG wire#powerrail
      Contact( #SAFETY_DOOR.LOCK_MANUAL_REQUEST )
      Contact( "DB2001_MODES_GENERAL".MG1.GENERAL.MANUAL_SELECTED )
      wire#w1
      Coil( #SAFETY_DOOR.LOCK_GLOBAL_REQUEST )
   END_RUNG
   RUNG wire#powerrail
      Contact( #SAFETY_DOOR.LOCK_AUTO_REQUEST )
      wire#w2
      Contact( "DB2001_MODES_GENERAL".MG1.GENERAL.AUTO_SINGLE_SEMI_SELECTED )
   END_RUNG wire#w1
   RUNG wire#w2
      Contact( "DB2001_MODES_GENERAL".MG1.MDA.MODE_SELECTED )
   END_RUNG wire#w1
   // the same network as SCL:
   #SAFETY_DOOR.LOCK_GLOBAL_REQUEST := (#SAFETY_DOOR.LOCK_MANUAL_REQUEST AND "DB2001_MODES_GENERAL".MG1.GENERAL.MANUAL_SELECTED) OR (#SAFETY_DOOR.LOCK_AUTO_REQUEST AND ("DB2001_MODES_GENERAL".MG1.GENERAL.AUTO_SINGLE_SEMI_SELECTED OR "DB2001_MODES_GENERAL".MG1.MDA.MODE_SELECTED));
END_REGION

REGION Network 12: LOCK COMMAND
   RUNG wire#powerrail
      Contact( #SAFETY_DOOR.LOCK_GLOBAL_REQUEST )
      Contact( #SAFETY_DOOR.LOCK_GENERAL_CONDITIONS )
      Coil( #SAFETY_DOOR.LOCK_COMMAND )
   END_RUNG
   // the same network as SCL:
   #SAFETY_DOOR.LOCK_COMMAND := #SAFETY_DOOR.LOCK_GLOBAL_REQUEST AND #SAFETY_DOOR.LOCK_GENERAL_CONDITIONS;
END_REGION

REGION Network 13: LOCK
   RUNG wire#powerrail
      Contact( #SAFETY_DOOR.LOCK_COMMAND )
      Coil( #SAFETY_DOOR.LOCK )
   END_RUNG
   // the same network as SCL:
   #SAFETY_DOOR.LOCK := #SAFETY_DOOR.LOCK_COMMAND;
END_REGION

REGION Network 14: UNLOCK PARTIAL CONDITIONS AUXILIARY
